REGION Network 1: CAN COT LIEU AGG1
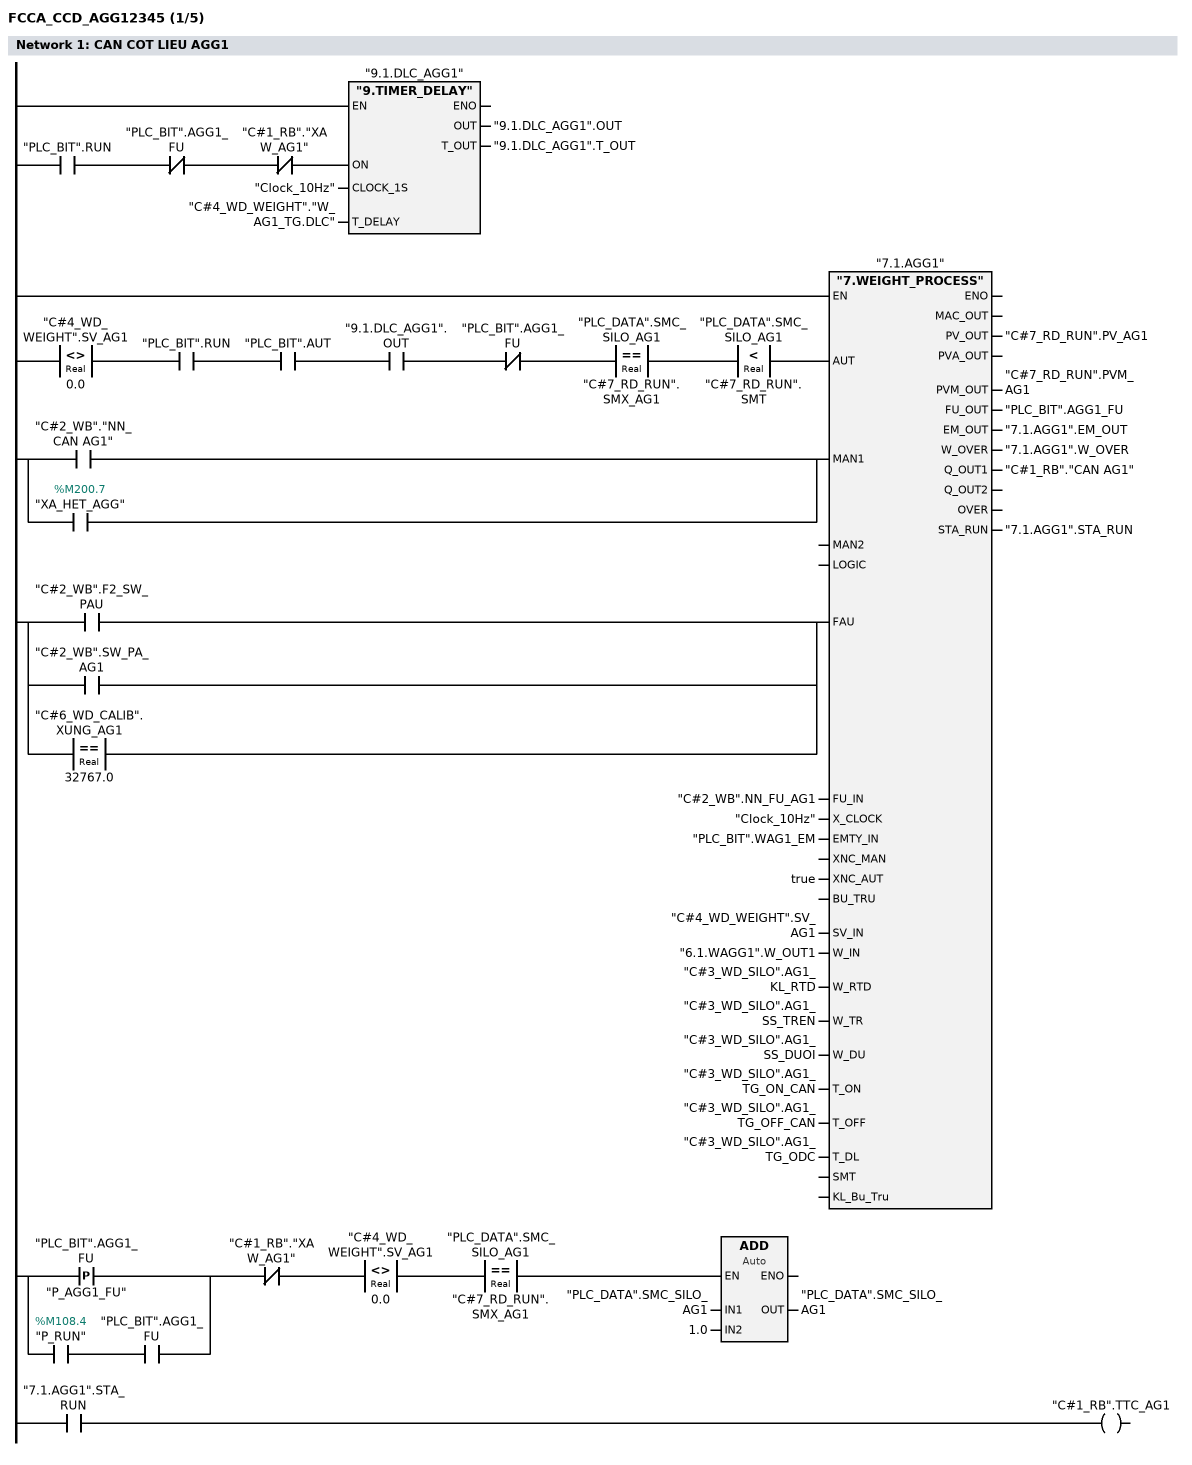
   RUNG wire#powerrail
      "9.1.DLC_AGG1"(ON := wire#w1, CLOCK_1S := "Clock_10Hz", T_DELAY := "C#4_WD_WEIGHT"."W_AG1_TG.DLC", OUT => "9.1.DLC_AGG1".OUT, T_OUT => "9.1.DLC_AGG1".T_OUT)
   END_RUNG
   RUNG wire#powerrail
      Contact( "PLC_BIT".RUN )
      I_Contact( "PLC_BIT".AGG1_FU )
      I_Contact( "C#1_RB"."XA W_AG1" )
   END_RUNG wire#w1
   RUNG wire#powerrail
      "7.1.AGG1"(AUT := wire#w2, MAN1 := wire#w3, FAU := wire#w4, MAN2 :=, LOGIC :=, FU_IN := "C#2_WB".NN_FU_AG1, X_CLOCK := "Clock_10Hz", EMTY_IN := "PLC_BIT".WAG1_EM, XNC_MAN :=, XNC_AUT := true, BU_TRU :=, SV_IN := "C#4_WD_WEIGHT".SV_AG1, W_IN := "6.1.WAGG1".W_OUT1, W_RTD := "C#3_WD_SILO".AG1_KL_RTD, W_TR := "C#3_WD_SILO".AG1_SS_TREN, W_DU := "C#3_WD_SILO".AG1_SS_DUOI, T_ON := "C#3_WD_SILO".AG1_TG_ON_CAN, T_OFF := "C#3_WD_SILO".AG1_TG_OFF_CAN, T_DL := "C#3_WD_SILO".AG1_TG_ODC, SMT :=, KL_Bu_Tru :=, MAC_OUT =>, PV_OUT => "C#7_RD_RUN".PV_AG1, PVA_OUT =>, PVM_OUT => "C#7_RD_RUN".PVM_AG1, FU_OUT => "PLC_BIT".AGG1_FU, EM_OUT => "7.1.AGG1".EM_OUT, W_OVER => "7.1.AGG1".W_OVER, Q_OUT1 => "C#1_RB"."CAN AG1", Q_OUT2 =>, OVER =>, STA_RUN => "7.1.AGG1".STA_RUN)
   END_RUNG
   RUNG wire#powerrail
      { S7_Templates := "SrcType := Real" } NE_Contact(in1 := "C#4_WD_WEIGHT".SV_AG1, in2 := 0.0)
      Contact( "PLC_BIT".RUN )
      Contact( "PLC_BIT".AUT )
      Contact( "9.1.DLC_AGG1".OUT )
      I_Contact( "PLC_BIT".AGG1_FU )
      { S7_Templates := "SrcType := Real" } EQ_Contact(in1 := "PLC_DATA".SMC_SILO_AG1, in2 := "C#7_RD_RUN".SMX_AG1)
      { S7_Templates := "SrcType := Real" } LT_Contact(in1 := "PLC_DATA".SMC_SILO_AG1, in2 := "C#7_RD_RUN".SMT)
   END_RUNG wire#w2
   RUNG wire#powerrail
      Contact( "C#2_WB"."NN_CAN AG1" )
   END_RUNG wire#w3
   RUNG wire#powerrail
      Contact( "XA_HET_AGG" )
   END_RUNG wire#w3
   RUNG wire#powerrail
      Contact( "C#2_WB".F2_SW_PAU )
   END_RUNG wire#w4
   RUNG wire#powerrail
      Contact( "C#2_WB".SW_PA_AG1 )
   END_RUNG wire#w4
   RUNG wire#powerrail
      { S7_Templates := "SrcType := Real" } EQ_Contact(in1 := "C#6_WD_CALIB".XUNG_AG1, in2 := 32767.0)
   END_RUNG wire#w4
   RUNG wire#powerrail
      P_Contact(operand := "PLC_BIT".AGG1_FU, bit := "P_AGG1_FU")
      wire#w5
      I_Contact( "C#1_RB"."XA W_AG1" )
      { S7_Templates := "SrcType := Real" } NE_Contact(in1 := "C#4_WD_WEIGHT".SV_AG1, in2 := 0.0)
      { S7_Templates := "SrcType := Real" } EQ_Contact(in1 := "PLC_DATA".SMC_SILO_AG1, in2 := "C#7_RD_RUN".SMX_AG1)
      Add(in1 := "PLC_DATA".SMC_SILO_AG1, in2 := 1.0, out => "PLC_DATA".SMC_SILO_AG1)
   END_RUNG
   RUNG wire#powerrail
      Contact( "P_RUN" )
      Contact( "PLC_BIT".AGG1_FU )
   END_RUNG wire#w5
   RUNG wire#powerrail
      Contact( "7.1.AGG1".STA_RUN )
      Coil( "C#1_RB".TTC_AG1 )
   END_RUNG
   // the same network as SCL:
   "9.1.DLC_AGG1"(ON := "PLC_BIT".RUN AND NOT "PLC_BIT".AGG1_FU AND NOT "C#1_RB"."XA W_AG1",   // "9.TIMER_DELAY"
                  CLOCK_1S := "Clock_10Hz",
                  T_DELAY := "C#4_WD_WEIGHT"."W_AG1_TG.DLC",
                  OUT => "9.1.DLC_AGG1".OUT,
                  T_OUT => "9.1.DLC_AGG1".T_OUT);
   "7.1.AGG1"(AUT := ("C#4_WD_WEIGHT".SV_AG1 <> 0.0) AND "PLC_BIT".RUN AND "PLC_BIT".AUT AND "9.1.DLC_AGG1".OUT AND NOT "PLC_BIT".AGG1_FU AND ("PLC_DATA".SMC_SILO_AG1 = "C#7_RD_RUN".SMX_AG1) AND ("PLC_DATA".SMC_SILO_AG1 < "C#7_RD_RUN".SMT),   // "7.WEIGHT_PROCESS"
              MAN1 := "C#2_WB"."NN_CAN AG1" OR "XA_HET_AGG",
              FAU := "C#2_WB".F2_SW_PAU OR "C#2_WB".SW_PA_AG1 OR ("C#6_WD_CALIB".XUNG_AG1 = 32767.0),
              FU_IN := "C#2_WB".NN_FU_AG1,
              X_CLOCK := "Clock_10Hz",
              EMTY_IN := "PLC_BIT".WAG1_EM,
              XNC_AUT := true,
              SV_IN := "C#4_WD_WEIGHT".SV_AG1,
              W_IN := "6.1.WAGG1".W_OUT1,
              W_RTD := "C#3_WD_SILO".AG1_KL_RTD,
              W_TR := "C#3_WD_SILO".AG1_SS_TREN,
              W_DU := "C#3_WD_SILO".AG1_SS_DUOI,
              T_ON := "C#3_WD_SILO".AG1_TG_ON_CAN,
              T_OFF := "C#3_WD_SILO".AG1_TG_OFF_CAN,
              T_DL := "C#3_WD_SILO".AG1_TG_ODC,
              PV_OUT => "C#7_RD_RUN".PV_AG1,
              PVM_OUT => "C#7_RD_RUN".PVM_AG1,
              FU_OUT => "PLC_BIT".AGG1_FU,
              EM_OUT => "7.1.AGG1".EM_OUT,
              W_OVER => "7.1.AGG1".W_OVER,
              Q_OUT1 => "C#1_RB"."CAN AG1",
              STA_RUN => "7.1.AGG1".STA_RUN);
   #_w1 := "PLC_BIT".AGG1_FU AND NOT "P_AGG1_FU";   // rising edge of "PLC_BIT".AGG1_FU
   "P_AGG1_FU" := "PLC_BIT".AGG1_FU;
   IF (#_w1 OR ("P_RUN" AND "PLC_BIT".AGG1_FU)) AND NOT "C#1_RB"."XA W_AG1" AND ("C#4_WD_WEIGHT".SV_AG1 <> 0.0) AND ("PLC_DATA".SMC_SILO_AG1 = "C#7_RD_RUN".SMX_AG1) THEN
       "PLC_DATA".SMC_SILO_AG1 := "PLC_DATA".SMC_SILO_AG1 + 1.0;
   END_IF;
   "C#1_RB".TTC_AG1 := "7.1.AGG1".STA_RUN;
END_REGION

REGION Network 2: CAN COT LIEU AGG2
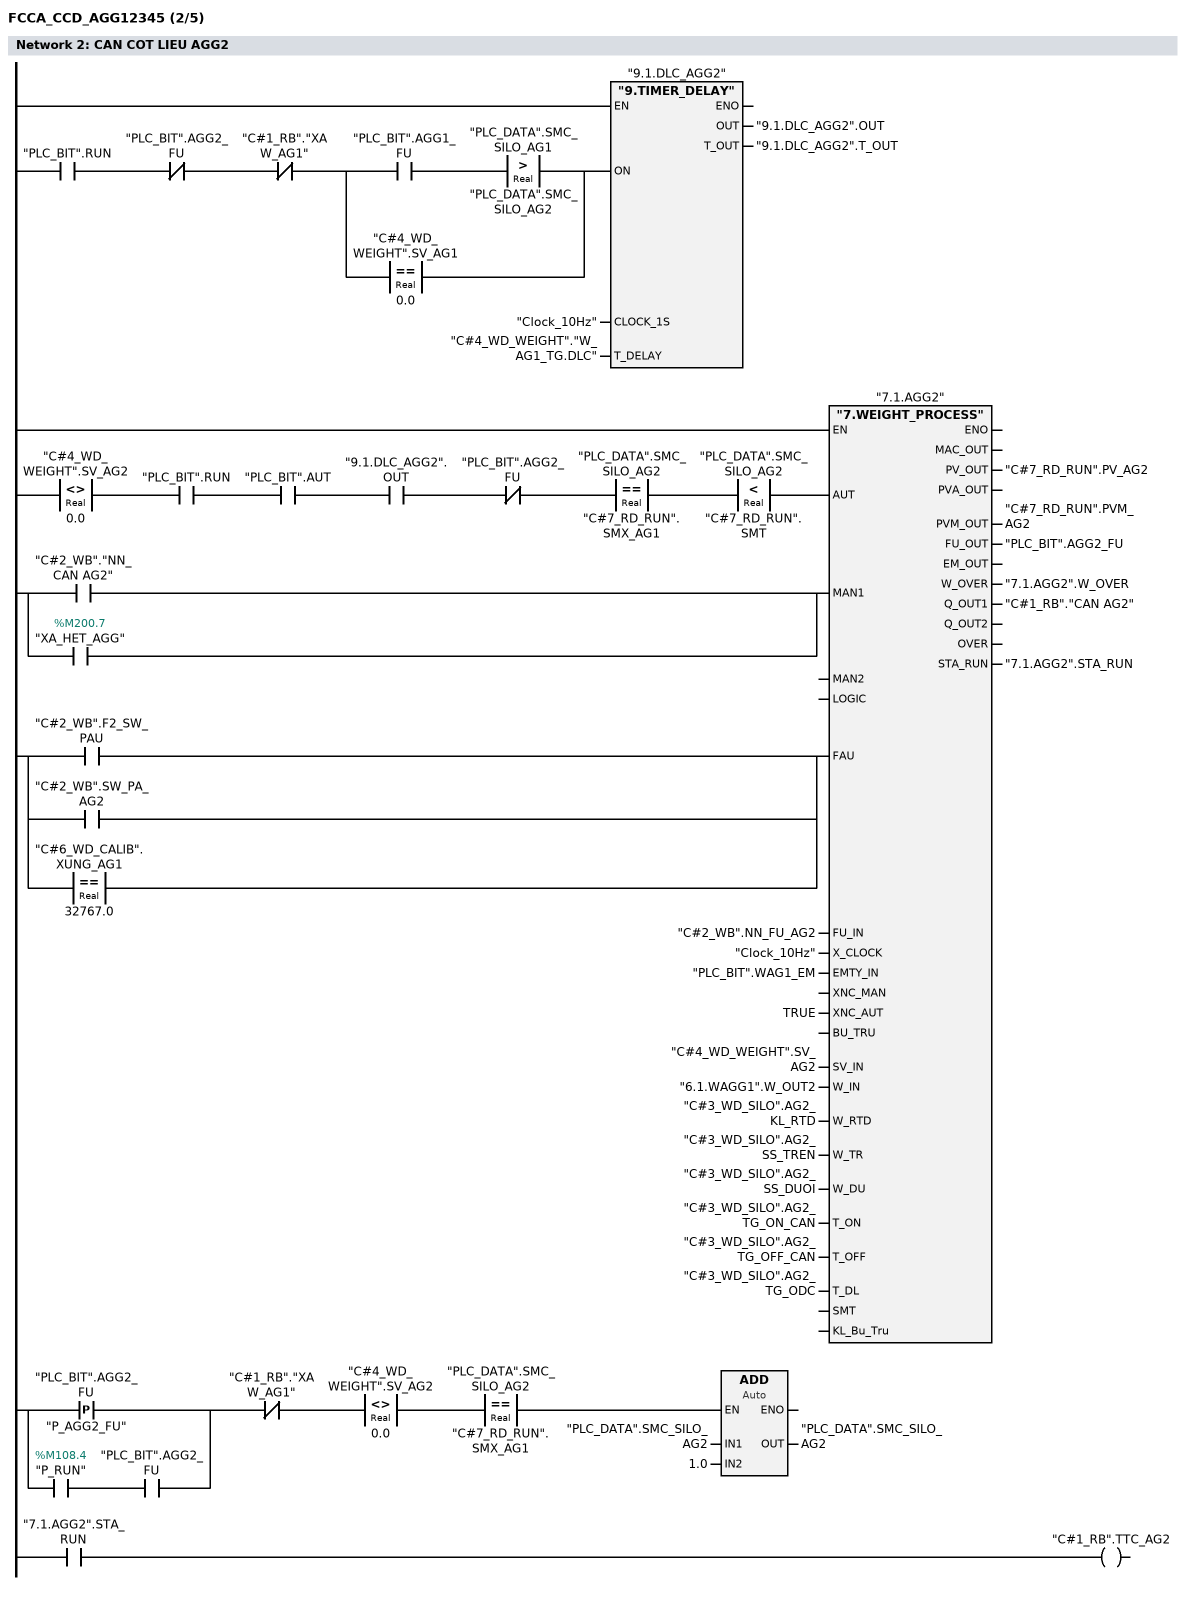
   RUNG wire#powerrail
      "9.1.DLC_AGG2"(ON := wire#w2, CLOCK_1S := "Clock_10Hz", T_DELAY := "C#4_WD_WEIGHT"."W_AG1_TG.DLC", OUT => "9.1.DLC_AGG2".OUT, T_OUT => "9.1.DLC_AGG2".T_OUT)
   END_RUNG
   RUNG wire#powerrail
      Contact( "PLC_BIT".RUN )
      I_Contact( "PLC_BIT".AGG2_FU )
      I_Contact( "C#1_RB"."XA W_AG1" )
      wire#w1
      Contact( "PLC_BIT".AGG1_FU )
      { S7_Templates := "SrcType := Real" } GT_Contact(in1 := "PLC_DATA".SMC_SILO_AG1, in2 := "PLC_DATA".SMC_SILO_AG2)
   END_RUNG wire#w2
   RUNG wire#w1
      { S7_Templates := "SrcType := Real" } EQ_Contact(in1 := "C#4_WD_WEIGHT".SV_AG1, in2 := 0.0)
   END_RUNG wire#w2
   RUNG wire#powerrail
      "7.1.AGG2"(AUT := wire#w3, MAN1 := wire#w4, FAU := wire#w5, MAN2 :=, LOGIC :=, FU_IN := "C#2_WB".NN_FU_AG2, X_CLOCK := "Clock_10Hz", EMTY_IN := "PLC_BIT".WAG1_EM, XNC_MAN :=, XNC_AUT := TRUE, BU_TRU :=, SV_IN := "C#4_WD_WEIGHT".SV_AG2, W_IN := "6.1.WAGG1".W_OUT2, W_RTD := "C#3_WD_SILO".AG2_KL_RTD, W_TR := "C#3_WD_SILO".AG2_SS_TREN, W_DU := "C#3_WD_SILO".AG2_SS_DUOI, T_ON := "C#3_WD_SILO".AG2_TG_ON_CAN, T_OFF := "C#3_WD_SILO".AG2_TG_OFF_CAN, T_DL := "C#3_WD_SILO".AG2_TG_ODC, SMT :=, KL_Bu_Tru :=, MAC_OUT =>, PV_OUT => "C#7_RD_RUN".PV_AG2, PVA_OUT =>, PVM_OUT => "C#7_RD_RUN".PVM_AG2, FU_OUT => "PLC_BIT".AGG2_FU, EM_OUT =>, W_OVER => "7.1.AGG2".W_OVER, Q_OUT1 => "C#1_RB"."CAN AG2", Q_OUT2 =>, OVER =>, STA_RUN => "7.1.AGG2".STA_RUN)
   END_RUNG
   RUNG wire#powerrail
      { S7_Templates := "SrcType := Real" } NE_Contact(in1 := "C#4_WD_WEIGHT".SV_AG2, in2 := 0.0)
      Contact( "PLC_BIT".RUN )
      Contact( "PLC_BIT".AUT )
      Contact( "9.1.DLC_AGG2".OUT )
      I_Contact( "PLC_BIT".AGG2_FU )
      { S7_Templates := "SrcType := Real" } EQ_Contact(in1 := "PLC_DATA".SMC_SILO_AG2, in2 := "C#7_RD_RUN".SMX_AG1)
      { S7_Templates := "SrcType := Real" } LT_Contact(in1 := "PLC_DATA".SMC_SILO_AG2, in2 := "C#7_RD_RUN".SMT)
   END_RUNG wire#w3
   RUNG wire#powerrail
      Contact( "C#2_WB"."NN_CAN AG2" )
   END_RUNG wire#w4
   RUNG wire#powerrail
      Contact( "XA_HET_AGG" )
   END_RUNG wire#w4
   RUNG wire#powerrail
      Contact( "C#2_WB".F2_SW_PAU )
   END_RUNG wire#w5
   RUNG wire#powerrail
      Contact( "C#2_WB".SW_PA_AG2 )
   END_RUNG wire#w5
   RUNG wire#powerrail
      { S7_Templates := "SrcType := Real" } EQ_Contact(in1 := "C#6_WD_CALIB".XUNG_AG1, in2 := 32767.0)
   END_RUNG wire#w5
   RUNG wire#powerrail
      P_Contact(operand := "PLC_BIT".AGG2_FU, bit := "P_AGG2_FU")
      wire#w6
      I_Contact( "C#1_RB"."XA W_AG1" )
      { S7_Templates := "SrcType := Real" } NE_Contact(in1 := "C#4_WD_WEIGHT".SV_AG2, in2 := 0.0)
      { S7_Templates := "SrcType := Real" } EQ_Contact(in1 := "PLC_DATA".SMC_SILO_AG2, in2 := "C#7_RD_RUN".SMX_AG1)
      Add(in1 := "PLC_DATA".SMC_SILO_AG2, in2 := 1.0, out => "PLC_DATA".SMC_SILO_AG2)
   END_RUNG
   RUNG wire#powerrail
      Contact( "P_RUN" )
      Contact( "PLC_BIT".AGG2_FU )
   END_RUNG wire#w6
   RUNG wire#powerrail
      Contact( "7.1.AGG2".STA_RUN )
      Coil( "C#1_RB".TTC_AG2 )
   END_RUNG
   // the same network as SCL:
   "9.1.DLC_AGG2"(ON := "PLC_BIT".RUN AND NOT "PLC_BIT".AGG2_FU AND NOT "C#1_RB"."XA W_AG1" AND (("PLC_BIT".AGG1_FU AND ("PLC_DATA".SMC_SILO_AG1 > "PLC_DATA".SMC_SILO_AG2)) OR ("C#4_WD_WEIGHT".SV_AG1 = 0.0)),   // "9.TIMER_DELAY"
                  CLOCK_1S := "Clock_10Hz",
                  T_DELAY := "C#4_WD_WEIGHT"."W_AG1_TG.DLC",
                  OUT => "9.1.DLC_AGG2".OUT,
                  T_OUT => "9.1.DLC_AGG2".T_OUT);
   "7.1.AGG2"(AUT := ("C#4_WD_WEIGHT".SV_AG2 <> 0.0) AND "PLC_BIT".RUN AND "PLC_BIT".AUT AND "9.1.DLC_AGG2".OUT AND NOT "PLC_BIT".AGG2_FU AND ("PLC_DATA".SMC_SILO_AG2 = "C#7_RD_RUN".SMX_AG1) AND ("PLC_DATA".SMC_SILO_AG2 < "C#7_RD_RUN".SMT),   // "7.WEIGHT_PROCESS"
              MAN1 := "C#2_WB"."NN_CAN AG2" OR "XA_HET_AGG",
              FAU := "C#2_WB".F2_SW_PAU OR "C#2_WB".SW_PA_AG2 OR ("C#6_WD_CALIB".XUNG_AG1 = 32767.0),
              FU_IN := "C#2_WB".NN_FU_AG2,
              X_CLOCK := "Clock_10Hz",
              EMTY_IN := "PLC_BIT".WAG1_EM,
              XNC_AUT := TRUE,
              SV_IN := "C#4_WD_WEIGHT".SV_AG2,
              W_IN := "6.1.WAGG1".W_OUT2,
              W_RTD := "C#3_WD_SILO".AG2_KL_RTD,
              W_TR := "C#3_WD_SILO".AG2_SS_TREN,
              W_DU := "C#3_WD_SILO".AG2_SS_DUOI,
              T_ON := "C#3_WD_SILO".AG2_TG_ON_CAN,
              T_OFF := "C#3_WD_SILO".AG2_TG_OFF_CAN,
              T_DL := "C#3_WD_SILO".AG2_TG_ODC,
              PV_OUT => "C#7_RD_RUN".PV_AG2,
              PVM_OUT => "C#7_RD_RUN".PVM_AG2,
              FU_OUT => "PLC_BIT".AGG2_FU,
              W_OVER => "7.1.AGG2".W_OVER,
              Q_OUT1 => "C#1_RB"."CAN AG2",
              STA_RUN => "7.1.AGG2".STA_RUN);
   #_w1 := "PLC_BIT".AGG2_FU AND NOT "P_AGG2_FU";   // rising edge of "PLC_BIT".AGG2_FU
   "P_AGG2_FU" := "PLC_BIT".AGG2_FU;
   IF (#_w1 OR ("P_RUN" AND "PLC_BIT".AGG2_FU)) AND NOT "C#1_RB"."XA W_AG1" AND ("C#4_WD_WEIGHT".SV_AG2 <> 0.0) AND ("PLC_DATA".SMC_SILO_AG2 = "C#7_RD_RUN".SMX_AG1) THEN
       "PLC_DATA".SMC_SILO_AG2 := "PLC_DATA".SMC_SILO_AG2 + 1.0;
   END_IF;
   "C#1_RB".TTC_AG2 := "7.1.AGG2".STA_RUN;
END_REGION

REGION Network 3: CAN COT LIEU AGG3
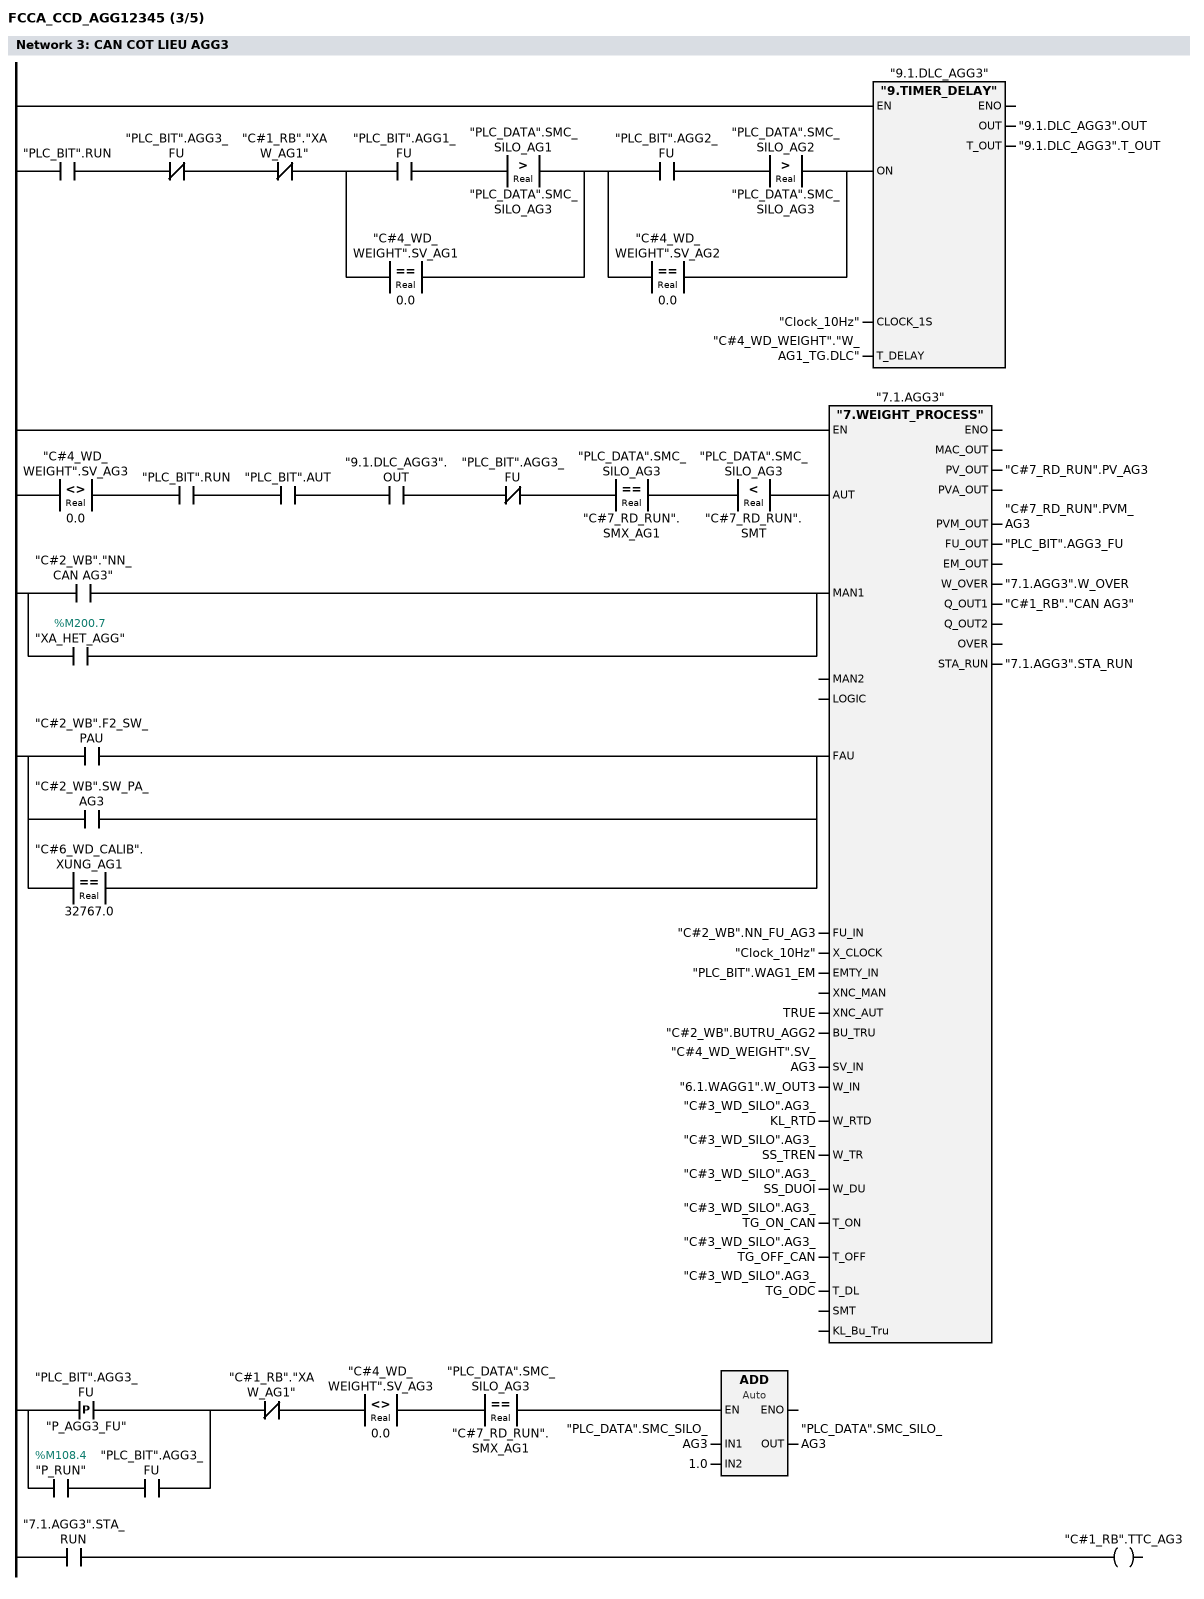
   RUNG wire#powerrail
      "9.1.DLC_AGG3"(ON := wire#w3, CLOCK_1S := "Clock_10Hz", T_DELAY := "C#4_WD_WEIGHT"."W_AG1_TG.DLC", OUT => "9.1.DLC_AGG3".OUT, T_OUT => "9.1.DLC_AGG3".T_OUT)
   END_RUNG
   RUNG wire#powerrail
      Contact( "PLC_BIT".RUN )
      I_Contact( "PLC_BIT".AGG3_FU )
      I_Contact( "C#1_RB"."XA W_AG1" )
      wire#w1
      Contact( "PLC_BIT".AGG1_FU )
      { S7_Templates := "SrcType := Real" } GT_Contact(in1 := "PLC_DATA".SMC_SILO_AG1, in2 := "PLC_DATA".SMC_SILO_AG3)
      wire#w2
      Contact( "PLC_BIT".AGG2_FU )
      { S7_Templates := "SrcType := Real" } GT_Contact(in1 := "PLC_DATA".SMC_SILO_AG2, in2 := "PLC_DATA".SMC_SILO_AG3)
   END_RUNG wire#w3
   RUNG wire#w1
      { S7_Templates := "SrcType := Real" } EQ_Contact(in1 := "C#4_WD_WEIGHT".SV_AG1, in2 := 0.0)
   END_RUNG wire#w2
   RUNG wire#w2
      { S7_Templates := "SrcType := Real" } EQ_Contact(in1 := "C#4_WD_WEIGHT".SV_AG2, in2 := 0.0)
   END_RUNG wire#w3
   RUNG wire#powerrail
      "7.1.AGG3"(AUT := wire#w4, MAN1 := wire#w5, FAU := wire#w6, MAN2 :=, LOGIC :=, FU_IN := "C#2_WB".NN_FU_AG3, X_CLOCK := "Clock_10Hz", EMTY_IN := "PLC_BIT".WAG1_EM, XNC_MAN :=, XNC_AUT := TRUE, BU_TRU := "C#2_WB".BUTRU_AGG2, SV_IN := "C#4_WD_WEIGHT".SV_AG3, W_IN := "6.1.WAGG1".W_OUT3, W_RTD := "C#3_WD_SILO".AG3_KL_RTD, W_TR := "C#3_WD_SILO".AG3_SS_TREN, W_DU := "C#3_WD_SILO".AG3_SS_DUOI, T_ON := "C#3_WD_SILO".AG3_TG_ON_CAN, T_OFF := "C#3_WD_SILO".AG3_TG_OFF_CAN, T_DL := "C#3_WD_SILO".AG3_TG_ODC, SMT :=, KL_Bu_Tru :=, MAC_OUT =>, PV_OUT => "C#7_RD_RUN".PV_AG3, PVA_OUT =>, PVM_OUT => "C#7_RD_RUN".PVM_AG3, FU_OUT => "PLC_BIT".AGG3_FU, EM_OUT =>, W_OVER => "7.1.AGG3".W_OVER, Q_OUT1 => "C#1_RB"."CAN AG3", Q_OUT2 =>, OVER =>, STA_RUN => "7.1.AGG3".STA_RUN)
   END_RUNG
   RUNG wire#powerrail
      { S7_Templates := "SrcType := Real" } NE_Contact(in1 := "C#4_WD_WEIGHT".SV_AG3, in2 := 0.0)
      Contact( "PLC_BIT".RUN )
      Contact( "PLC_BIT".AUT )
      Contact( "9.1.DLC_AGG3".OUT )
      I_Contact( "PLC_BIT".AGG3_FU )
      { S7_Templates := "SrcType := Real" } EQ_Contact(in1 := "PLC_DATA".SMC_SILO_AG3, in2 := "C#7_RD_RUN".SMX_AG1)
      { S7_Templates := "SrcType := Real" } LT_Contact(in1 := "PLC_DATA".SMC_SILO_AG3, in2 := "C#7_RD_RUN".SMT)
   END_RUNG wire#w4
   RUNG wire#powerrail
      Contact( "C#2_WB"."NN_CAN AG3" )
   END_RUNG wire#w5
   RUNG wire#powerrail
      Contact( "XA_HET_AGG" )
   END_RUNG wire#w5
   RUNG wire#powerrail
      Contact( "C#2_WB".F2_SW_PAU )
   END_RUNG wire#w6
   RUNG wire#powerrail
      Contact( "C#2_WB".SW_PA_AG3 )
   END_RUNG wire#w6
   RUNG wire#powerrail
      { S7_Templates := "SrcType := Real" } EQ_Contact(in1 := "C#6_WD_CALIB".XUNG_AG1, in2 := 32767.0)
   END_RUNG wire#w6
   RUNG wire#powerrail
      P_Contact(operand := "PLC_BIT".AGG3_FU, bit := "P_AGG3_FU")
      wire#w7
      I_Contact( "C#1_RB"."XA W_AG1" )
      { S7_Templates := "SrcType := Real" } NE_Contact(in1 := "C#4_WD_WEIGHT".SV_AG3, in2 := 0.0)
      { S7_Templates := "SrcType := Real" } EQ_Contact(in1 := "PLC_DATA".SMC_SILO_AG3, in2 := "C#7_RD_RUN".SMX_AG1)
      Add(in1 := "PLC_DATA".SMC_SILO_AG3, in2 := 1.0, out => "PLC_DATA".SMC_SILO_AG3)
   END_RUNG
   RUNG wire#powerrail
      Contact( "P_RUN" )
      Contact( "PLC_BIT".AGG3_FU )
   END_RUNG wire#w7
   RUNG wire#powerrail
      Contact( "7.1.AGG3".STA_RUN )
      Coil( "C#1_RB".TTC_AG3 )
   END_RUNG
   // the same network as SCL:
   "9.1.DLC_AGG3"(ON := "PLC_BIT".RUN AND NOT "PLC_BIT".AGG3_FU AND NOT "C#1_RB"."XA W_AG1" AND (("PLC_BIT".AGG1_FU AND ("PLC_DATA".SMC_SILO_AG1 > "PLC_DATA".SMC_SILO_AG3)) OR ("C#4_WD_WEIGHT".SV_AG1 = 0.0)) AND (("PLC_BIT".AGG2_FU AND ("PLC_DATA".SMC_SILO_AG2 > "PLC_DATA".SMC_SILO_AG3)) OR ("C#4_WD_WEIGHT".SV_AG2 = 0.0)),   // "9.TIMER_DELAY"
                  CLOCK_1S := "Clock_10Hz",
                  T_DELAY := "C#4_WD_WEIGHT"."W_AG1_TG.DLC",
                  OUT => "9.1.DLC_AGG3".OUT,
                  T_OUT => "9.1.DLC_AGG3".T_OUT);
   "7.1.AGG3"(AUT := ("C#4_WD_WEIGHT".SV_AG3 <> 0.0) AND "PLC_BIT".RUN AND "PLC_BIT".AUT AND "9.1.DLC_AGG3".OUT AND NOT "PLC_BIT".AGG3_FU AND ("PLC_DATA".SMC_SILO_AG3 = "C#7_RD_RUN".SMX_AG1) AND ("PLC_DATA".SMC_SILO_AG3 < "C#7_RD_RUN".SMT),   // "7.WEIGHT_PROCESS"
              MAN1 := "C#2_WB"."NN_CAN AG3" OR "XA_HET_AGG",
              FAU := "C#2_WB".F2_SW_PAU OR "C#2_WB".SW_PA_AG3 OR ("C#6_WD_CALIB".XUNG_AG1 = 32767.0),
              FU_IN := "C#2_WB".NN_FU_AG3,
              X_CLOCK := "Clock_10Hz",
              EMTY_IN := "PLC_BIT".WAG1_EM,
              XNC_AUT := TRUE,
              BU_TRU := "C#2_WB".BUTRU_AGG2,
              SV_IN := "C#4_WD_WEIGHT".SV_AG3,
              W_IN := "6.1.WAGG1".W_OUT3,
              W_RTD := "C#3_WD_SILO".AG3_KL_RTD,
              W_TR := "C#3_WD_SILO".AG3_SS_TREN,
              W_DU := "C#3_WD_SILO".AG3_SS_DUOI,
              T_ON := "C#3_WD_SILO".AG3_TG_ON_CAN,
              T_OFF := "C#3_WD_SILO".AG3_TG_OFF_CAN,
              T_DL := "C#3_WD_SILO".AG3_TG_ODC,
              PV_OUT => "C#7_RD_RUN".PV_AG3,
              PVM_OUT => "C#7_RD_RUN".PVM_AG3,
              FU_OUT => "PLC_BIT".AGG3_FU,
              W_OVER => "7.1.AGG3".W_OVER,
              Q_OUT1 => "C#1_RB"."CAN AG3",
              STA_RUN => "7.1.AGG3".STA_RUN);
   #_w1 := "PLC_BIT".AGG3_FU AND NOT "P_AGG3_FU";   // rising edge of "PLC_BIT".AGG3_FU
   "P_AGG3_FU" := "PLC_BIT".AGG3_FU;
   IF (#_w1 OR ("P_RUN" AND "PLC_BIT".AGG3_FU)) AND NOT "C#1_RB"."XA W_AG1" AND ("C#4_WD_WEIGHT".SV_AG3 <> 0.0) AND ("PLC_DATA".SMC_SILO_AG3 = "C#7_RD_RUN".SMX_AG1) THEN
       "PLC_DATA".SMC_SILO_AG3 := "PLC_DATA".SMC_SILO_AG3 + 1.0;
   END_IF;
   "C#1_RB".TTC_AG3 := "7.1.AGG3".STA_RUN;
END_REGION

REGION Network 4: CAN COT LIEU AGG4
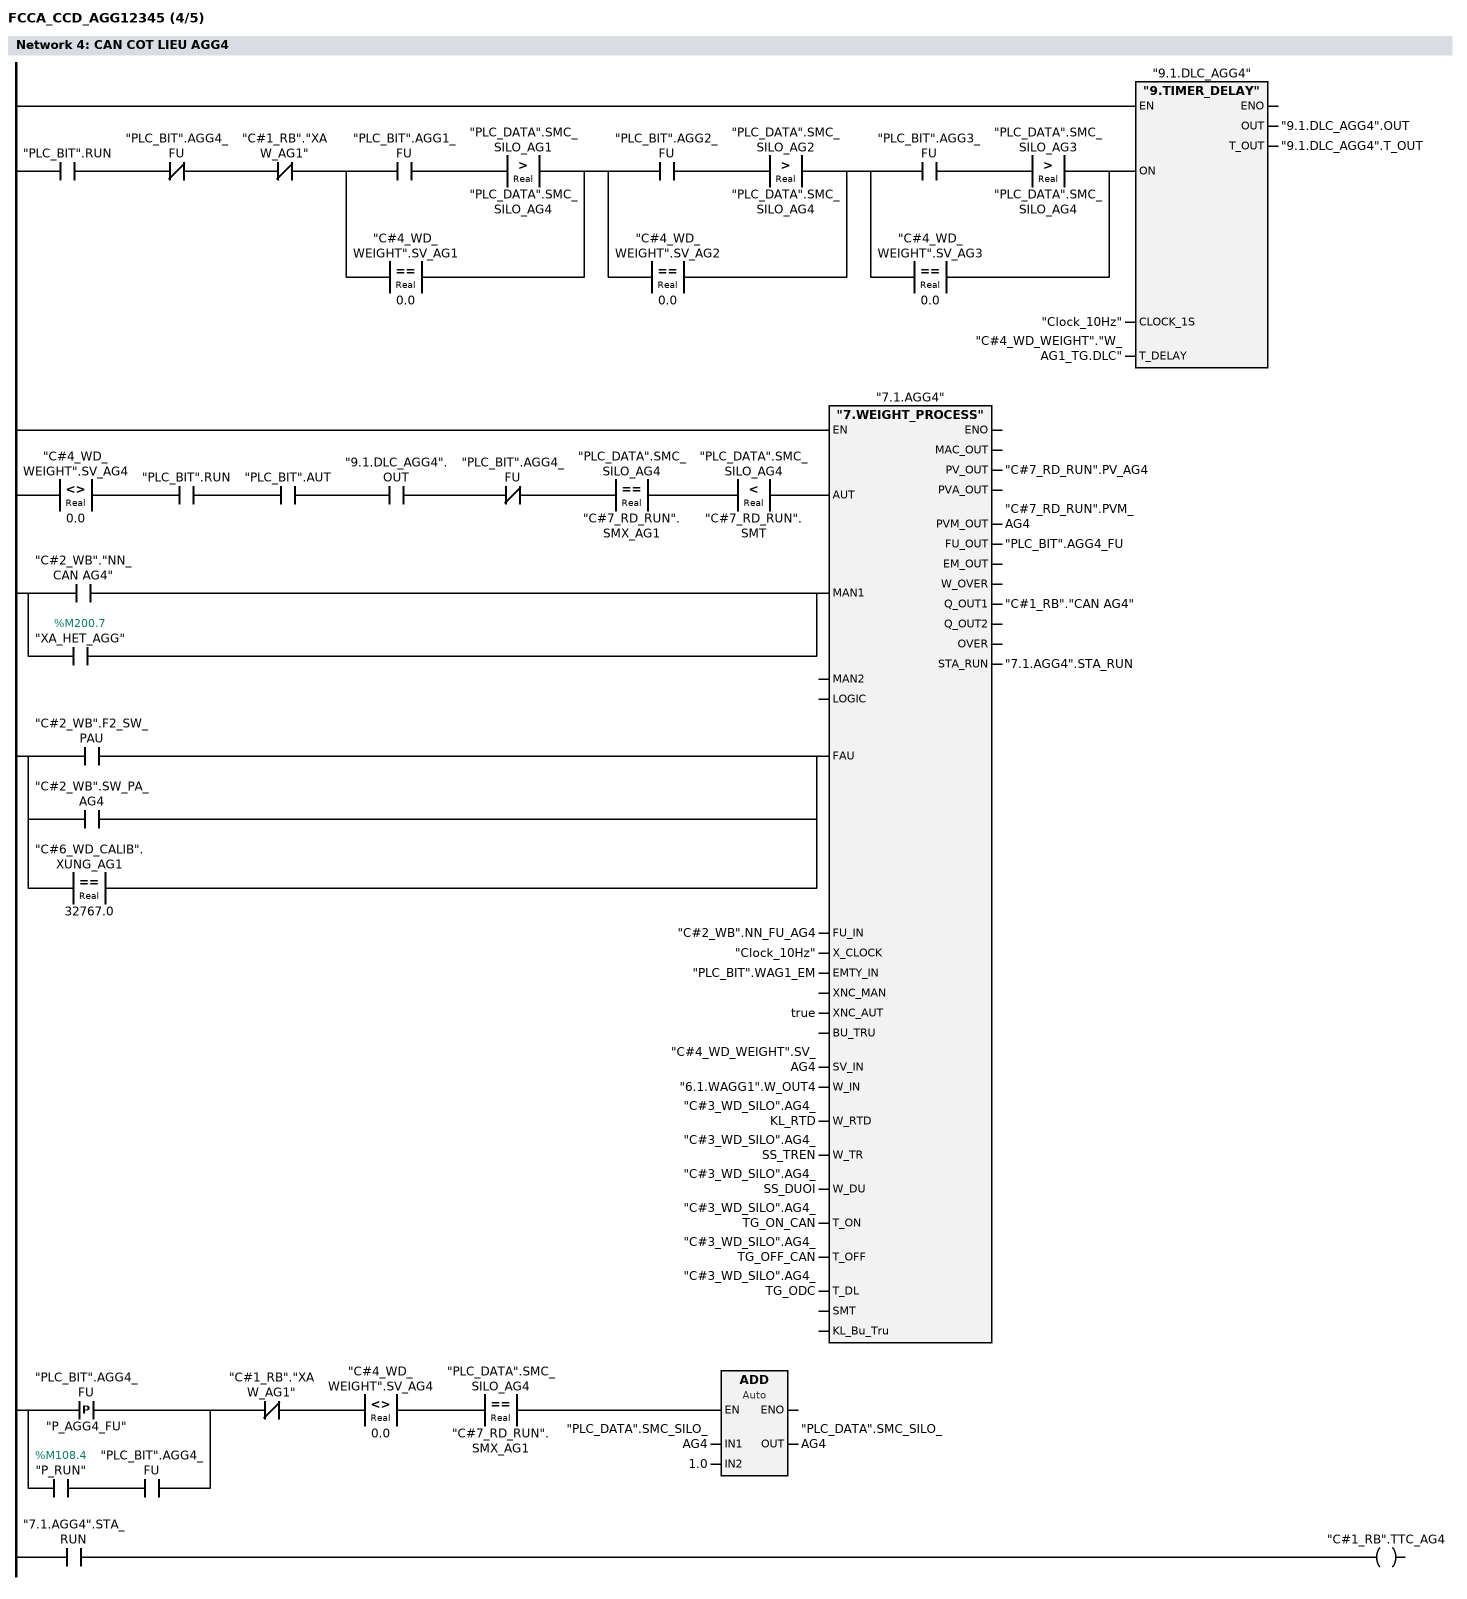
   RUNG wire#powerrail
      "9.1.DLC_AGG4"(ON := wire#w4, CLOCK_1S := "Clock_10Hz", T_DELAY := "C#4_WD_WEIGHT"."W_AG1_TG.DLC", OUT => "9.1.DLC_AGG4".OUT, T_OUT => "9.1.DLC_AGG4".T_OUT)
   END_RUNG
   RUNG wire#powerrail
      Contact( "PLC_BIT".RUN )
      I_Contact( "PLC_BIT".AGG4_FU )
      I_Contact( "C#1_RB"."XA W_AG1" )
      wire#w1
      Contact( "PLC_BIT".AGG1_FU )
      { S7_Templates := "SrcType := Real" } GT_Contact(in1 := "PLC_DATA".SMC_SILO_AG1, in2 := "PLC_DATA".SMC_SILO_AG4)
      wire#w2
      Contact( "PLC_BIT".AGG2_FU )
      { S7_Templates := "SrcType := Real" } GT_Contact(in1 := "PLC_DATA".SMC_SILO_AG2, in2 := "PLC_DATA".SMC_SILO_AG4)
      wire#w3
      Contact( "PLC_BIT".AGG3_FU )
      { S7_Templates := "SrcType := Real" } GT_Contact(in1 := "PLC_DATA".SMC_SILO_AG3, in2 := "PLC_DATA".SMC_SILO_AG4)
   END_RUNG wire#w4
   RUNG wire#w1
      { S7_Templates := "SrcType := Real" } EQ_Contact(in1 := "C#4_WD_WEIGHT".SV_AG1, in2 := 0.0)
   END_RUNG wire#w2
   RUNG wire#w2
      { S7_Templates := "SrcType := Real" } EQ_Contact(in1 := "C#4_WD_WEIGHT".SV_AG2, in2 := 0.0)
   END_RUNG wire#w3
   RUNG wire#w3
      { S7_Templates := "SrcType := Real" } EQ_Contact(in1 := "C#4_WD_WEIGHT".SV_AG3, in2 := 0.0)
   END_RUNG wire#w4
   RUNG wire#powerrail
      "7.1.AGG4"(AUT := wire#w5, MAN1 := wire#w6, FAU := wire#w7, MAN2 :=, LOGIC :=, FU_IN := "C#2_WB".NN_FU_AG4, X_CLOCK := "Clock_10Hz", EMTY_IN := "PLC_BIT".WAG1_EM, XNC_MAN :=, XNC_AUT := true, BU_TRU :=, SV_IN := "C#4_WD_WEIGHT".SV_AG4, W_IN := "6.1.WAGG1".W_OUT4, W_RTD := "C#3_WD_SILO".AG4_KL_RTD, W_TR := "C#3_WD_SILO".AG4_SS_TREN, W_DU := "C#3_WD_SILO".AG4_SS_DUOI, T_ON := "C#3_WD_SILO".AG4_TG_ON_CAN, T_OFF := "C#3_WD_SILO".AG4_TG_OFF_CAN, T_DL := "C#3_WD_SILO".AG4_TG_ODC, SMT :=, KL_Bu_Tru :=, MAC_OUT =>, PV_OUT => "C#7_RD_RUN".PV_AG4, PVA_OUT =>, PVM_OUT => "C#7_RD_RUN".PVM_AG4, FU_OUT => "PLC_BIT".AGG4_FU, EM_OUT =>, W_OVER =>, Q_OUT1 => "C#1_RB"."CAN AG4", Q_OUT2 =>, OVER =>, STA_RUN => "7.1.AGG4".STA_RUN)
   END_RUNG
   RUNG wire#powerrail
      { S7_Templates := "SrcType := Real" } NE_Contact(in1 := "C#4_WD_WEIGHT".SV_AG4, in2 := 0.0)
      Contact( "PLC_BIT".RUN )
      Contact( "PLC_BIT".AUT )
      Contact( "9.1.DLC_AGG4".OUT )
      I_Contact( "PLC_BIT".AGG4_FU )
      { S7_Templates := "SrcType := Real" } EQ_Contact(in1 := "PLC_DATA".SMC_SILO_AG4, in2 := "C#7_RD_RUN".SMX_AG1)
      { S7_Templates := "SrcType := Real" } LT_Contact(in1 := "PLC_DATA".SMC_SILO_AG4, in2 := "C#7_RD_RUN".SMT)
   END_RUNG wire#w5
   RUNG wire#powerrail
      Contact( "C#2_WB"."NN_CAN AG4" )
   END_RUNG wire#w6
   RUNG wire#powerrail
      Contact( "XA_HET_AGG" )
   END_RUNG wire#w6
   RUNG wire#powerrail
      Contact( "C#2_WB".F2_SW_PAU )
   END_RUNG wire#w7
   RUNG wire#powerrail
      Contact( "C#2_WB".SW_PA_AG4 )
   END_RUNG wire#w7
   RUNG wire#powerrail
      { S7_Templates := "SrcType := Real" } EQ_Contact(in1 := "C#6_WD_CALIB".XUNG_AG1, in2 := 32767.0)
   END_RUNG wire#w7
   RUNG wire#powerrail
      P_Contact(operand := "PLC_BIT".AGG4_FU, bit := "P_AGG4_FU")
      wire#w8
      I_Contact( "C#1_RB"."XA W_AG1" )
      { S7_Templates := "SrcType := Real" } NE_Contact(in1 := "C#4_WD_WEIGHT".SV_AG4, in2 := 0.0)
      { S7_Templates := "SrcType := Real" } EQ_Contact(in1 := "PLC_DATA".SMC_SILO_AG4, in2 := "C#7_RD_RUN".SMX_AG1)
      Add(in1 := "PLC_DATA".SMC_SILO_AG4, in2 := 1.0, out => "PLC_DATA".SMC_SILO_AG4)
   END_RUNG
   RUNG wire#powerrail
      Contact( "P_RUN" )
      Contact( "PLC_BIT".AGG4_FU )
   END_RUNG wire#w8
   RUNG wire#powerrail
      Contact( "7.1.AGG4".STA_RUN )
      Coil( "C#1_RB".TTC_AG4 )
   END_RUNG
   // the same network as SCL:
   "9.1.DLC_AGG4"(ON := "PLC_BIT".RUN AND NOT "PLC_BIT".AGG4_FU AND NOT "C#1_RB"."XA W_AG1" AND (("PLC_BIT".AGG1_FU AND ("PLC_DATA".SMC_SILO_AG1 > "PLC_DATA".SMC_SILO_AG4)) OR ("C#4_WD_WEIGHT".SV_AG1 = 0.0)) AND (("PLC_BIT".AGG2_FU AND ("PLC_DATA".SMC_SILO_AG2 > "PLC_DATA".SMC_SILO_AG4)) OR ("C#4_WD_WEIGHT".SV_AG2 = 0.0)) AND (("PLC_BIT".AGG3_FU AND ("PLC_DATA".SMC_SILO_AG3 > "PLC_DATA".SMC_SILO_AG4)) OR ("C#4_WD_WEIGHT".SV_AG3 = 0.0)),   // "9.TIMER_DELAY"
                  CLOCK_1S := "Clock_10Hz",
                  T_DELAY := "C#4_WD_WEIGHT"."W_AG1_TG.DLC",
                  OUT => "9.1.DLC_AGG4".OUT,
                  T_OUT => "9.1.DLC_AGG4".T_OUT);
   "7.1.AGG4"(AUT := ("C#4_WD_WEIGHT".SV_AG4 <> 0.0) AND "PLC_BIT".RUN AND "PLC_BIT".AUT AND "9.1.DLC_AGG4".OUT AND NOT "PLC_BIT".AGG4_FU AND ("PLC_DATA".SMC_SILO_AG4 = "C#7_RD_RUN".SMX_AG1) AND ("PLC_DATA".SMC_SILO_AG4 < "C#7_RD_RUN".SMT),   // "7.WEIGHT_PROCESS"
              MAN1 := "C#2_WB"."NN_CAN AG4" OR "XA_HET_AGG",
              FAU := "C#2_WB".F2_SW_PAU OR "C#2_WB".SW_PA_AG4 OR ("C#6_WD_CALIB".XUNG_AG1 = 32767.0),
              FU_IN := "C#2_WB".NN_FU_AG4,
              X_CLOCK := "Clock_10Hz",
              EMTY_IN := "PLC_BIT".WAG1_EM,
              XNC_AUT := true,
              SV_IN := "C#4_WD_WEIGHT".SV_AG4,
              W_IN := "6.1.WAGG1".W_OUT4,
              W_RTD := "C#3_WD_SILO".AG4_KL_RTD,
              W_TR := "C#3_WD_SILO".AG4_SS_TREN,
              W_DU := "C#3_WD_SILO".AG4_SS_DUOI,
              T_ON := "C#3_WD_SILO".AG4_TG_ON_CAN,
              T_OFF := "C#3_WD_SILO".AG4_TG_OFF_CAN,
              T_DL := "C#3_WD_SILO".AG4_TG_ODC,
              PV_OUT => "C#7_RD_RUN".PV_AG4,
              PVM_OUT => "C#7_RD_RUN".PVM_AG4,
              FU_OUT => "PLC_BIT".AGG4_FU,
              Q_OUT1 => "C#1_RB"."CAN AG4",
              STA_RUN => "7.1.AGG4".STA_RUN);
   #_w1 := "PLC_BIT".AGG4_FU AND NOT "P_AGG4_FU";   // rising edge of "PLC_BIT".AGG4_FU
   "P_AGG4_FU" := "PLC_BIT".AGG4_FU;
   IF (#_w1 OR ("P_RUN" AND "PLC_BIT".AGG4_FU)) AND NOT "C#1_RB"."XA W_AG1" AND ("C#4_WD_WEIGHT".SV_AG4 <> 0.0) AND ("PLC_DATA".SMC_SILO_AG4 = "C#7_RD_RUN".SMX_AG1) THEN
       "PLC_DATA".SMC_SILO_AG4 := "PLC_DATA".SMC_SILO_AG4 + 1.0;
   END_IF;
   "C#1_RB".TTC_AG4 := "7.1.AGG4".STA_RUN;
END_REGION

REGION Network 5: Trạng thái cân Ag4
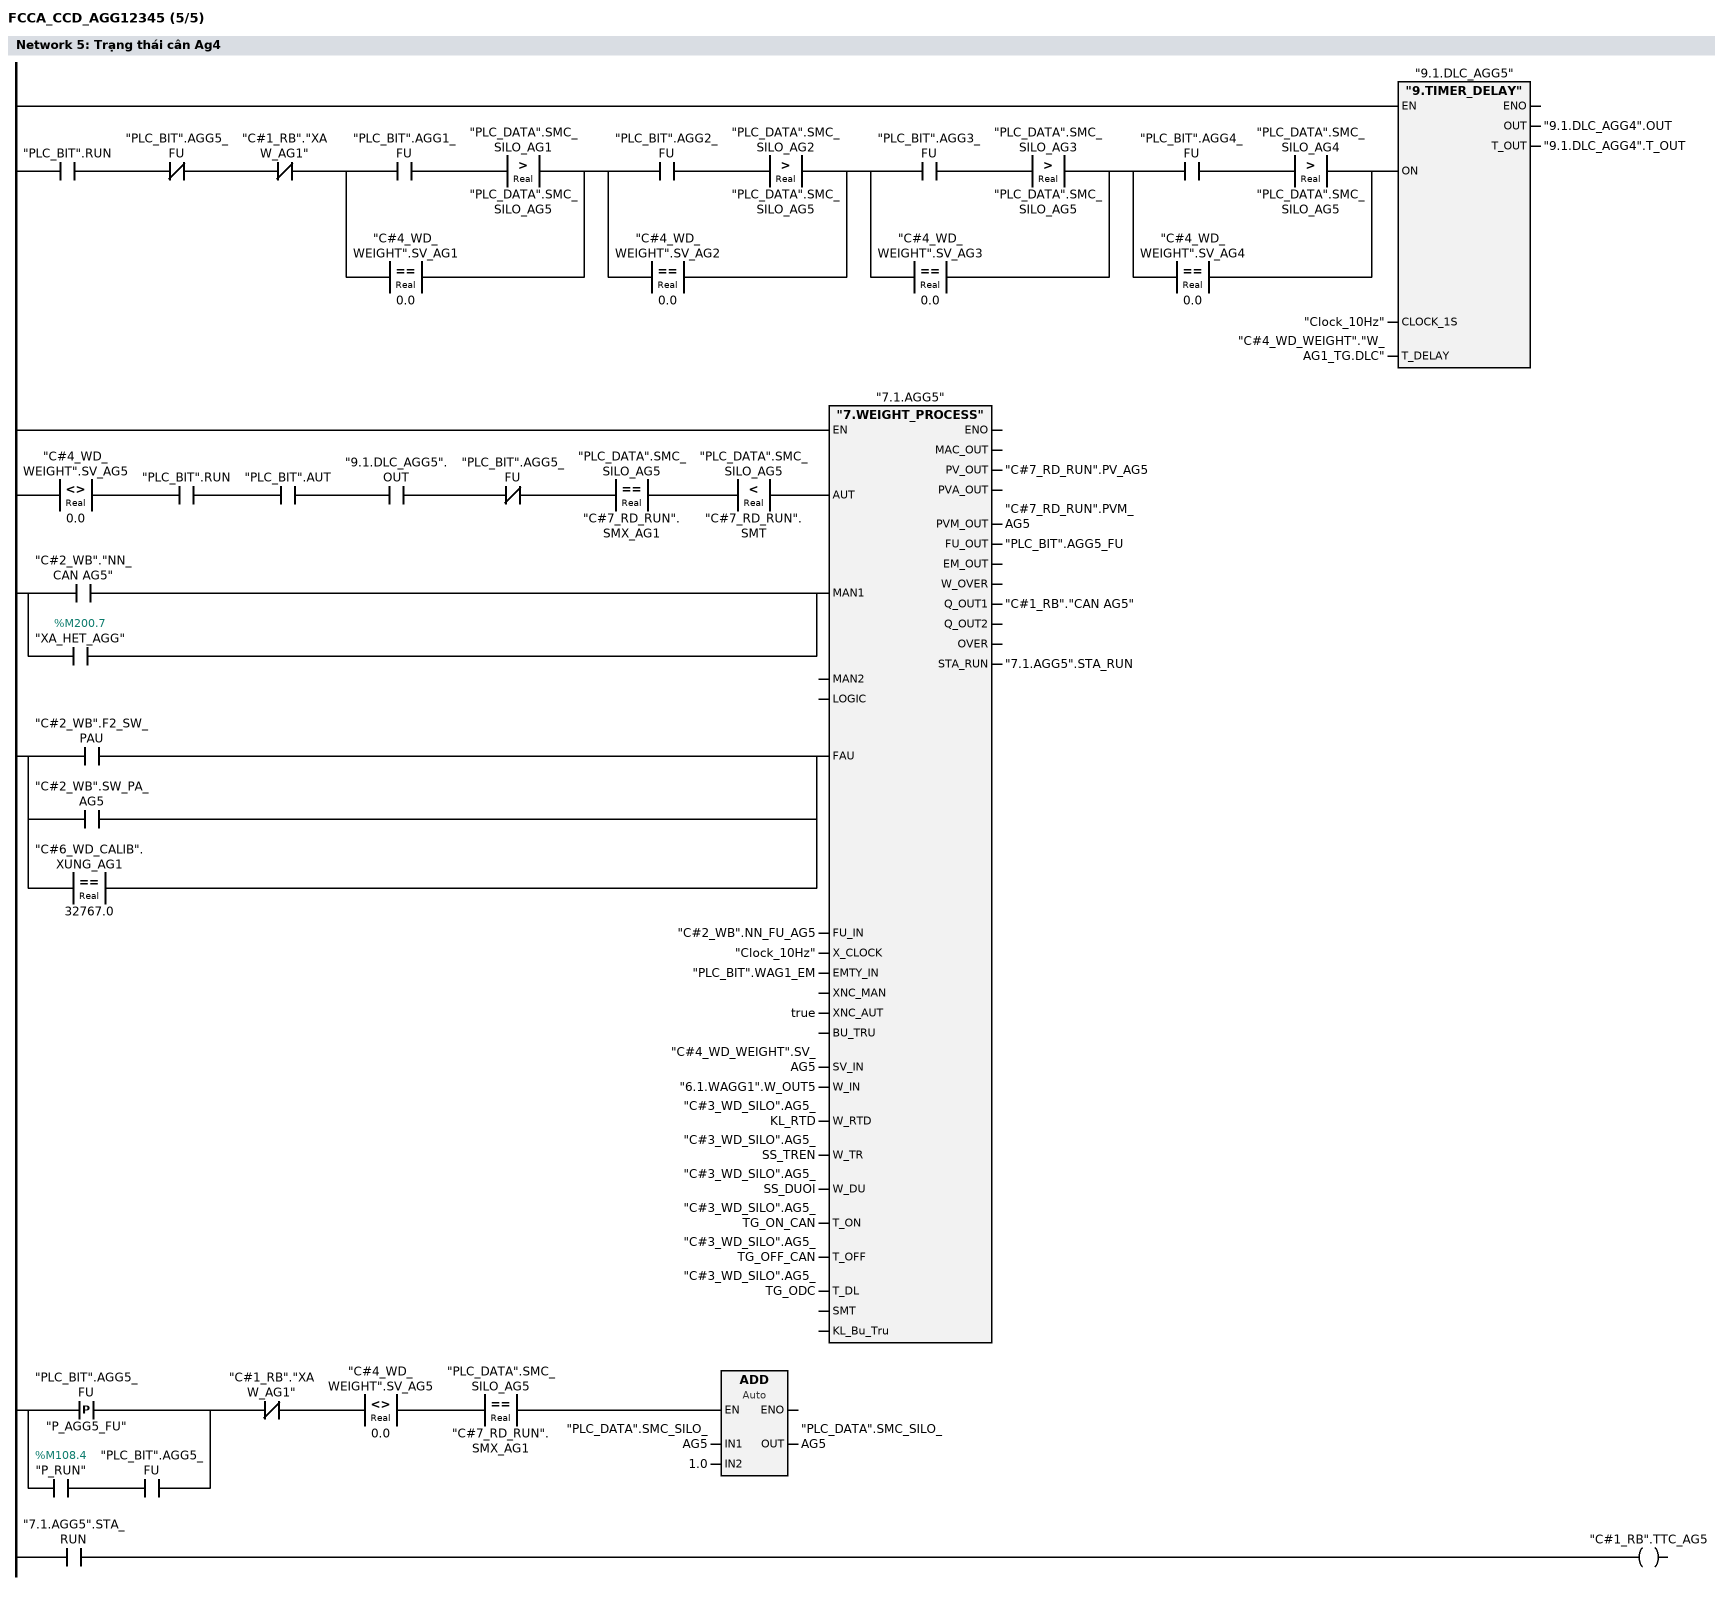
   RUNG wire#powerrail
      "9.1.DLC_AGG5"(ON := wire#w5, CLOCK_1S := "Clock_10Hz", T_DELAY := "C#4_WD_WEIGHT"."W_AG1_TG.DLC", OUT => "9.1.DLC_AGG4".OUT, T_OUT => "9.1.DLC_AGG4".T_OUT)
   END_RUNG
   RUNG wire#powerrail
      Contact( "PLC_BIT".RUN )
      I_Contact( "PLC_BIT".AGG5_FU )
      I_Contact( "C#1_RB"."XA W_AG1" )
      wire#w1
      Contact( "PLC_BIT".AGG1_FU )
      { S7_Templates := "SrcType := Real" } GT_Contact(in1 := "PLC_DATA".SMC_SILO_AG1, in2 := "PLC_DATA".SMC_SILO_AG5)
      wire#w2
      Contact( "PLC_BIT".AGG2_FU )
      { S7_Templates := "SrcType := Real" } GT_Contact(in1 := "PLC_DATA".SMC_SILO_AG2, in2 := "PLC_DATA".SMC_SILO_AG5)
      wire#w3
      Contact( "PLC_BIT".AGG3_FU )
      { S7_Templates := "SrcType := Real" } GT_Contact(in1 := "PLC_DATA".SMC_SILO_AG3, in2 := "PLC_DATA".SMC_SILO_AG5)
      wire#w4
      Contact( "PLC_BIT".AGG4_FU )
      { S7_Templates := "SrcType := Real" } GT_Contact(in1 := "PLC_DATA".SMC_SILO_AG4, in2 := "PLC_DATA".SMC_SILO_AG5)
   END_RUNG wire#w5
   RUNG wire#w1
      { S7_Templates := "SrcType := Real" } EQ_Contact(in1 := "C#4_WD_WEIGHT".SV_AG1, in2 := 0.0)
   END_RUNG wire#w2
   RUNG wire#w2
      { S7_Templates := "SrcType := Real" } EQ_Contact(in1 := "C#4_WD_WEIGHT".SV_AG2, in2 := 0.0)
   END_RUNG wire#w3
   RUNG wire#w3
      { S7_Templates := "SrcType := Real" } EQ_Contact(in1 := "C#4_WD_WEIGHT".SV_AG3, in2 := 0.0)
   END_RUNG wire#w4
   RUNG wire#w4
      { S7_Templates := "SrcType := Real" } EQ_Contact(in1 := "C#4_WD_WEIGHT".SV_AG4, in2 := 0.0)
   END_RUNG wire#w5
   RUNG wire#powerrail
      "7.1.AGG5"(AUT := wire#w6, MAN1 := wire#w7, FAU := wire#w8, MAN2 :=, LOGIC :=, FU_IN := "C#2_WB".NN_FU_AG5, X_CLOCK := "Clock_10Hz", EMTY_IN := "PLC_BIT".WAG1_EM, XNC_MAN :=, XNC_AUT := true, BU_TRU :=, SV_IN := "C#4_WD_WEIGHT".SV_AG5, W_IN := "6.1.WAGG1".W_OUT5, W_RTD := "C#3_WD_SILO".AG5_KL_RTD, W_TR := "C#3_WD_SILO".AG5_SS_TREN, W_DU := "C#3_WD_SILO".AG5_SS_DUOI, T_ON := "C#3_WD_SILO".AG5_TG_ON_CAN, T_OFF := "C#3_WD_SILO".AG5_TG_OFF_CAN, T_DL := "C#3_WD_SILO".AG5_TG_ODC, SMT :=, KL_Bu_Tru :=, MAC_OUT =>, PV_OUT => "C#7_RD_RUN".PV_AG5, PVA_OUT =>, PVM_OUT => "C#7_RD_RUN".PVM_AG5, FU_OUT => "PLC_BIT".AGG5_FU, EM_OUT =>, W_OVER =>, Q_OUT1 => "C#1_RB"."CAN AG5", Q_OUT2 =>, OVER =>, STA_RUN => "7.1.AGG5".STA_RUN)
   END_RUNG
   RUNG wire#powerrail
      { S7_Templates := "SrcType := Real" } NE_Contact(in1 := "C#4_WD_WEIGHT".SV_AG5, in2 := 0.0)
      Contact( "PLC_BIT".RUN )
      Contact( "PLC_BIT".AUT )
      Contact( "9.1.DLC_AGG5".OUT )
      I_Contact( "PLC_BIT".AGG5_FU )
      { S7_Templates := "SrcType := Real" } EQ_Contact(in1 := "PLC_DATA".SMC_SILO_AG5, in2 := "C#7_RD_RUN".SMX_AG1)
      { S7_Templates := "SrcType := Real" } LT_Contact(in1 := "PLC_DATA".SMC_SILO_AG5, in2 := "C#7_RD_RUN".SMT)
   END_RUNG wire#w6
   RUNG wire#powerrail
      Contact( "C#2_WB"."NN_CAN AG5" )
   END_RUNG wire#w7
   RUNG wire#powerrail
      Contact( "XA_HET_AGG" )
   END_RUNG wire#w7
   RUNG wire#powerrail
      Contact( "C#2_WB".F2_SW_PAU )
   END_RUNG wire#w8
   RUNG wire#powerrail
      Contact( "C#2_WB".SW_PA_AG5 )
   END_RUNG wire#w8
   RUNG wire#powerrail
      { S7_Templates := "SrcType := Real" } EQ_Contact(in1 := "C#6_WD_CALIB".XUNG_AG1, in2 := 32767.0)
   END_RUNG wire#w8
   RUNG wire#powerrail
      P_Contact(operand := "PLC_BIT".AGG5_FU, bit := "P_AGG5_FU")
      wire#w9
      I_Contact( "C#1_RB"."XA W_AG1" )
      { S7_Templates := "SrcType := Real" } NE_Contact(in1 := "C#4_WD_WEIGHT".SV_AG5, in2 := 0.0)
      { S7_Templates := "SrcType := Real" } EQ_Contact(in1 := "PLC_DATA".SMC_SILO_AG5, in2 := "C#7_RD_RUN".SMX_AG1)
      Add(in1 := "PLC_DATA".SMC_SILO_AG5, in2 := 1.0, out => "PLC_DATA".SMC_SILO_AG5)
   END_RUNG
   RUNG wire#powerrail
      Contact( "P_RUN" )
      Contact( "PLC_BIT".AGG5_FU )
   END_RUNG wire#w9
   RUNG wire#powerrail
      Contact( "7.1.AGG5".STA_RUN )
      Coil( "C#1_RB".TTC_AG5 )
   END_RUNG
   // the same network as SCL:
   "9.1.DLC_AGG5"(ON := "PLC_BIT".RUN AND NOT "PLC_BIT".AGG5_FU AND NOT "C#1_RB"."XA W_AG1" AND (("PLC_BIT".AGG1_FU AND ("PLC_DATA".SMC_SILO_AG1 > "PLC_DATA".SMC_SILO_AG5)) OR ("C#4_WD_WEIGHT".SV_AG1 = 0.0)) AND (("PLC_BIT".AGG2_FU AND ("PLC_DATA".SMC_SILO_AG2 > "PLC_DATA".SMC_SILO_AG5)) OR ("C#4_WD_WEIGHT".SV_AG2 = 0.0)) AND (("PLC_BIT".AGG3_FU AND ("PLC_DATA".SMC_SILO_AG3 > "PLC_DATA".SMC_SILO_AG5)) OR ("C#4_WD_WEIGHT".SV_AG3 = 0.0)) AND (("PLC_BIT".AGG4_FU AND ("PLC_DATA".SMC_SILO_AG4 > "PLC_DATA".SMC_SILO_AG5)) OR ("C#4_WD_WEIGHT".SV_AG4 = 0.0)),   // "9.TIMER_DELAY"
                  CLOCK_1S := "Clock_10Hz",
                  T_DELAY := "C#4_WD_WEIGHT"."W_AG1_TG.DLC",
                  OUT => "9.1.DLC_AGG4".OUT,
                  T_OUT => "9.1.DLC_AGG4".T_OUT);
   "7.1.AGG5"(AUT := ("C#4_WD_WEIGHT".SV_AG5 <> 0.0) AND "PLC_BIT".RUN AND "PLC_BIT".AUT AND "9.1.DLC_AGG5".OUT AND NOT "PLC_BIT".AGG5_FU AND ("PLC_DATA".SMC_SILO_AG5 = "C#7_RD_RUN".SMX_AG1) AND ("PLC_DATA".SMC_SILO_AG5 < "C#7_RD_RUN".SMT),   // "7.WEIGHT_PROCESS"
              MAN1 := "C#2_WB"."NN_CAN AG5" OR "XA_HET_AGG",
              FAU := "C#2_WB".F2_SW_PAU OR "C#2_WB".SW_PA_AG5 OR ("C#6_WD_CALIB".XUNG_AG1 = 32767.0),
              FU_IN := "C#2_WB".NN_FU_AG5,
              X_CLOCK := "Clock_10Hz",
              EMTY_IN := "PLC_BIT".WAG1_EM,
              XNC_AUT := true,
              SV_IN := "C#4_WD_WEIGHT".SV_AG5,
              W_IN := "6.1.WAGG1".W_OUT5,
              W_RTD := "C#3_WD_SILO".AG5_KL_RTD,
              W_TR := "C#3_WD_SILO".AG5_SS_TREN,
              W_DU := "C#3_WD_SILO".AG5_SS_DUOI,
              T_ON := "C#3_WD_SILO".AG5_TG_ON_CAN,
              T_OFF := "C#3_WD_SILO".AG5_TG_OFF_CAN,
              T_DL := "C#3_WD_SILO".AG5_TG_ODC,
              PV_OUT => "C#7_RD_RUN".PV_AG5,
              PVM_OUT => "C#7_RD_RUN".PVM_AG5,
              FU_OUT => "PLC_BIT".AGG5_FU,
              Q_OUT1 => "C#1_RB"."CAN AG5",
              STA_RUN => "7.1.AGG5".STA_RUN);
   #_w1 := "PLC_BIT".AGG5_FU AND NOT "P_AGG5_FU";   // rising edge of "PLC_BIT".AGG5_FU
   "P_AGG5_FU" := "PLC_BIT".AGG5_FU;
   IF (#_w1 OR ("P_RUN" AND "PLC_BIT".AGG5_FU)) AND NOT "C#1_RB"."XA W_AG1" AND ("C#4_WD_WEIGHT".SV_AG5 <> 0.0) AND ("PLC_DATA".SMC_SILO_AG5 = "C#7_RD_RUN".SMX_AG1) THEN
       "PLC_DATA".SMC_SILO_AG5 := "PLC_DATA".SMC_SILO_AG5 + 1.0;
   END_IF;
   "C#1_RB".TTC_AG5 := "7.1.AGG5".STA_RUN;
END_REGION
END_FUNCTION

FUNCTION_BLOCK "7.WEIGHT_PROCESS"   // FB7, LAD
{ S7_Optimized_Access := 'TRUE' }
VERSION : 0.1
// Chú ý:
// W_DU: nhập khối lượng giớ hạn dưới để tính SS_DUOI sai số dưới, ví dụ SV_IN cài là 1000kg, giới hạn dưới cài là W_DU=55kg, vì KL_BU=0.0 nên> SS_DUOI=1000-55=945kg
// W_RTD: cài đặt khối lượng rơi tự do, từ đó tính điểm cắt Rơi tự do, ví dụ W_RTD=95kg, khi đó điểm cắt Rơi tự do KL_RTD=1000-95=905kg
// Thực tế khi đó: cân sẽ được cân thô đến điểm cắt RTD là 905kg thì nó sẽ bắt đầu chuyển sang Cân Tinh,
// stored: AutoNumber false, CodeModifiedDate 2026-01-15T16:25:50.2794651Z, CompileDate 2026-01-15T16:25:50.5180497Z, CreationDate 2026-01-15T16:22:49.8270549Z, DownloadWithoutReinit false, HandleErrorsWithinBlock false, InterfaceModifiedDate 2024-08-06T09:13:34.3012657Z, IsConsistent true, IsIECCheckEnabled false, IsKnowHowProtected false, IsRetainMemResEnabled false, IsWriteProtected false, LibraryConformanceStatus Warning: The object contains access to global data blocks., MemoryReserve 100, ModifiedDate 2026-01-15T16:25:50.2794651Z, ParameterModified 2024-08-06T08:53:48.4792275Z, PLCSimAdvancedSupport false, SetENOAutomatically False, StructureModified 2024-08-06T09:13:34.3012657Z, UDAEnableTagReadback false
   VAR_INPUT
      AUT : Bool;
      MAN1 : Bool;
      MAN2 : Bool;
      LOGIC : Bool;
      FAU : Bool;   // Tạm dừng cân trong mode Auto
      FU_IN : Bool;   // Nút nhấn báo đầy Silo (phần mềm ghi xuống)
      X_CLOCK : Bool;
      EMTY_IN : Bool;   // Nút nhấn (hoặc tín hiệu trên phần mềm) báo cân rỗng
      XNC_MAN : Bool;
      XNC_AUT : Bool;
      BU_TRU : Bool;   // Nếu =false thì CAN_DƯ luôn bằng 0
      SV_IN : Real;
      W_IN : Real;   // Khối lượng cân hiện tại
      W_RTD : Real;   // Khối lựng rơi tự do
      W_TR : Real;   // KL giới hạn trên
      W_DU : Real;   // KL giới hạn dưới
      T_ON : Real;   // Thời gian cân mở
      T_OFF : Real;   // Thời gian cân đóng
      T_DL : Real;   // Thời gian đợi rơi thêm
      SMT : Real;
      KL_Bu_Tru : Real;   // >0.0 là bù chủ động vào KL_BU, ngược lại sẽ dùng CAN DƯ
   END_VAR
   VAR_OUTPUT
      MAC_OUT : Real;
      PV_OUT : Real;
      PVA_OUT : Real;
      PVM_OUT : Real;
      FU_OUT : Bool;   // Báo cân đầy
      EM_OUT : Bool;
      W_OVER : Real;
      Q_OUT1 : Bool;
      Q_OUT2 : Bool;
      OVER : Bool;
      STA_RUN : Bool;
   END_VAR
   VAR RETAIN
      FU { ExternalAccessible := 'False'; ExternalVisible := 'False'; ExternalWritable := 'False'} : Bool;   // Bít nhớ báo cân đầy
      EM { ExternalAccessible := 'False'; ExternalVisible := 'False'; ExternalWritable := 'False'} : Bool;
      "CAN DU" { ExternalAccessible := 'False'; ExternalVisible := 'False'; ExternalWritable := 'False'} : Real;   // Nếu BU_TRU=false thì CAN_DU luôn =0
      PVA { ExternalAccessible := 'False'; ExternalVisible := 'False'; ExternalWritable := 'False'} : Real;
      PVM { ExternalAccessible := 'False'; ExternalVisible := 'False'; ExternalWritable := 'False'} : Real;
      TOFF { ExternalAccessible := 'False'; ExternalVisible := 'False'; ExternalWritable := 'False'} : Real;
      TON { ExternalAccessible := 'False'; ExternalVisible := 'False'; ExternalWritable := 'False'} : Real;
      T_DLFULL { ExternalAccessible := 'False'; ExternalVisible := 'False'; ExternalWritable := 'False'} : Real;   // Đếm thời gian báo đầy
      "T_DLT/T" { ExternalAccessible := 'False'; ExternalVisible := 'False'; ExternalWritable := 'False'} : Real;   // Đếm thời gian cho lượng rơi thêm
      KL_BU : Real;   // Nhập băng KL_tru_bu hoặc nếu cân bị Cân Dư
      CLK_DLE { ExternalAccessible := 'False'; ExternalVisible := 'False'; ExternalWritable := 'False'} : Bool;
      CLK_DLF { ExternalAccessible := 'False'; ExternalVisible := 'False'; ExternalWritable := 'False'} : Bool;
      "CLK_DLT/T" { ExternalAccessible := 'False'; ExternalVisible := 'False'; ExternalWritable := 'False'} : Bool;
      CLK_TT { ExternalAccessible := 'False'; ExternalVisible := 'False'; ExternalWritable := 'False'} : Bool;
      "TEMP_T/T" { ExternalAccessible := 'False'; ExternalVisible := 'False'; ExternalWritable := 'False'} : Bool;   // Hết thời gian đóng cân ==> mở cân
      "RUN_T/T" { ExternalAccessible := 'False'; ExternalVisible := 'False'; ExternalWritable := 'False'} : Bool;   // Bật chạy thô tinh sau khi hết thời gian đợi rơi thêm
   END_VAR
   VAR
      RUN_MAN : Bool;
      RUN_AUT : Bool;
      "CUA_T/T" : Bool;
      P_OUT1 : Bool;
      P_OUT2 : Bool;
      P_EMTY : Bool;
      P_FU : Bool;
   END_VAR
   VAR_TEMP
      "SS TREN" : Real;
      "SS DUOI" : Real;
      "KL RTD" : Real;   // Điểm cắt Rơi tự do
   END_VAR
   VAR_TEMP   // added for the SCL form of the ladder/FBD networks
      _w1 : Bool;
      _w2 : Bool;
      _w3 : Bool;
   END_VAR
BEGIN

REGION Network 1: MOVE MAC
   // Nếu BU_TRU=false thì CAN_Du luôn bằng 0, khi đó nếu KL_Bu_Tru không được nhập thì KL_BU luôn =0.0
   // Thực tế trong chưng trình này, các điều kiện đang khiến CAN_DU=0.0 và KL_BU=0.0
   // Khi đó SS_DUOI=SV_IN - W_DU
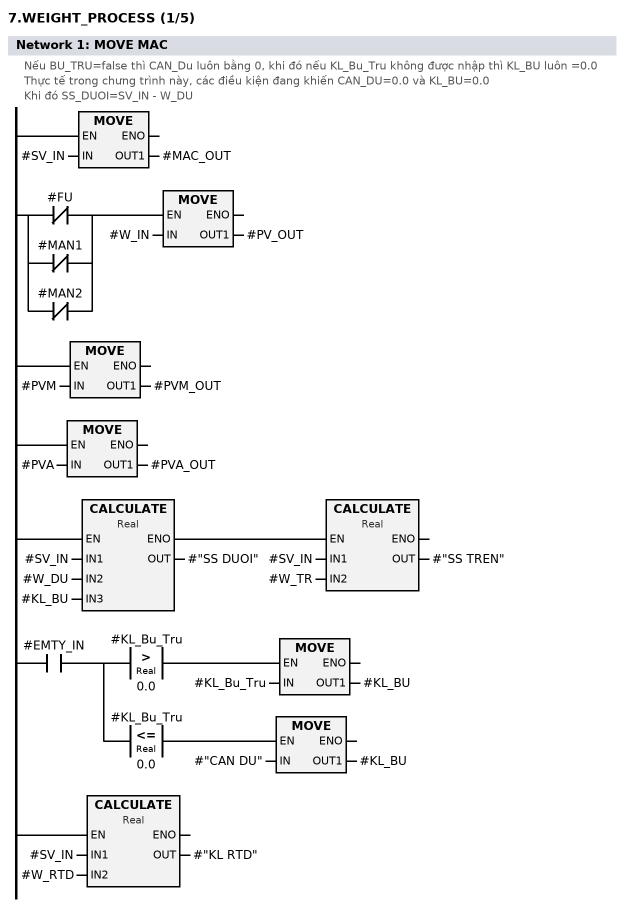
   RUNG wire#powerrail
      Move(in := #SV_IN, out1 => #MAC_OUT)
   END_RUNG
   RUNG wire#powerrail
      I_Contact( #FU )
      wire#w1
      Move(in := #W_IN, out1 => #PV_OUT)
   END_RUNG
   RUNG wire#powerrail
      I_Contact( #MAN1 )
   END_RUNG wire#w1
   RUNG wire#powerrail
      I_Contact( #MAN2 )
   END_RUNG wire#w1
   RUNG wire#powerrail
      Move(in := #PVM, out1 => #PVM_OUT)
   END_RUNG
   RUNG wire#powerrail
      Move(in := #PVA, out1 => #PVA_OUT)
   END_RUNG
   RUNG wire#powerrail
      { S7_Templates := "SrcType := Real"; S7_Expression := "IN1-IN2-IN3" } Calculate(in1 := #SV_IN, in2 := #W_DU, in3 := #KL_BU, out => #"SS DUOI")
      { S7_Templates := "SrcType := Real"; S7_Expression := "IN1+IN2" } Calculate(in1 := #SV_IN, in2 := #W_TR, out => #"SS TREN")
   END_RUNG
   RUNG wire#powerrail
      Contact( #EMTY_IN )
      wire#w2
      { S7_Templates := "SrcType := Real" } GT_Contact(in1 := #KL_Bu_Tru, in2 := 0.0)
      Move(in := #KL_Bu_Tru, out1 => #KL_BU)
   END_RUNG
   RUNG wire#w2
      { S7_Templates := "SrcType := Real" } LE_Contact(in1 := #KL_Bu_Tru, in2 := 0.0)
      Move(in := #"CAN DU", out1 => #KL_BU)
   END_RUNG
   RUNG wire#powerrail
      { S7_Templates := "SrcType := Real"; S7_Expression := "IN1-IN2" } Calculate(in1 := #SV_IN, in2 := #W_RTD, out => #"KL RTD")
   END_RUNG
   // the same network as SCL:
   #MAC_OUT := #SV_IN;
   IF NOT #FU OR NOT #MAN1 OR NOT #MAN2 THEN #PV_OUT := #W_IN; END_IF;
   #PVM_OUT := #PVM;
   #PVA_OUT := #PVA;
   #"SS DUOI" := #SV_IN-#W_DU-#KL_BU;
   #"SS TREN" := #SV_IN+#W_TR;
   IF #EMTY_IN AND (#KL_Bu_Tru > 0.0) THEN #KL_BU := #KL_Bu_Tru; END_IF;
   IF #EMTY_IN AND (#KL_Bu_Tru <= 0.0) THEN #KL_BU := #"CAN DU"; END_IF;
   #"KL RTD" := #SV_IN-#W_RTD;
END_REGION

REGION Network 2: KHOI LUONG CAN DU
   // Tính lượng CAN DƯ, khi cân FU, nếu vì lý do nào đó mà W_IN tiếp tục tăng, túc cân tiếp tục được nạp, thì  giá trị Dư đó xẽ được lưu lại vào biến #CAN DU
   // Báo tràn OVER: trong chế độ AUTO, nếu W_IN lớn hơn SS TRÊN sẽ báo tràn, khi bật FU_OUT thì không kích báo tràn tiếp được
   // Nhưng OVER này được giữ, nó chỉ bị reset khi xả cân, khi đó W_IN nhỏ hơn SS_TREN
   // W_OVER chính là lượng cân dư
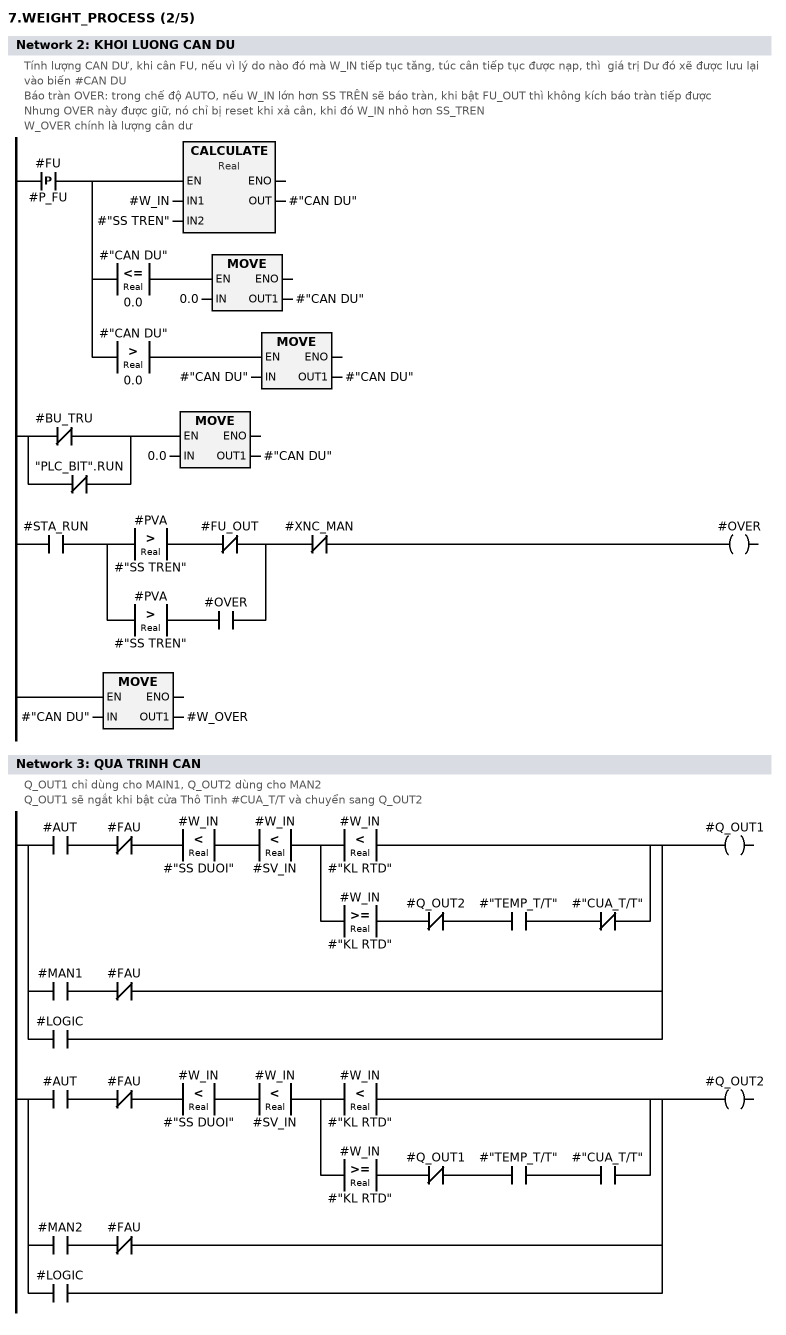
   RUNG wire#powerrail
      P_Contact(operand := #FU, bit := #P_FU)
      wire#w1
      { S7_Templates := "SrcType := Real"; S7_Expression := "IN1-IN2" } Calculate(in1 := #W_IN, in2 := #"SS TREN", out => #"CAN DU")
   END_RUNG
   RUNG wire#w1
      { S7_Templates := "SrcType := Real" } LE_Contact(in1 := #"CAN DU", in2 := 0.0)
      Move(in := 0.0, out1 => #"CAN DU")
   END_RUNG
   RUNG wire#w1
      { S7_Templates := "SrcType := Real" } GT_Contact(in1 := #"CAN DU", in2 := 0.0)
      Move(in := #"CAN DU", out1 => #"CAN DU")
   END_RUNG
   RUNG wire#powerrail
      I_Contact( #BU_TRU )
      wire#w2
      Move(in := 0.0, out1 => #"CAN DU")
   END_RUNG
   RUNG wire#powerrail
      I_Contact( "PLC_BIT".RUN )
   END_RUNG wire#w2
   RUNG wire#powerrail
      Contact( #STA_RUN )
      wire#w3
      { S7_Templates := "SrcType := Real" } GT_Contact(in1 := #PVA, in2 := #"SS TREN")
      I_Contact( #FU_OUT )
      wire#w4
      I_Contact( #XNC_MAN )
      Coil( #OVER )
   END_RUNG
   RUNG wire#w3
      { S7_Templates := "SrcType := Real" } GT_Contact(in1 := #PVA, in2 := #"SS TREN")
      Contact( #OVER )
   END_RUNG wire#w4
   RUNG wire#powerrail
      Move(in := #"CAN DU", out1 => #W_OVER)
   END_RUNG
   // the same network as SCL:
   #_w1 := #FU AND NOT #P_FU;   // rising edge of #FU
   #P_FU := #FU;
   IF #_w1 THEN #"CAN DU" := #W_IN-#"SS TREN"; END_IF;
   IF #_w1 AND (#"CAN DU" <= 0.0) THEN #"CAN DU" := 0.0; END_IF;
   IF #_w1 AND (#"CAN DU" > 0.0) THEN #"CAN DU" := #"CAN DU"; END_IF;
   IF NOT #BU_TRU OR NOT "PLC_BIT".RUN THEN #"CAN DU" := 0.0; END_IF;
   #OVER := #STA_RUN AND (((#PVA > #"SS TREN") AND NOT #FU_OUT) OR ((#PVA > #"SS TREN") AND #OVER)) AND NOT #XNC_MAN;
   #W_OVER := #"CAN DU";
END_REGION

REGION Network 3: QUA TRINH CAN
   // Q_OUT1 chỉ dùng cho MAIN1, Q_OUT2 dùng cho MAN2
   // Q_OUT1 sẽ ngắt khi bật cửa Thô Tinh #CUA_T/T và chuyển sang Q_OUT2
   RUNG wire#powerrail
      Contact( #AUT )
      I_Contact( #FAU )
      { S7_Templates := "SrcType := Real" } LT_Contact(in1 := #W_IN, in2 := #"SS DUOI")
      { S7_Templates := "SrcType := Real" } LT_Contact(in1 := #W_IN, in2 := #SV_IN)
      wire#w1
      { S7_Templates := "SrcType := Real" } LT_Contact(in1 := #W_IN, in2 := #"KL RTD")
      wire#w2
      Coil( #Q_OUT1 )
   END_RUNG
   RUNG wire#w1
      { S7_Templates := "SrcType := Real" } GE_Contact(in1 := #W_IN, in2 := #"KL RTD")
      I_Contact( #Q_OUT2 )
      Contact( #"TEMP_T/T" )
      I_Contact( #"CUA_T/T" )
   END_RUNG wire#w2
   RUNG wire#powerrail
      Contact( #MAN1 )
      I_Contact( #FAU )
   END_RUNG wire#w2
   RUNG wire#powerrail
      Contact( #LOGIC )
   END_RUNG wire#w2
   RUNG wire#powerrail
      Contact( #AUT )
      I_Contact( #FAU )
      { S7_Templates := "SrcType := Real" } LT_Contact(in1 := #W_IN, in2 := #"SS DUOI")
      { S7_Templates := "SrcType := Real" } LT_Contact(in1 := #W_IN, in2 := #SV_IN)
      wire#w3
      { S7_Templates := "SrcType := Real" } LT_Contact(in1 := #W_IN, in2 := #"KL RTD")
      wire#w4
      Coil( #Q_OUT2 )
   END_RUNG
   RUNG wire#w3
      { S7_Templates := "SrcType := Real" } GE_Contact(in1 := #W_IN, in2 := #"KL RTD")
      I_Contact( #Q_OUT1 )
      Contact( #"TEMP_T/T" )
      Contact( #"CUA_T/T" )
   END_RUNG wire#w4
   RUNG wire#powerrail
      Contact( #MAN2 )
      I_Contact( #FAU )
   END_RUNG wire#w4
   RUNG wire#powerrail
      Contact( #LOGIC )
   END_RUNG wire#w4
   // the same network as SCL:
   #Q_OUT1 := (#AUT AND NOT #FAU AND (#W_IN < #"SS DUOI") AND (#W_IN < #SV_IN) AND ((#W_IN < #"KL RTD") OR ((#W_IN >= #"KL RTD") AND NOT #Q_OUT2 AND #"TEMP_T/T" AND NOT #"CUA_T/T"))) OR (#MAN1 AND NOT #FAU) OR #LOGIC;
   #Q_OUT2 := (#AUT AND NOT #FAU AND (#W_IN < #"SS DUOI") AND (#W_IN < #SV_IN) AND ((#W_IN < #"KL RTD") OR ((#W_IN >= #"KL RTD") AND NOT #Q_OUT1 AND #"TEMP_T/T" AND #"CUA_T/T"))) OR (#MAN2 AND NOT #FAU) OR #LOGIC;
END_REGION

REGION Network 4: CHIA PV
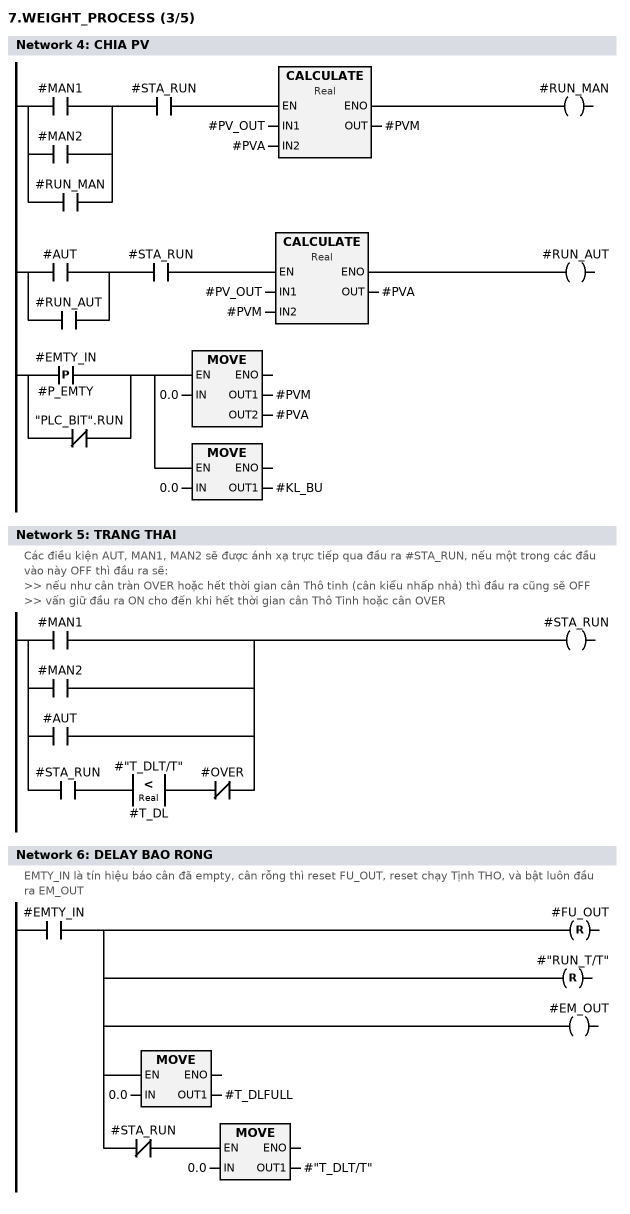
   RUNG wire#powerrail
      Contact( #MAN1 )
      wire#w1
      Contact( #STA_RUN )
      { S7_Templates := "SrcType := Real"; S7_Expression := "IN1-IN2" } Calculate(in1 := #PV_OUT, in2 := #PVA, out => #PVM)
      Coil( #RUN_MAN )
   END_RUNG
   RUNG wire#powerrail
      Contact( #MAN2 )
   END_RUNG wire#w1
   RUNG wire#powerrail
      Contact( #RUN_MAN )
   END_RUNG wire#w1
   RUNG wire#powerrail
      Contact( #AUT )
      wire#w2
      Contact( #STA_RUN )
      { S7_Templates := "SrcType := Real"; S7_Expression := "IN1-IN2" } Calculate(in1 := #PV_OUT, in2 := #PVM, out => #PVA)
      Coil( #RUN_AUT )
   END_RUNG
   RUNG wire#powerrail
      Contact( #RUN_AUT )
   END_RUNG wire#w2
   RUNG wire#powerrail
      P_Contact(operand := #EMTY_IN, bit := #P_EMTY)
      wire#w3
      Move(in := 0.0, out1 => #PVM, out2 => #PVA)
   END_RUNG
   RUNG wire#powerrail
      I_Contact( "PLC_BIT".RUN )
   END_RUNG wire#w3
   RUNG wire#w3
      Move(in := 0.0, out1 => #KL_BU)
   END_RUNG
   // the same network as SCL:
   #_w1 := (#MAN1 OR #MAN2 OR #RUN_MAN) AND #STA_RUN;
   IF #_w1 THEN #PVM := #PV_OUT-#PVA; END_IF;
   #RUN_MAN := #_w1;
   #_w2 := (#AUT OR #RUN_AUT) AND #STA_RUN;
   IF #_w2 THEN #PVA := #PV_OUT-#PVM; END_IF;
   #RUN_AUT := #_w2;
   #_w3 := #EMTY_IN AND NOT #P_EMTY;   // rising edge of #EMTY_IN
   #P_EMTY := #EMTY_IN;
   IF #_w3 OR NOT "PLC_BIT".RUN THEN
       #PVM := 0.0;
       #PVA := 0.0;
       #KL_BU := 0.0;
   END_IF;
END_REGION

REGION Network 5: TRANG THAI
   // Các điều kiện AUT, MAN1, MAN2 sẽ được ánh xạ trực tiếp qua đầu ra #STA_RUN, nếu một trong các đầu vào này OFF thì đầu ra sẽ:
   // >> nếu như cân tràn OVER hoặc hết thời gian cân Thô tinh (cân kiểu nhấp nhả) thì đầu ra cũng sẽ OFF
   // >> vấn giữ đầu ra ON cho đến khi hết thời gian cân Thô Tinh hoặc cân OVER
   RUNG wire#powerrail
      Contact( #MAN1 )
      wire#w1
      Coil( #STA_RUN )
   END_RUNG
   RUNG wire#powerrail
      Contact( #MAN2 )
   END_RUNG wire#w1
   RUNG wire#powerrail
      Contact( #AUT )
   END_RUNG wire#w1
   RUNG wire#powerrail
      Contact( #STA_RUN )
      { S7_Templates := "SrcType := Real" } LT_Contact(in1 := #"T_DLT/T", in2 := #T_DL)
      I_Contact( #OVER )
   END_RUNG wire#w1
   // the same network as SCL:
   #STA_RUN := #MAN1 OR #MAN2 OR #AUT OR (#STA_RUN AND (#"T_DLT/T" < #T_DL) AND NOT #OVER);
END_REGION

REGION Network 6: DELAY BAO RONG
   // EMTY_IN là tín hiệu báo cân đã empty, cân rỗng thì reset FU_OUT, reset chạy Tịnh THO, và bật luôn đầu ra EM_OUT
   RUNG wire#powerrail
      Contact( #EMTY_IN )
      wire#w1
      R_Coil( #FU_OUT )
   END_RUNG
   RUNG wire#w1
      R_Coil( #"RUN_T/T" )
   END_RUNG
   RUNG wire#w1
      Coil( #EM_OUT )
   END_RUNG
   RUNG wire#w1
      Move(in := 0.0, out1 => #T_DLFULL)
   END_RUNG
   RUNG wire#w1
      I_Contact( #STA_RUN )
      Move(in := 0.0, out1 => #"T_DLT/T")
   END_RUNG
   // the same network as SCL:
   IF #EMTY_IN THEN
       #FU_OUT := FALSE;
       #"RUN_T/T" := FALSE;
   END_IF;
   #EM_OUT := #EMTY_IN;
   IF #EMTY_IN THEN #T_DLFULL := 0.0; END_IF;
   IF #EMTY_IN AND NOT #STA_RUN THEN #"T_DLT/T" := 0.0; END_IF;
END_REGION

REGION Network 7: DELAY BAO DAY
   // Khi khối lượng đầu vào vượt qua sai số dưới, thì bắt đầu đếm để tình thời gian Delay trước khi báo FU
   // nếu thời gian đếm nó vượt qua giá trị cài đặt (cũng chính là thời gian đợi chơ lượng rơi thêm), thì SET ngõ ra #FU_OUT
   // 
   // Chú ý: chế độ MAN thì nó không báo FU
   // Cân FULL khi giá trị cân nó vượt qua SS_DUOI rồi đợi thêm một khoảng thời gian rơi thêm
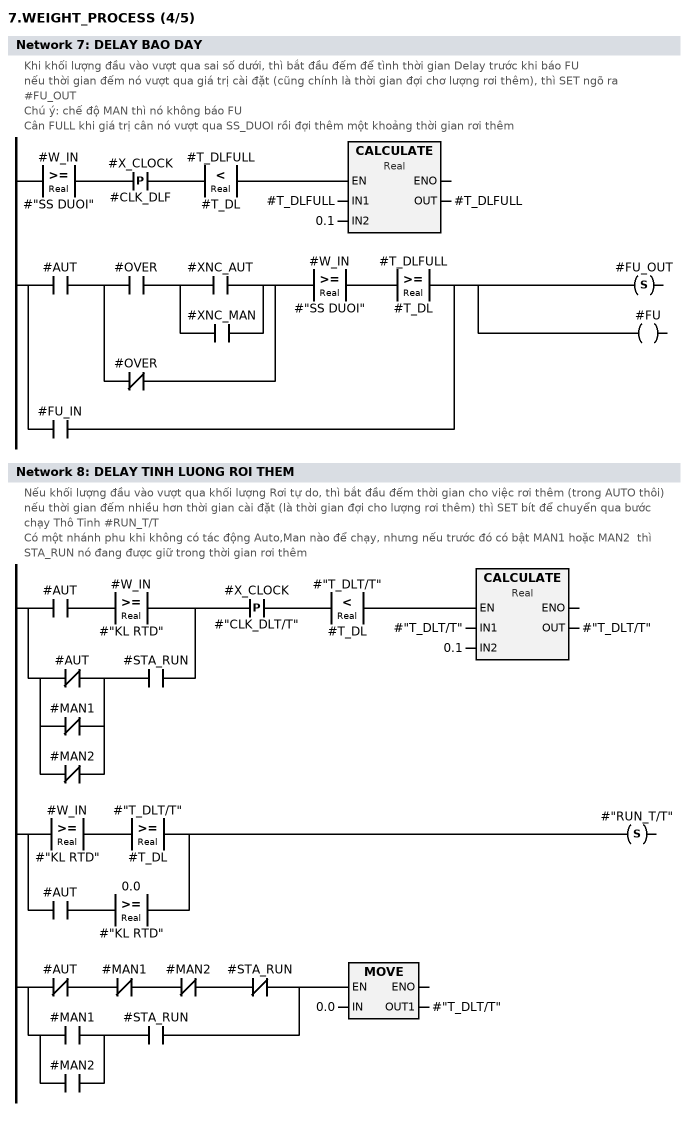
   RUNG wire#powerrail
      { S7_Templates := "SrcType := Real" } GE_Contact(in1 := #W_IN, in2 := #"SS DUOI")
      P_Contact(operand := #X_CLOCK, bit := #CLK_DLF)
      { S7_Templates := "SrcType := Real" } LT_Contact(in1 := #T_DLFULL, in2 := #T_DL)
      { S7_Templates := "SrcType := Real"; S7_Expression := "IN1+IN2" } Calculate(in1 := #T_DLFULL, in2 := 0.1, out => #T_DLFULL)
   END_RUNG
   RUNG wire#powerrail
      Contact( #AUT )
      wire#w1
      Contact( #OVER )
      wire#w2
      Contact( #XNC_AUT )
      wire#w3
      { S7_Templates := "SrcType := Real" } GE_Contact(in1 := #W_IN, in2 := #"SS DUOI")
      { S7_Templates := "SrcType := Real" } GE_Contact(in1 := #T_DLFULL, in2 := #T_DL)
      wire#w4
      S_Coil( #FU_OUT )
   END_RUNG
   RUNG wire#w2
      Contact( #XNC_MAN )
   END_RUNG wire#w3
   RUNG wire#w1
      I_Contact( #OVER )
   END_RUNG wire#w3
   RUNG wire#powerrail
      Contact( #FU_IN )
   END_RUNG wire#w4
   RUNG wire#w4
      Coil( #FU )
   END_RUNG
   // the same network as SCL:
   #_w1 := (#W_IN >= #"SS DUOI") AND #X_CLOCK AND NOT #CLK_DLF;   // rising edge of #X_CLOCK
   #CLK_DLF := #X_CLOCK;
   IF #_w1 AND (#T_DLFULL < #T_DL) THEN #T_DLFULL := #T_DLFULL+0.1; END_IF;
   #_w2 := (#AUT AND ((#OVER AND (#XNC_AUT OR #XNC_MAN)) OR NOT #OVER) AND (#W_IN >= #"SS DUOI") AND (#T_DLFULL >= #T_DL)) OR #FU_IN;
   IF #_w2 THEN #FU_OUT := TRUE; END_IF;
   #FU := #_w2;
END_REGION

REGION Network 8: DELAY TINH LUONG ROI THEM
   // Nếu khối lượng đầu vào vượt qua khối lượng Rơi tự do, thì bắt đầu đếm thời gian cho việc rơi thêm (trong AUTO thôi)
   // nếu thời gian đếm nhiều hơn thời gian cài đặt (là thời gian đợi cho lượng rơi thêm) thì SET bít để chuyển qua bước chạy Thô Tinh #RUN_T/T
   // 
   // Có một nhánh phu khi không có tác động Auto,Man nào để chạy, nhưng nếu trước đó có bật MAN1 hoặc MAN2  thì STA_RUN nó đang được giữ trong thời gian rơi thêm
   RUNG wire#powerrail
      Contact( #AUT )
      { S7_Templates := "SrcType := Real" } GE_Contact(in1 := #W_IN, in2 := #"KL RTD")
      wire#w1
      P_Contact(operand := #X_CLOCK, bit := #"CLK_DLT/T")
      { S7_Templates := "SrcType := Real" } LT_Contact(in1 := #"T_DLT/T", in2 := #T_DL)
      { S7_Templates := "SrcType := Real"; S7_Expression := "IN1+IN2" } Calculate(in1 := #"T_DLT/T", in2 := 0.1, out => #"T_DLT/T")
   END_RUNG
   RUNG wire#powerrail
      I_Contact( #AUT )
      wire#w2
      Contact( #STA_RUN )
   END_RUNG wire#w1
   RUNG wire#powerrail
      I_Contact( #MAN1 )
   END_RUNG wire#w2
   RUNG wire#powerrail
      I_Contact( #MAN2 )
   END_RUNG wire#w2
   RUNG wire#powerrail
      { S7_Templates := "SrcType := Real" } GE_Contact(in1 := #W_IN, in2 := #"KL RTD")
      { S7_Templates := "SrcType := Real" } GE_Contact(in1 := #"T_DLT/T", in2 := #T_DL)
      wire#w3
      S_Coil( #"RUN_T/T" )
   END_RUNG
   RUNG wire#powerrail
      Contact( #AUT )
      { S7_Templates := "SrcType := Real" } GE_Contact(in1 := 0.0, in2 := #"KL RTD")
   END_RUNG wire#w3
   RUNG wire#powerrail
      I_Contact( #AUT )
      I_Contact( #MAN1 )
      I_Contact( #MAN2 )
      I_Contact( #STA_RUN )
      wire#w4
      Move(in := 0.0, out1 => #"T_DLT/T")
   END_RUNG
   RUNG wire#powerrail
      Contact( #MAN1 )
      wire#w5
      Contact( #STA_RUN )
   END_RUNG wire#w4
   RUNG wire#powerrail
      Contact( #MAN2 )
   END_RUNG wire#w5
   // the same network as SCL:
   #_w1 := ((#AUT AND (#W_IN >= #"KL RTD")) OR ((NOT #AUT OR NOT #MAN1 OR NOT #MAN2) AND #STA_RUN)) AND #X_CLOCK AND NOT #"CLK_DLT/T";   // rising edge of #X_CLOCK
   #"CLK_DLT/T" := #X_CLOCK;
   IF #_w1 AND (#"T_DLT/T" < #T_DL) THEN #"T_DLT/T" := #"T_DLT/T"+0.1; END_IF;
   IF ((#W_IN >= #"KL RTD") AND (#"T_DLT/T" >= #T_DL)) OR (#AUT AND (0.0 >= #"KL RTD")) THEN
       #"RUN_T/T" := TRUE;
   END_IF;
   IF (NOT #AUT AND NOT #MAN1 AND NOT #MAN2 AND NOT #STA_RUN) OR ((#MAN1 OR #MAN2) AND #STA_RUN) THEN
       #"T_DLT/T" := 0.0;
   END_IF;
END_REGION

REGION Network 9: CAN THO TINH
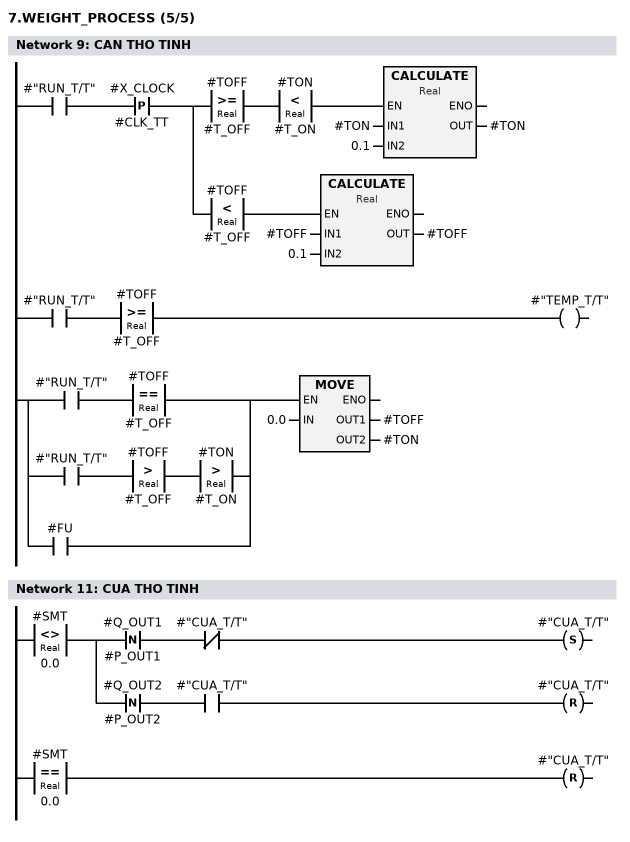
   RUNG wire#powerrail
      Contact( #"RUN_T/T" )
      P_Contact(operand := #X_CLOCK, bit := #CLK_TT)
      wire#w1
      { S7_Templates := "SrcType := Real" } GE_Contact(in1 := #TOFF, in2 := #T_OFF)
      { S7_Templates := "SrcType := Real" } LT_Contact(in1 := #TON, in2 := #T_ON)
      { S7_Templates := "SrcType := Real"; S7_Expression := "IN1+IN2" } Calculate(in1 := #TON, in2 := 0.1, out => #TON)
   END_RUNG
   RUNG wire#w1
      { S7_Templates := "SrcType := Real" } LT_Contact(in1 := #TOFF, in2 := #T_OFF)
      { S7_Templates := "SrcType := Real"; S7_Expression := "IN1+IN2" } Calculate(in1 := #TOFF, in2 := 0.1, out => #TOFF)
   END_RUNG
   RUNG wire#powerrail
      Contact( #"RUN_T/T" )
      { S7_Templates := "SrcType := Real" } GE_Contact(in1 := #TOFF, in2 := #T_OFF)
      Coil( #"TEMP_T/T" )
   END_RUNG
   RUNG wire#powerrail
      Contact( #"RUN_T/T" )
      { S7_Templates := "SrcType := Real" } EQ_Contact(in1 := #TOFF, in2 := #T_OFF)
      wire#w2
      Move(in := 0.0, out1 => #TOFF, out2 => #TON)
   END_RUNG
   RUNG wire#powerrail
      Contact( #"RUN_T/T" )
      { S7_Templates := "SrcType := Real" } GT_Contact(in1 := #TOFF, in2 := #T_OFF)
      { S7_Templates := "SrcType := Real" } GT_Contact(in1 := #TON, in2 := #T_ON)
   END_RUNG wire#w2
   RUNG wire#powerrail
      Contact( #FU )
   END_RUNG wire#w2
   // the same network as SCL:
   #_w1 := #"RUN_T/T" AND #X_CLOCK AND NOT #CLK_TT;   // rising edge of #X_CLOCK
   #CLK_TT := #X_CLOCK;
   IF #_w1 AND (#TOFF >= #T_OFF) AND (#TON < #T_ON) THEN #TON := #TON+0.1; END_IF;
   IF #_w1 AND (#TOFF < #T_OFF) THEN #TOFF := #TOFF+0.1; END_IF;
   #"TEMP_T/T" := #"RUN_T/T" AND (#TOFF >= #T_OFF);
   IF (#"RUN_T/T" AND (#TOFF = #T_OFF)) OR (#"RUN_T/T" AND (#TOFF > #T_OFF) AND (#TON > #T_ON)) OR #FU THEN
       #TOFF := 0.0;
       #TON := 0.0;
   END_IF;
END_REGION

REGION Network 10: CAN LOGIC
END_REGION

REGION Network 11: CUA THO TINH
   RUNG wire#powerrail
      { S7_Templates := "SrcType := Real" } NE_Contact(in1 := #SMT, in2 := 0.0)
      wire#w1
      N_Contact(operand := #Q_OUT1, bit := #P_OUT1)
      I_Contact( #"CUA_T/T" )
      S_Coil( #"CUA_T/T" )
   END_RUNG
   RUNG wire#w1
      N_Contact(operand := #Q_OUT2, bit := #P_OUT2)
      Contact( #"CUA_T/T" )
      R_Coil( #"CUA_T/T" )
   END_RUNG
   RUNG wire#powerrail
      { S7_Templates := "SrcType := Real" } EQ_Contact(in1 := #SMT, in2 := 0.0)
      R_Coil( #"CUA_T/T" )
   END_RUNG
   // the same network as SCL:
   #_w1 := #SMT <> 0.0;
   #_w2 := #_w1 AND NOT #Q_OUT1 AND #P_OUT1;   // falling edge of #Q_OUT1
   #P_OUT1 := #Q_OUT1;
   IF #_w2 AND NOT #"CUA_T/T" THEN #"CUA_T/T" := TRUE; END_IF;
   #_w3 := #_w1 AND NOT #Q_OUT2 AND #P_OUT2;   // falling edge of #Q_OUT2
   #P_OUT2 := #Q_OUT2;
   IF #_w3 AND #"CUA_T/T" THEN #"CUA_T/T" := FALSE; END_IF;
   IF #SMT = 0.0 THEN #"CUA_T/T" := FALSE; END_IF;
END_REGION
END_FUNCTION_BLOCK

FUNCTION "FCXL_IND_AGG1" : Void   // FC6, LAD
{ S7_Optimized_Access := 'TRUE' }
VERSION : 0.1
// stored: AutoNumber true, CodeModifiedDate 2026-01-15T16:25:53.86748Z, CompileDate 2026-01-15T16:25:53.9093246Z, CreationDate 2026-01-15T16:24:02.4619467Z, HandleErrorsWithinBlock false, InterfaceModifiedDate 2026-01-10T11:03:05.6285532Z, IsConsistent true, IsIECCheckEnabled false, IsKnowHowProtected false, IsWriteProtected false, LibraryConformanceStatus Error: The block contains calls of single instances. Warning: The object contains access to global data blocks. Warning: The block contains direct access to inputs, outputs, bit memories, indirect access to the registry or indirect access to external memory areas that are unknown at the time of compilation., ModifiedDate 2026-01-15T16:25:53.86748Z, ParameterModified 2026-01-10T11:03:05.6285532Z, PLCSimAdvancedSupport false, SetENOAutomatically False, StructureModified 2026-01-10T11:03:05.6285532Z, UDAEnableTagReadback false
   VAR_TEMP   // added for the SCL form of the ladder/FBD networks
      _w1 : Bool;
      _w2 : Bool;
      _w3 : Bool;
   END_VAR
BEGIN

REGION Network 1: Cân độc lập AGG1 Full
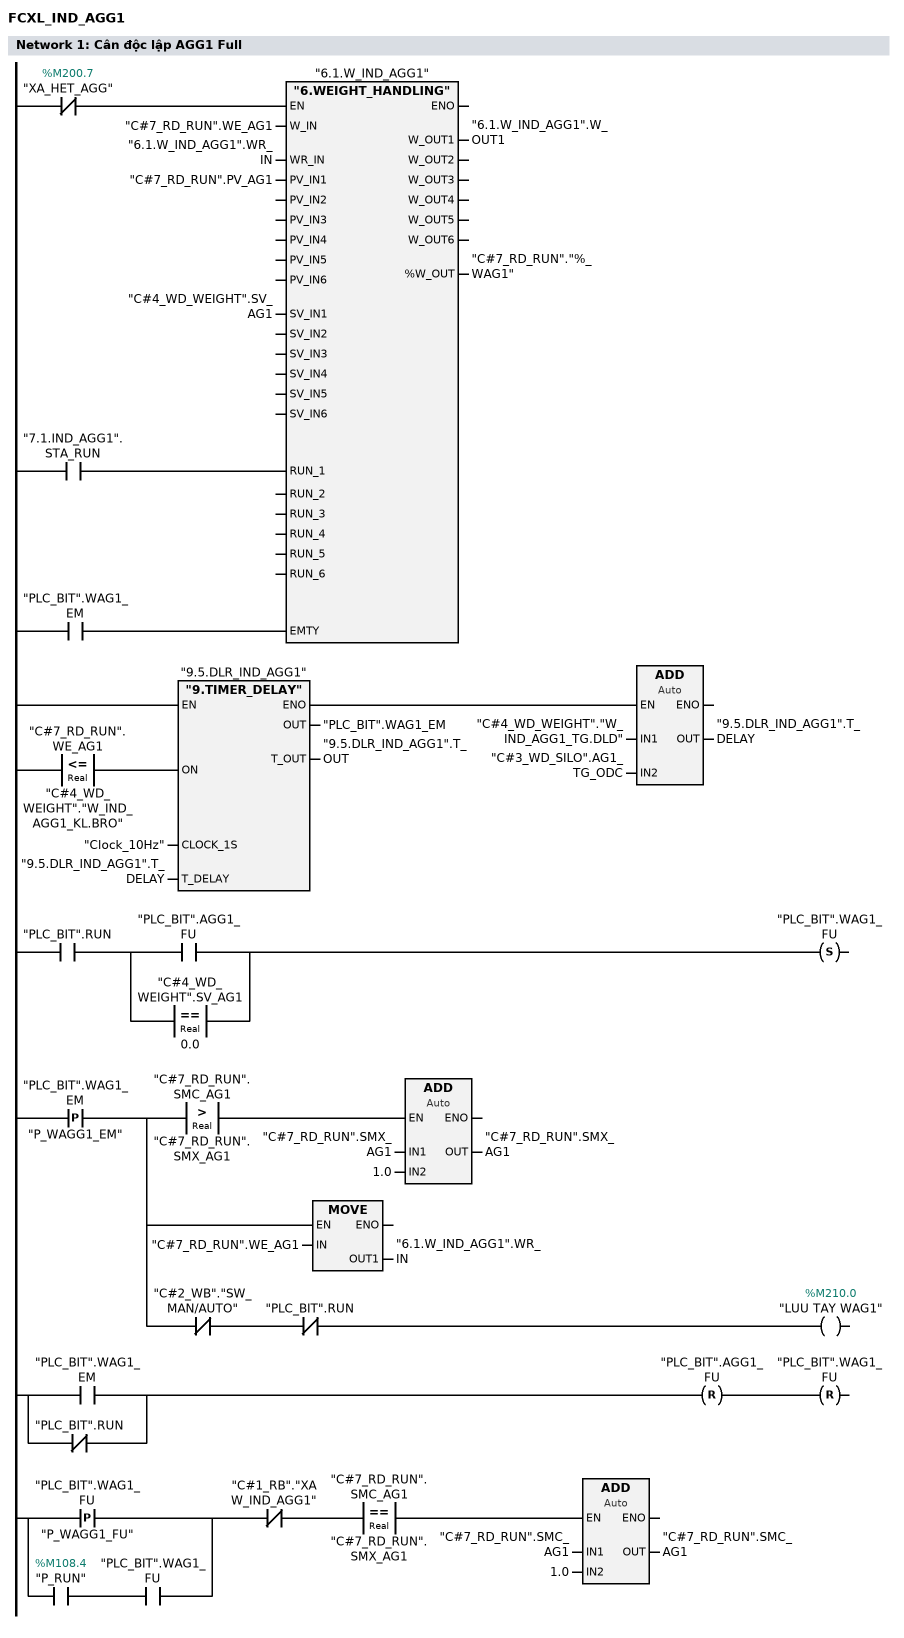
   RUNG wire#powerrail
      I_Contact( "XA_HET_AGG" )
      "6.1.W_IND_AGG1"(RUN_1 := wire#w1, EMTY := wire#w2, W_IN := "C#7_RD_RUN".WE_AG1, WR_IN := "6.1.W_IND_AGG1".WR_IN, PV_IN1 := "C#7_RD_RUN".PV_AG1, PV_IN2 :=, PV_IN3 :=, PV_IN4 :=, PV_IN5 :=, PV_IN6 :=, SV_IN1 := "C#4_WD_WEIGHT".SV_AG1, SV_IN2 :=, SV_IN3 :=, SV_IN4 :=, SV_IN5 :=, SV_IN6 :=, RUN_2 :=, RUN_3 :=, RUN_4 :=, RUN_5 :=, RUN_6 :=, W_OUT1 => "6.1.W_IND_AGG1".W_OUT1, W_OUT2 =>, W_OUT3 =>, W_OUT4 =>, W_OUT5 =>, W_OUT6 =>, "%W_OUT" => "C#7_RD_RUN"."%_WAG1")
   END_RUNG
   RUNG wire#powerrail
      Contact( "7.1.IND_AGG1".STA_RUN )
   END_RUNG wire#w1
   RUNG wire#powerrail
      Contact( "PLC_BIT".WAG1_EM )
   END_RUNG wire#w2
   RUNG wire#powerrail
      "9.5.DLR_IND_AGG1"(ON := wire#w3, CLOCK_1S := "Clock_10Hz", T_DELAY := "9.5.DLR_IND_AGG1".T_DELAY, OUT => "PLC_BIT".WAG1_EM, T_OUT => "9.5.DLR_IND_AGG1".T_OUT)
      Add(in1 := "C#4_WD_WEIGHT"."W_IND_AGG1_TG.DLD", in2 := "C#3_WD_SILO".AG1_TG_ODC, out => "9.5.DLR_IND_AGG1".T_DELAY)
   END_RUNG
   RUNG wire#powerrail
      { S7_Templates := "SrcType := Real" } LE_Contact(in1 := "C#7_RD_RUN".WE_AG1, in2 := "C#4_WD_WEIGHT"."W_IND_AGG1_KL.BRO")
   END_RUNG wire#w3
   RUNG wire#powerrail
      Contact( "PLC_BIT".RUN )
      wire#w4
      Contact( "PLC_BIT".AGG1_FU )
      wire#w5
      S_Coil( "PLC_BIT".WAG1_FU )
   END_RUNG
   RUNG wire#w4
      { S7_Templates := "SrcType := Real" } EQ_Contact(in1 := "C#4_WD_WEIGHT".SV_AG1, in2 := 0.0)
   END_RUNG wire#w5
   RUNG wire#powerrail
      P_Contact(operand := "PLC_BIT".WAG1_EM, bit := "P_WAGG1_EM")
      wire#w6
      { S7_Templates := "SrcType := Real" } GT_Contact(in1 := "C#7_RD_RUN".SMC_AG1, in2 := "C#7_RD_RUN".SMX_AG1)
      Add(in1 := "C#7_RD_RUN".SMX_AG1, in2 := 1.0, out => "C#7_RD_RUN".SMX_AG1)
   END_RUNG
   RUNG wire#w6
      Move(in := "C#7_RD_RUN".WE_AG1, out1 => "6.1.W_IND_AGG1".WR_IN)
   END_RUNG
   RUNG wire#w6
      I_Contact( "C#2_WB"."SW_MAN/AUTO" )
      I_Contact( "PLC_BIT".RUN )
      Coil( "LUU TAY WAG1" )
   END_RUNG
   RUNG wire#powerrail
      Contact( "PLC_BIT".WAG1_EM )
      wire#w7
      R_Coil( "PLC_BIT".AGG1_FU )
      R_Coil( "PLC_BIT".WAG1_FU )
   END_RUNG
   RUNG wire#powerrail
      I_Contact( "PLC_BIT".RUN )
   END_RUNG wire#w7
   RUNG wire#powerrail
      P_Contact(operand := "PLC_BIT".WAG1_FU, bit := "P_WAGG1_FU")
      wire#w8
      I_Contact( "C#1_RB"."XA W_IND_AGG1" )
      { S7_Templates := "SrcType := Real" } EQ_Contact(in1 := "C#7_RD_RUN".SMC_AG1, in2 := "C#7_RD_RUN".SMX_AG1)
      Add(in1 := "C#7_RD_RUN".SMC_AG1, in2 := 1.0, out => "C#7_RD_RUN".SMC_AG1)
   END_RUNG
   RUNG wire#powerrail
      Contact( "P_RUN" )
      Contact( "PLC_BIT".WAG1_FU )
   END_RUNG wire#w8
   // the same network as SCL:
   IF NOT "XA_HET_AGG" THEN
       "6.1.W_IND_AGG1"(W_IN := "C#7_RD_RUN".WE_AG1,   // "6.WEIGHT_HANDLING"
                        WR_IN := "6.1.W_IND_AGG1".WR_IN,
                        PV_IN1 := "C#7_RD_RUN".PV_AG1,
                        SV_IN1 := "C#4_WD_WEIGHT".SV_AG1,
                        RUN_1 := "7.1.IND_AGG1".STA_RUN,
                        EMTY := "PLC_BIT".WAG1_EM,
                        W_OUT1 => "6.1.W_IND_AGG1".W_OUT1,
                        "%W_OUT" => "C#7_RD_RUN"."%_WAG1");
   END_IF;
   "9.5.DLR_IND_AGG1"(ON := "C#7_RD_RUN".WE_AG1 <= "C#4_WD_WEIGHT"."W_IND_AGG1_KL.BRO",   // "9.TIMER_DELAY"
                      CLOCK_1S := "Clock_10Hz",
                      T_DELAY := "9.5.DLR_IND_AGG1".T_DELAY,
                      OUT => "PLC_BIT".WAG1_EM,
                      T_OUT => "9.5.DLR_IND_AGG1".T_OUT,
                      ENO => #_w1);
   IF #_w1 THEN
       "9.5.DLR_IND_AGG1".T_DELAY := "C#4_WD_WEIGHT"."W_IND_AGG1_TG.DLD" + "C#3_WD_SILO".AG1_TG_ODC;
   END_IF;
   IF "PLC_BIT".RUN AND ("PLC_BIT".AGG1_FU OR ("C#4_WD_WEIGHT".SV_AG1 = 0.0)) THEN
       "PLC_BIT".WAG1_FU := TRUE;
   END_IF;
   #_w2 := "PLC_BIT".WAG1_EM AND NOT "P_WAGG1_EM";   // rising edge of "PLC_BIT".WAG1_EM
   "P_WAGG1_EM" := "PLC_BIT".WAG1_EM;
   IF #_w2 AND ("C#7_RD_RUN".SMC_AG1 > "C#7_RD_RUN".SMX_AG1) THEN
       "C#7_RD_RUN".SMX_AG1 := "C#7_RD_RUN".SMX_AG1 + 1.0;
   END_IF;
   IF #_w2 THEN "6.1.W_IND_AGG1".WR_IN := "C#7_RD_RUN".WE_AG1; END_IF;
   "LUU TAY WAG1" := #_w2 AND NOT "C#2_WB"."SW_MAN/AUTO" AND NOT "PLC_BIT".RUN;
   IF "PLC_BIT".WAG1_EM OR NOT "PLC_BIT".RUN THEN
       "PLC_BIT".AGG1_FU := FALSE;
       "PLC_BIT".WAG1_FU := FALSE;
   END_IF;
   #_w3 := "PLC_BIT".WAG1_FU AND NOT "P_WAGG1_FU";   // rising edge of "PLC_BIT".WAG1_FU
   "P_WAGG1_FU" := "PLC_BIT".WAG1_FU;
   IF (#_w3 OR ("P_RUN" AND "PLC_BIT".WAG1_FU)) AND NOT "C#1_RB"."XA W_IND_AGG1" AND ("C#7_RD_RUN".SMC_AG1 = "C#7_RD_RUN".SMX_AG1) THEN
       "C#7_RD_RUN".SMC_AG1 := "C#7_RD_RUN".SMC_AG1 + 1.0;
   END_IF;
END_REGION
END_FUNCTION

FUNCTION "FCCA_IND_AGG1" : Void   // FC20, LAD
{ S7_Optimized_Access := 'TRUE' }
VERSION : 0.1
// stored: AutoNumber false, CodeModifiedDate 2026-01-15T16:25:53.7815162Z, CompileDate 2026-01-15T16:25:53.8212538Z, CreationDate 2026-01-15T16:24:02.4619467Z, HandleErrorsWithinBlock false, InterfaceModifiedDate 2026-01-10T08:55:50.3009267Z, IsConsistent true, IsIECCheckEnabled false, IsKnowHowProtected false, IsWriteProtected false, LibraryConformanceStatus Error: The block contains calls of single instances. Warning: The object contains access to global data blocks. Warning: The block contains direct access to inputs, outputs, bit memories, indirect access to the registry or indirect access to external memory areas that are unknown at the time of compilation., ModifiedDate 2026-01-15T16:25:53.7815162Z, ParameterModified 2026-01-10T08:55:50.3009267Z, PLCSimAdvancedSupport false, SetENOAutomatically False, StructureModified 2026-01-10T08:55:50.3009267Z, UDAEnableTagReadback false
BEGIN

REGION Network 1: Trạng thái cân AGG1
   // Đầu tiên nó sẽ đợi một khoảng thời gian gọi là Thời gian trễ cân, sau đó nó mới đủ điều kiện để cân
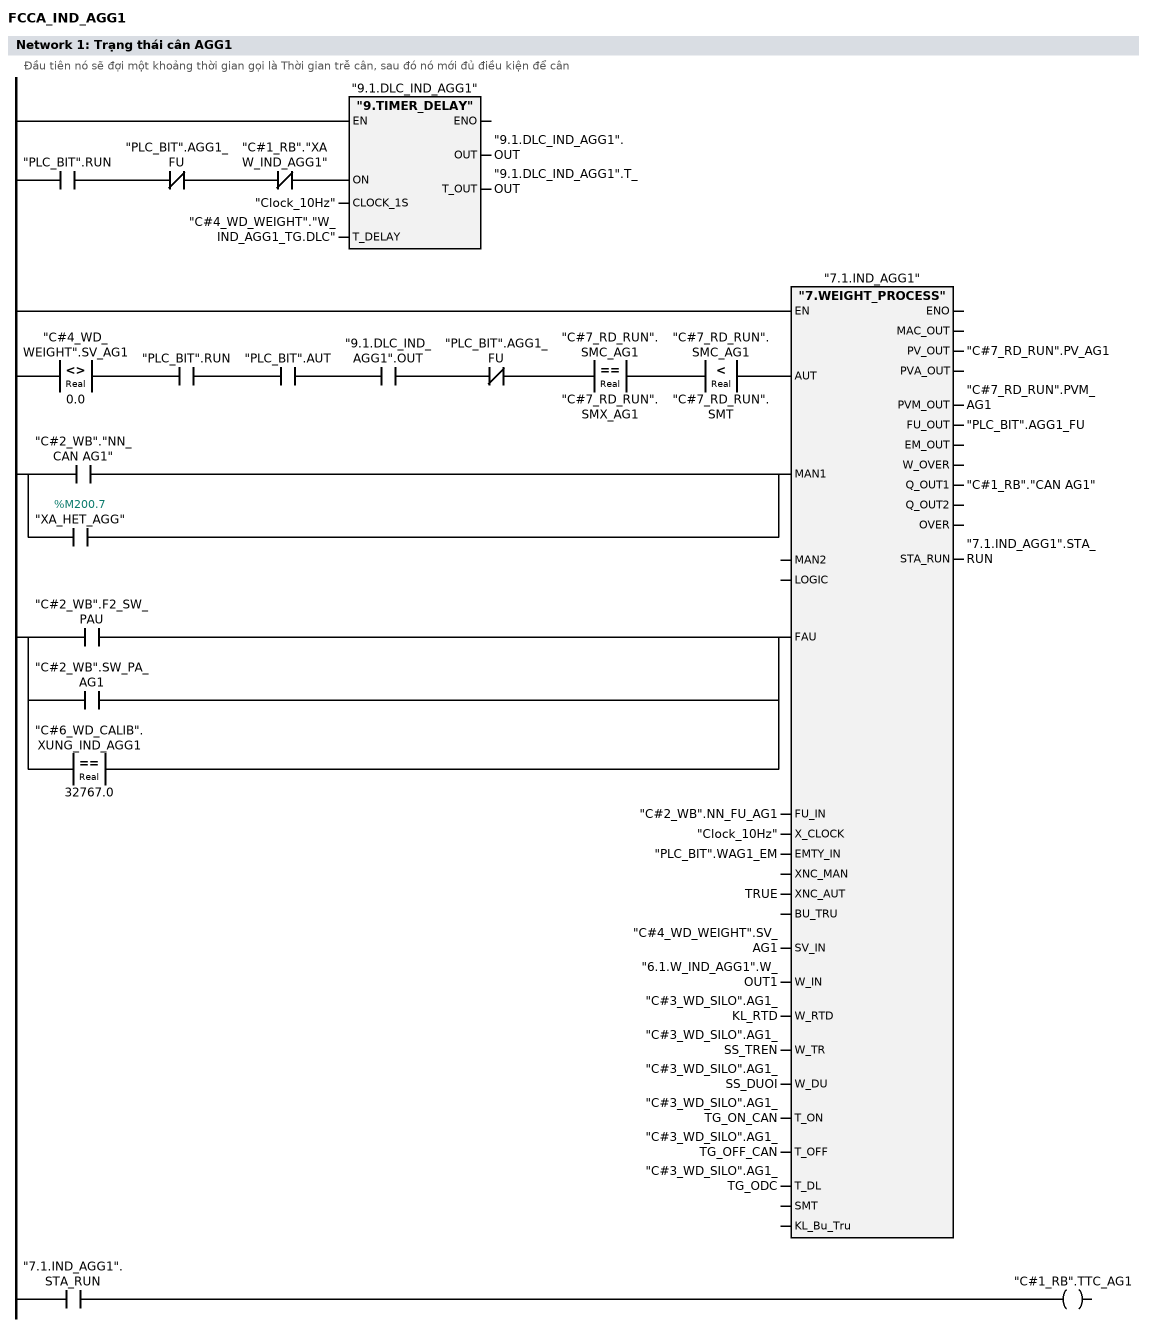
   RUNG wire#powerrail
      "9.1.DLC_IND_AGG1"(ON := wire#w1, CLOCK_1S := "Clock_10Hz", T_DELAY := "C#4_WD_WEIGHT"."W_IND_AGG1_TG.DLC", OUT => "9.1.DLC_IND_AGG1".OUT, T_OUT => "9.1.DLC_IND_AGG1".T_OUT)
   END_RUNG
   RUNG wire#powerrail
      Contact( "PLC_BIT".RUN )
      I_Contact( "PLC_BIT".AGG1_FU )
      I_Contact( "C#1_RB"."XA W_IND_AGG1" )
   END_RUNG wire#w1
   RUNG wire#powerrail
      "7.1.IND_AGG1"(AUT := wire#w2, MAN1 := wire#w3, FAU := wire#w4, MAN2 :=, LOGIC :=, FU_IN := "C#2_WB".NN_FU_AG1, X_CLOCK := "Clock_10Hz", EMTY_IN := "PLC_BIT".WAG1_EM, XNC_MAN :=, XNC_AUT := TRUE, BU_TRU :=, SV_IN := "C#4_WD_WEIGHT".SV_AG1, W_IN := "6.1.W_IND_AGG1".W_OUT1, W_RTD := "C#3_WD_SILO".AG1_KL_RTD, W_TR := "C#3_WD_SILO".AG1_SS_TREN, W_DU := "C#3_WD_SILO".AG1_SS_DUOI, T_ON := "C#3_WD_SILO".AG1_TG_ON_CAN, T_OFF := "C#3_WD_SILO".AG1_TG_OFF_CAN, T_DL := "C#3_WD_SILO".AG1_TG_ODC, SMT :=, KL_Bu_Tru :=, MAC_OUT =>, PV_OUT => "C#7_RD_RUN".PV_AG1, PVA_OUT =>, PVM_OUT => "C#7_RD_RUN".PVM_AG1, FU_OUT => "PLC_BIT".AGG1_FU, EM_OUT =>, W_OVER =>, Q_OUT1 => "C#1_RB"."CAN AG1", Q_OUT2 =>, OVER =>, STA_RUN => "7.1.IND_AGG1".STA_RUN)
   END_RUNG
   RUNG wire#powerrail
      { S7_Templates := "SrcType := Real" } NE_Contact(in1 := "C#4_WD_WEIGHT".SV_AG1, in2 := 0.0)
      Contact( "PLC_BIT".RUN )
      Contact( "PLC_BIT".AUT )
      Contact( "9.1.DLC_IND_AGG1".OUT )
      I_Contact( "PLC_BIT".AGG1_FU )
      { S7_Templates := "SrcType := Real" } EQ_Contact(in1 := "C#7_RD_RUN".SMC_AG1, in2 := "C#7_RD_RUN".SMX_AG1)
      { S7_Templates := "SrcType := Real" } LT_Contact(in1 := "C#7_RD_RUN".SMC_AG1, in2 := "C#7_RD_RUN".SMT)
   END_RUNG wire#w2
   RUNG wire#powerrail
      Contact( "C#2_WB"."NN_CAN AG1" )
   END_RUNG wire#w3
   RUNG wire#powerrail
      Contact( "XA_HET_AGG" )
   END_RUNG wire#w3
   RUNG wire#powerrail
      Contact( "C#2_WB".F2_SW_PAU )
   END_RUNG wire#w4
   RUNG wire#powerrail
      Contact( "C#2_WB".SW_PA_AG1 )
   END_RUNG wire#w4
   RUNG wire#powerrail
      { S7_Templates := "SrcType := Real" } EQ_Contact(in1 := "C#6_WD_CALIB".XUNG_IND_AGG1, in2 := 32767.0)
   END_RUNG wire#w4
   RUNG wire#powerrail
      Contact( "7.1.IND_AGG1".STA_RUN )
      Coil( "C#1_RB".TTC_AG1 )
   END_RUNG
   // the same network as SCL:
   "9.1.DLC_IND_AGG1"(ON := "PLC_BIT".RUN AND NOT "PLC_BIT".AGG1_FU AND NOT "C#1_RB"."XA W_IND_AGG1",   // "9.TIMER_DELAY"
                      CLOCK_1S := "Clock_10Hz",
                      T_DELAY := "C#4_WD_WEIGHT"."W_IND_AGG1_TG.DLC",
                      OUT => "9.1.DLC_IND_AGG1".OUT,
                      T_OUT => "9.1.DLC_IND_AGG1".T_OUT);
   "7.1.IND_AGG1"(AUT := ("C#4_WD_WEIGHT".SV_AG1 <> 0.0) AND "PLC_BIT".RUN AND "PLC_BIT".AUT AND "9.1.DLC_IND_AGG1".OUT AND NOT "PLC_BIT".AGG1_FU AND ("C#7_RD_RUN".SMC_AG1 = "C#7_RD_RUN".SMX_AG1) AND ("C#7_RD_RUN".SMC_AG1 < "C#7_RD_RUN".SMT),   // "7.WEIGHT_PROCESS"
                  MAN1 := "C#2_WB"."NN_CAN AG1" OR "XA_HET_AGG",
                  FAU := "C#2_WB".F2_SW_PAU OR "C#2_WB".SW_PA_AG1 OR ("C#6_WD_CALIB".XUNG_IND_AGG1 = 32767.0),
                  FU_IN := "C#2_WB".NN_FU_AG1,
                  X_CLOCK := "Clock_10Hz",
                  EMTY_IN := "PLC_BIT".WAG1_EM,
                  XNC_AUT := TRUE,
                  SV_IN := "C#4_WD_WEIGHT".SV_AG1,
                  W_IN := "6.1.W_IND_AGG1".W_OUT1,
                  W_RTD := "C#3_WD_SILO".AG1_KL_RTD,
                  W_TR := "C#3_WD_SILO".AG1_SS_TREN,
                  W_DU := "C#3_WD_SILO".AG1_SS_DUOI,
                  T_ON := "C#3_WD_SILO".AG1_TG_ON_CAN,
                  T_OFF := "C#3_WD_SILO".AG1_TG_OFF_CAN,
                  T_DL := "C#3_WD_SILO".AG1_TG_ODC,
                  PV_OUT => "C#7_RD_RUN".PV_AG1,
                  PVM_OUT => "C#7_RD_RUN".PVM_AG1,
                  FU_OUT => "PLC_BIT".AGG1_FU,
                  Q_OUT1 => "C#1_RB"."CAN AG1",
                  STA_RUN => "7.1.IND_AGG1".STA_RUN);
   "C#1_RB".TTC_AG1 := "7.1.IND_AGG1".STA_RUN;
END_REGION
END_FUNCTION

FUNCTION "FCXL_IND_AGG2" : Void   // FC21, LAD
{ S7_Optimized_Access := 'TRUE' }
VERSION : 0.1
// stored: AutoNumber true, CodeModifiedDate 2026-01-15T16:25:53.7007107Z, CompileDate 2026-01-15T16:25:53.7394906Z, CreationDate 2026-01-15T16:24:02.4619467Z, HandleErrorsWithinBlock false, InterfaceModifiedDate 2026-01-11T04:47:47.7058671Z, IsConsistent true, IsIECCheckEnabled false, IsKnowHowProtected false, IsWriteProtected false, LibraryConformanceStatus Error: The block contains calls of single instances. Warning: The object contains access to global data blocks. Warning: The block contains direct access to inputs, outputs, bit memories, indirect access to the registry or indirect access to external memory areas that are unknown at the time of compilation., ModifiedDate 2026-01-15T16:25:53.7007107Z, ParameterModified 2026-01-11T04:47:47.7058671Z, PLCSimAdvancedSupport false, SetENOAutomatically False, StructureModified 2026-01-11T04:47:47.7058671Z, UDAEnableTagReadback false
   VAR_TEMP   // added for the SCL form of the ladder/FBD networks
      _w1 : Bool;
      _w2 : Bool;
      _w3 : Bool;
   END_VAR
BEGIN

REGION Network 1: Cân độc lập AGG2 Full
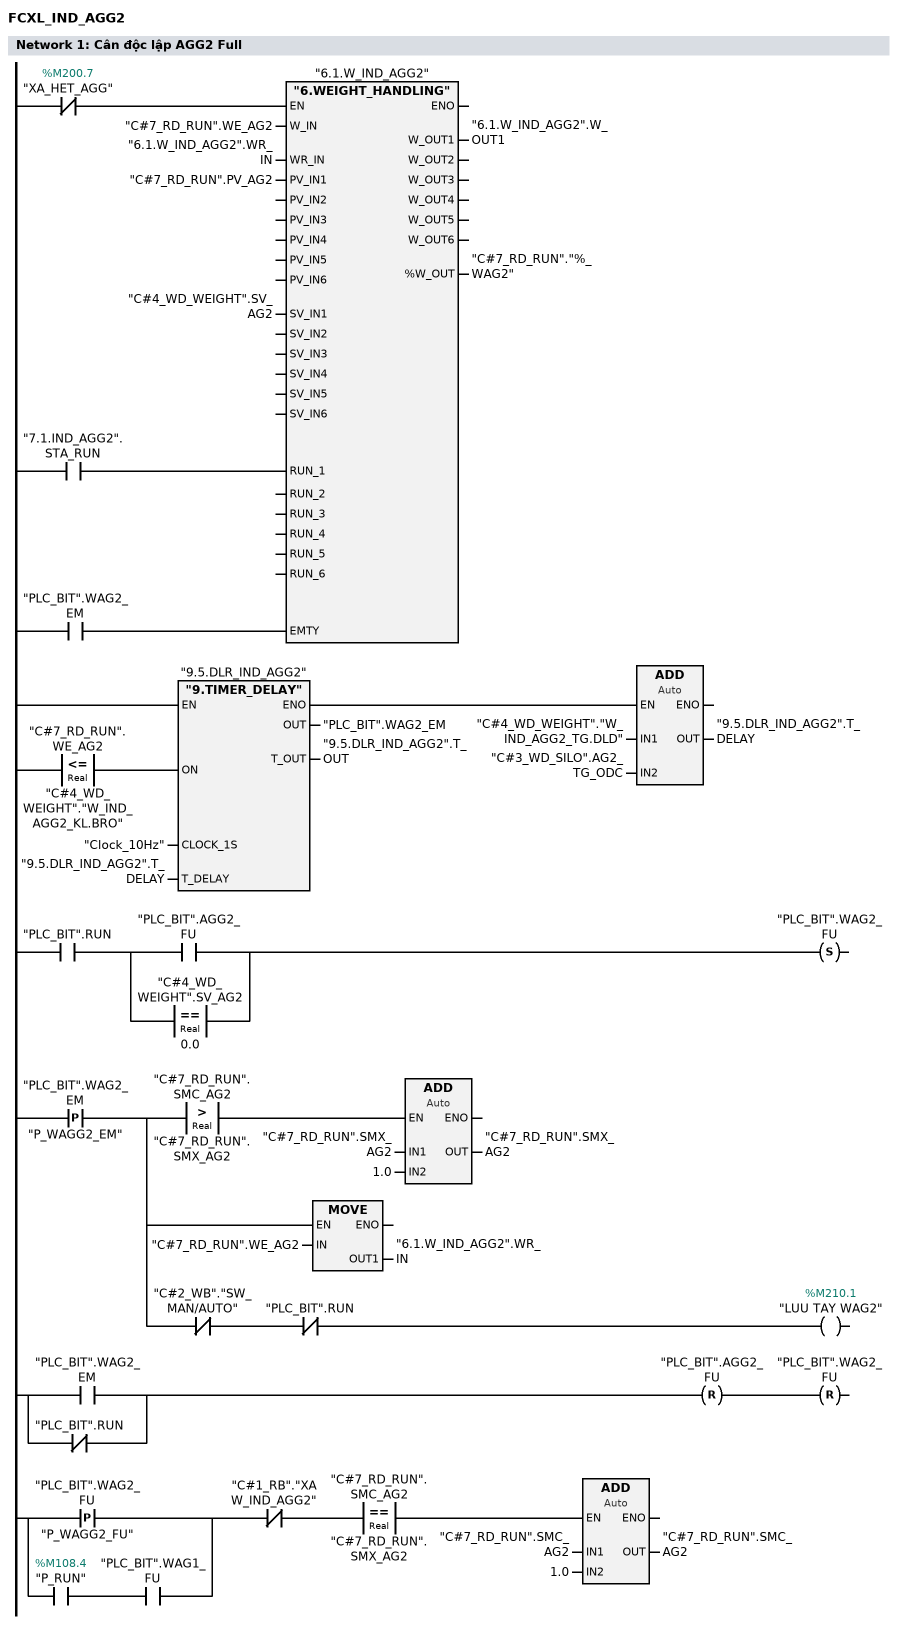
   RUNG wire#powerrail
      I_Contact( "XA_HET_AGG" )
      "6.1.W_IND_AGG2"(RUN_1 := wire#w1, EMTY := wire#w2, W_IN := "C#7_RD_RUN".WE_AG2, WR_IN := "6.1.W_IND_AGG2".WR_IN, PV_IN1 := "C#7_RD_RUN".PV_AG2, PV_IN2 :=, PV_IN3 :=, PV_IN4 :=, PV_IN5 :=, PV_IN6 :=, SV_IN1 := "C#4_WD_WEIGHT".SV_AG2, SV_IN2 :=, SV_IN3 :=, SV_IN4 :=, SV_IN5 :=, SV_IN6 :=, RUN_2 :=, RUN_3 :=, RUN_4 :=, RUN_5 :=, RUN_6 :=, W_OUT1 => "6.1.W_IND_AGG2".W_OUT1, W_OUT2 =>, W_OUT3 =>, W_OUT4 =>, W_OUT5 =>, W_OUT6 =>, "%W_OUT" => "C#7_RD_RUN"."%_WAG2")
   END_RUNG
   RUNG wire#powerrail
      Contact( "7.1.IND_AGG2".STA_RUN )
   END_RUNG wire#w1
   RUNG wire#powerrail
      Contact( "PLC_BIT".WAG2_EM )
   END_RUNG wire#w2
   RUNG wire#powerrail
      "9.5.DLR_IND_AGG2"(ON := wire#w3, CLOCK_1S := "Clock_10Hz", T_DELAY := "9.5.DLR_IND_AGG2".T_DELAY, OUT => "PLC_BIT".WAG2_EM, T_OUT => "9.5.DLR_IND_AGG2".T_OUT)
      Add(in1 := "C#4_WD_WEIGHT"."W_IND_AGG2_TG.DLD", in2 := "C#3_WD_SILO".AG2_TG_ODC, out => "9.5.DLR_IND_AGG2".T_DELAY)
   END_RUNG
   RUNG wire#powerrail
      { S7_Templates := "SrcType := Real" } LE_Contact(in1 := "C#7_RD_RUN".WE_AG2, in2 := "C#4_WD_WEIGHT"."W_IND_AGG2_KL.BRO")
   END_RUNG wire#w3
   RUNG wire#powerrail
      Contact( "PLC_BIT".RUN )
      wire#w4
      Contact( "PLC_BIT".AGG2_FU )
      wire#w5
      S_Coil( "PLC_BIT".WAG2_FU )
   END_RUNG
   RUNG wire#w4
      { S7_Templates := "SrcType := Real" } EQ_Contact(in1 := "C#4_WD_WEIGHT".SV_AG2, in2 := 0.0)
   END_RUNG wire#w5
   RUNG wire#powerrail
      P_Contact(operand := "PLC_BIT".WAG2_EM, bit := "P_WAGG2_EM")
      wire#w6
      { S7_Templates := "SrcType := Real" } GT_Contact(in1 := "C#7_RD_RUN".SMC_AG2, in2 := "C#7_RD_RUN".SMX_AG2)
      Add(in1 := "C#7_RD_RUN".SMX_AG2, in2 := 1.0, out => "C#7_RD_RUN".SMX_AG2)
   END_RUNG
   RUNG wire#w6
      Move(in := "C#7_RD_RUN".WE_AG2, out1 => "6.1.W_IND_AGG2".WR_IN)
   END_RUNG
   RUNG wire#w6
      I_Contact( "C#2_WB"."SW_MAN/AUTO" )
      I_Contact( "PLC_BIT".RUN )
      Coil( "LUU TAY WAG2" )
   END_RUNG
   RUNG wire#powerrail
      Contact( "PLC_BIT".WAG2_EM )
      wire#w7
      R_Coil( "PLC_BIT".AGG2_FU )
      R_Coil( "PLC_BIT".WAG2_FU )
   END_RUNG
   RUNG wire#powerrail
      I_Contact( "PLC_BIT".RUN )
   END_RUNG wire#w7
   RUNG wire#powerrail
      P_Contact(operand := "PLC_BIT".WAG2_FU, bit := "P_WAGG2_FU")
      wire#w8
      I_Contact( "C#1_RB"."XA W_IND_AGG2" )
      { S7_Templates := "SrcType := Real" } EQ_Contact(in1 := "C#7_RD_RUN".SMC_AG2, in2 := "C#7_RD_RUN".SMX_AG2)
      Add(in1 := "C#7_RD_RUN".SMC_AG2, in2 := 1.0, out => "C#7_RD_RUN".SMC_AG2)
   END_RUNG
   RUNG wire#powerrail
      Contact( "P_RUN" )
      Contact( "PLC_BIT".WAG1_FU )
   END_RUNG wire#w8
   // the same network as SCL:
   IF NOT "XA_HET_AGG" THEN
       "6.1.W_IND_AGG2"(W_IN := "C#7_RD_RUN".WE_AG2,   // "6.WEIGHT_HANDLING"
                        WR_IN := "6.1.W_IND_AGG2".WR_IN,
                        PV_IN1 := "C#7_RD_RUN".PV_AG2,
                        SV_IN1 := "C#4_WD_WEIGHT".SV_AG2,
                        RUN_1 := "7.1.IND_AGG2".STA_RUN,
                        EMTY := "PLC_BIT".WAG2_EM,
                        W_OUT1 => "6.1.W_IND_AGG2".W_OUT1,
                        "%W_OUT" => "C#7_RD_RUN"."%_WAG2");
   END_IF;
   "9.5.DLR_IND_AGG2"(ON := "C#7_RD_RUN".WE_AG2 <= "C#4_WD_WEIGHT"."W_IND_AGG2_KL.BRO",   // "9.TIMER_DELAY"
                      CLOCK_1S := "Clock_10Hz",
                      T_DELAY := "9.5.DLR_IND_AGG2".T_DELAY,
                      OUT => "PLC_BIT".WAG2_EM,
                      T_OUT => "9.5.DLR_IND_AGG2".T_OUT,
                      ENO => #_w1);
   IF #_w1 THEN
       "9.5.DLR_IND_AGG2".T_DELAY := "C#4_WD_WEIGHT"."W_IND_AGG2_TG.DLD" + "C#3_WD_SILO".AG2_TG_ODC;
   END_IF;
   IF "PLC_BIT".RUN AND ("PLC_BIT".AGG2_FU OR ("C#4_WD_WEIGHT".SV_AG2 = 0.0)) THEN
       "PLC_BIT".WAG2_FU := TRUE;
   END_IF;
   #_w2 := "PLC_BIT".WAG2_EM AND NOT "P_WAGG2_EM";   // rising edge of "PLC_BIT".WAG2_EM
   "P_WAGG2_EM" := "PLC_BIT".WAG2_EM;
   IF #_w2 AND ("C#7_RD_RUN".SMC_AG2 > "C#7_RD_RUN".SMX_AG2) THEN
       "C#7_RD_RUN".SMX_AG2 := "C#7_RD_RUN".SMX_AG2 + 1.0;
   END_IF;
   IF #_w2 THEN "6.1.W_IND_AGG2".WR_IN := "C#7_RD_RUN".WE_AG2; END_IF;
   "LUU TAY WAG2" := #_w2 AND NOT "C#2_WB"."SW_MAN/AUTO" AND NOT "PLC_BIT".RUN;
   IF "PLC_BIT".WAG2_EM OR NOT "PLC_BIT".RUN THEN
       "PLC_BIT".AGG2_FU := FALSE;
       "PLC_BIT".WAG2_FU := FALSE;
   END_IF;
   #_w3 := "PLC_BIT".WAG2_FU AND NOT "P_WAGG2_FU";   // rising edge of "PLC_BIT".WAG2_FU
   "P_WAGG2_FU" := "PLC_BIT".WAG2_FU;
   IF (#_w3 OR ("P_RUN" AND "PLC_BIT".WAG1_FU)) AND NOT "C#1_RB"."XA W_IND_AGG2" AND ("C#7_RD_RUN".SMC_AG2 = "C#7_RD_RUN".SMX_AG2) THEN
       "C#7_RD_RUN".SMC_AG2 := "C#7_RD_RUN".SMC_AG2 + 1.0;
   END_IF;
END_REGION
END_FUNCTION

FUNCTION "FCCA_IND_AGG2" : Void   // FC8, LAD
{ S7_Optimized_Access := 'TRUE' }
VERSION : 0.1
// stored: AutoNumber true, CodeModifiedDate 2026-01-15T16:25:55.0920194Z, CompileDate 2026-01-15T16:25:55.1307959Z, CreationDate 2026-01-15T16:24:02.4619467Z, HandleErrorsWithinBlock false, InterfaceModifiedDate 2026-01-11T04:46:28.8679318Z, IsConsistent true, IsIECCheckEnabled false, IsKnowHowProtected false, IsWriteProtected false, LibraryConformanceStatus Error: The block contains calls of single instances. Warning: The object contains access to global data blocks. Warning: The block contains direct access to inputs, outputs, bit memories, indirect access to the registry or indirect access to external memory areas that are unknown at the time of compilation., ModifiedDate 2026-01-15T16:25:55.0920194Z, ParameterModified 2026-01-11T04:46:28.8679318Z, PLCSimAdvancedSupport false, SetENOAutomatically False, StructureModified 2026-01-11T04:46:28.8679318Z, UDAEnableTagReadback false
BEGIN

REGION Network 1: Trạng thái cân AGG2
   // Đầu tiên nó sẽ đợi một khoảng thời gian gọi là Thời gian trễ cân, sau đó nó mới đủ điều kiện để cân
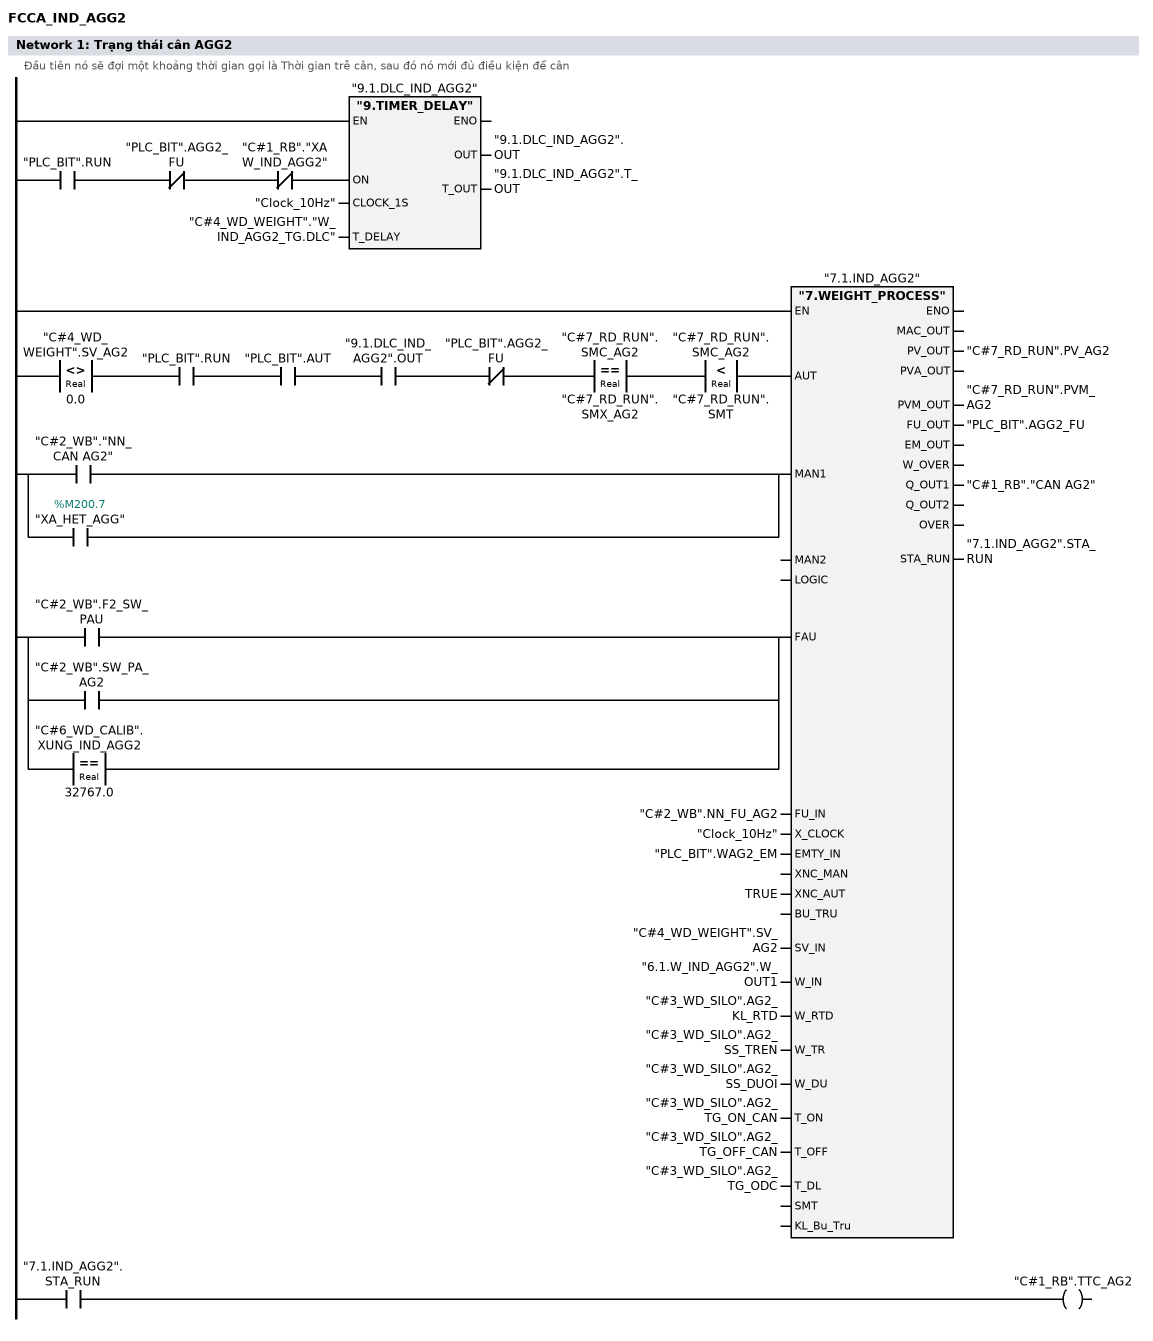
   RUNG wire#powerrail
      "9.1.DLC_IND_AGG2"(ON := wire#w1, CLOCK_1S := "Clock_10Hz", T_DELAY := "C#4_WD_WEIGHT"."W_IND_AGG2_TG.DLC", OUT => "9.1.DLC_IND_AGG2".OUT, T_OUT => "9.1.DLC_IND_AGG2".T_OUT)
   END_RUNG
   RUNG wire#powerrail
      Contact( "PLC_BIT".RUN )
      I_Contact( "PLC_BIT".AGG2_FU )
      I_Contact( "C#1_RB"."XA W_IND_AGG2" )
   END_RUNG wire#w1
   RUNG wire#powerrail
      "7.1.IND_AGG2"(AUT := wire#w2, MAN1 := wire#w3, FAU := wire#w4, MAN2 :=, LOGIC :=, FU_IN := "C#2_WB".NN_FU_AG2, X_CLOCK := "Clock_10Hz", EMTY_IN := "PLC_BIT".WAG2_EM, XNC_MAN :=, XNC_AUT := TRUE, BU_TRU :=, SV_IN := "C#4_WD_WEIGHT".SV_AG2, W_IN := "6.1.W_IND_AGG2".W_OUT1, W_RTD := "C#3_WD_SILO".AG2_KL_RTD, W_TR := "C#3_WD_SILO".AG2_SS_TREN, W_DU := "C#3_WD_SILO".AG2_SS_DUOI, T_ON := "C#3_WD_SILO".AG2_TG_ON_CAN, T_OFF := "C#3_WD_SILO".AG2_TG_OFF_CAN, T_DL := "C#3_WD_SILO".AG2_TG_ODC, SMT :=, KL_Bu_Tru :=, MAC_OUT =>, PV_OUT => "C#7_RD_RUN".PV_AG2, PVA_OUT =>, PVM_OUT => "C#7_RD_RUN".PVM_AG2, FU_OUT => "PLC_BIT".AGG2_FU, EM_OUT =>, W_OVER =>, Q_OUT1 => "C#1_RB"."CAN AG2", Q_OUT2 =>, OVER =>, STA_RUN => "7.1.IND_AGG2".STA_RUN)
   END_RUNG
   RUNG wire#powerrail
      { S7_Templates := "SrcType := Real" } NE_Contact(in1 := "C#4_WD_WEIGHT".SV_AG2, in2 := 0.0)
      Contact( "PLC_BIT".RUN )
      Contact( "PLC_BIT".AUT )
      Contact( "9.1.DLC_IND_AGG2".OUT )
      I_Contact( "PLC_BIT".AGG2_FU )
      { S7_Templates := "SrcType := Real" } EQ_Contact(in1 := "C#7_RD_RUN".SMC_AG2, in2 := "C#7_RD_RUN".SMX_AG2)
      { S7_Templates := "SrcType := Real" } LT_Contact(in1 := "C#7_RD_RUN".SMC_AG2, in2 := "C#7_RD_RUN".SMT)
   END_RUNG wire#w2
   RUNG wire#powerrail
      Contact( "C#2_WB"."NN_CAN AG2" )
   END_RUNG wire#w3
   RUNG wire#powerrail
      Contact( "XA_HET_AGG" )
   END_RUNG wire#w3
   RUNG wire#powerrail
      Contact( "C#2_WB".F2_SW_PAU )
   END_RUNG wire#w4
   RUNG wire#powerrail
      Contact( "C#2_WB".SW_PA_AG2 )
   END_RUNG wire#w4
   RUNG wire#powerrail
      { S7_Templates := "SrcType := Real" } EQ_Contact(in1 := "C#6_WD_CALIB".XUNG_IND_AGG2, in2 := 32767.0)
   END_RUNG wire#w4
   RUNG wire#powerrail
      Contact( "7.1.IND_AGG2".STA_RUN )
      Coil( "C#1_RB".TTC_AG2 )
   END_RUNG
   // the same network as SCL:
   "9.1.DLC_IND_AGG2"(ON := "PLC_BIT".RUN AND NOT "PLC_BIT".AGG2_FU AND NOT "C#1_RB"."XA W_IND_AGG2",   // "9.TIMER_DELAY"
                      CLOCK_1S := "Clock_10Hz",
                      T_DELAY := "C#4_WD_WEIGHT"."W_IND_AGG2_TG.DLC",
                      OUT => "9.1.DLC_IND_AGG2".OUT,
                      T_OUT => "9.1.DLC_IND_AGG2".T_OUT);
   "7.1.IND_AGG2"(AUT := ("C#4_WD_WEIGHT".SV_AG2 <> 0.0) AND "PLC_BIT".RUN AND "PLC_BIT".AUT AND "9.1.DLC_IND_AGG2".OUT AND NOT "PLC_BIT".AGG2_FU AND ("C#7_RD_RUN".SMC_AG2 = "C#7_RD_RUN".SMX_AG2) AND ("C#7_RD_RUN".SMC_AG2 < "C#7_RD_RUN".SMT),   // "7.WEIGHT_PROCESS"
                  MAN1 := "C#2_WB"."NN_CAN AG2" OR "XA_HET_AGG",
                  FAU := "C#2_WB".F2_SW_PAU OR "C#2_WB".SW_PA_AG2 OR ("C#6_WD_CALIB".XUNG_IND_AGG2 = 32767.0),
                  FU_IN := "C#2_WB".NN_FU_AG2,
                  X_CLOCK := "Clock_10Hz",
                  EMTY_IN := "PLC_BIT".WAG2_EM,
                  XNC_AUT := TRUE,
                  SV_IN := "C#4_WD_WEIGHT".SV_AG2,
                  W_IN := "6.1.W_IND_AGG2".W_OUT1,
                  W_RTD := "C#3_WD_SILO".AG2_KL_RTD,
                  W_TR := "C#3_WD_SILO".AG2_SS_TREN,
                  W_DU := "C#3_WD_SILO".AG2_SS_DUOI,
                  T_ON := "C#3_WD_SILO".AG2_TG_ON_CAN,
                  T_OFF := "C#3_WD_SILO".AG2_TG_OFF_CAN,
                  T_DL := "C#3_WD_SILO".AG2_TG_ODC,
                  PV_OUT => "C#7_RD_RUN".PV_AG2,
                  PVM_OUT => "C#7_RD_RUN".PVM_AG2,
                  FU_OUT => "PLC_BIT".AGG2_FU,
                  Q_OUT1 => "C#1_RB"."CAN AG2",
                  STA_RUN => "7.1.IND_AGG2".STA_RUN);
   "C#1_RB".TTC_AG2 := "7.1.IND_AGG2".STA_RUN;
END_REGION
END_FUNCTION

FUNCTION "FCXL_IND_AGG3" : Void   // FC22, LAD
{ S7_Optimized_Access := 'TRUE' }
VERSION : 0.1
// stored: AutoNumber true, CodeModifiedDate 2026-01-15T16:25:53.6082795Z, CompileDate 2026-01-15T16:25:53.6491144Z, CreationDate 2026-01-15T16:24:02.4619467Z, HandleErrorsWithinBlock false, InterfaceModifiedDate 2026-01-11T04:48:05.8897553Z, IsConsistent true, IsIECCheckEnabled false, IsKnowHowProtected false, IsWriteProtected false, LibraryConformanceStatus Error: The block contains calls of single instances. Warning: The object contains access to global data blocks. Warning: The block contains direct access to inputs, outputs, bit memories, indirect access to the registry or indirect access to external memory areas that are unknown at the time of compilation., ModifiedDate 2026-01-15T16:25:53.6082795Z, ParameterModified 2026-01-11T04:48:05.8897553Z, PLCSimAdvancedSupport false, SetENOAutomatically False, StructureModified 2026-01-11T04:48:05.8897553Z, UDAEnableTagReadback false
   VAR_TEMP   // added for the SCL form of the ladder/FBD networks
      _w1 : Bool;
      _w2 : Bool;
      _w3 : Bool;
   END_VAR
BEGIN

REGION Network 1: Cân độc lập AGG3 Full
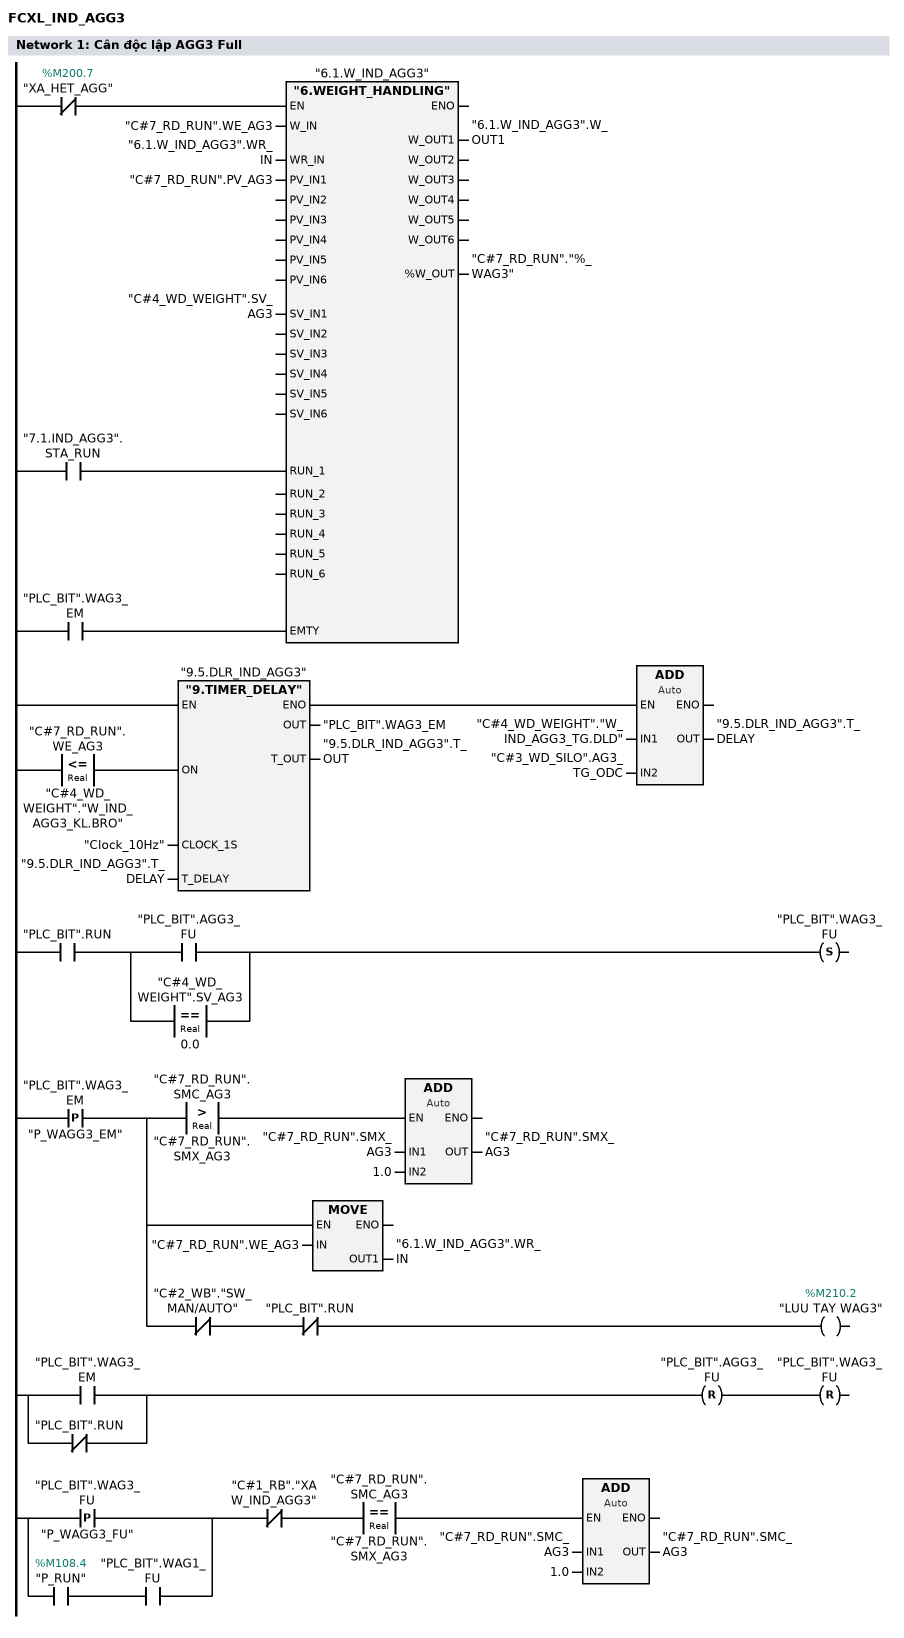
   RUNG wire#powerrail
      I_Contact( "XA_HET_AGG" )
      "6.1.W_IND_AGG3"(RUN_1 := wire#w1, EMTY := wire#w2, W_IN := "C#7_RD_RUN".WE_AG3, WR_IN := "6.1.W_IND_AGG3".WR_IN, PV_IN1 := "C#7_RD_RUN".PV_AG3, PV_IN2 :=, PV_IN3 :=, PV_IN4 :=, PV_IN5 :=, PV_IN6 :=, SV_IN1 := "C#4_WD_WEIGHT".SV_AG3, SV_IN2 :=, SV_IN3 :=, SV_IN4 :=, SV_IN5 :=, SV_IN6 :=, RUN_2 :=, RUN_3 :=, RUN_4 :=, RUN_5 :=, RUN_6 :=, W_OUT1 => "6.1.W_IND_AGG3".W_OUT1, W_OUT2 =>, W_OUT3 =>, W_OUT4 =>, W_OUT5 =>, W_OUT6 =>, "%W_OUT" => "C#7_RD_RUN"."%_WAG3")
   END_RUNG
   RUNG wire#powerrail
      Contact( "7.1.IND_AGG3".STA_RUN )
   END_RUNG wire#w1
   RUNG wire#powerrail
      Contact( "PLC_BIT".WAG3_EM )
   END_RUNG wire#w2
   RUNG wire#powerrail
      "9.5.DLR_IND_AGG3"(ON := wire#w3, CLOCK_1S := "Clock_10Hz", T_DELAY := "9.5.DLR_IND_AGG3".T_DELAY, OUT => "PLC_BIT".WAG3_EM, T_OUT => "9.5.DLR_IND_AGG3".T_OUT)
      Add(in1 := "C#4_WD_WEIGHT"."W_IND_AGG3_TG.DLD", in2 := "C#3_WD_SILO".AG3_TG_ODC, out => "9.5.DLR_IND_AGG3".T_DELAY)
   END_RUNG
   RUNG wire#powerrail
      { S7_Templates := "SrcType := Real" } LE_Contact(in1 := "C#7_RD_RUN".WE_AG3, in2 := "C#4_WD_WEIGHT"."W_IND_AGG3_KL.BRO")
   END_RUNG wire#w3
   RUNG wire#powerrail
      Contact( "PLC_BIT".RUN )
      wire#w4
      Contact( "PLC_BIT".AGG3_FU )
      wire#w5
      S_Coil( "PLC_BIT".WAG3_FU )
   END_RUNG
   RUNG wire#w4
      { S7_Templates := "SrcType := Real" } EQ_Contact(in1 := "C#4_WD_WEIGHT".SV_AG3, in2 := 0.0)
   END_RUNG wire#w5
   RUNG wire#powerrail
      P_Contact(operand := "PLC_BIT".WAG3_EM, bit := "P_WAGG3_EM")
      wire#w6
      { S7_Templates := "SrcType := Real" } GT_Contact(in1 := "C#7_RD_RUN".SMC_AG3, in2 := "C#7_RD_RUN".SMX_AG3)
      Add(in1 := "C#7_RD_RUN".SMX_AG3, in2 := 1.0, out => "C#7_RD_RUN".SMX_AG3)
   END_RUNG
   RUNG wire#w6
      Move(in := "C#7_RD_RUN".WE_AG3, out1 => "6.1.W_IND_AGG3".WR_IN)
   END_RUNG
   RUNG wire#w6
      I_Contact( "C#2_WB"."SW_MAN/AUTO" )
      I_Contact( "PLC_BIT".RUN )
      Coil( "LUU TAY WAG3" )
   END_RUNG
   RUNG wire#powerrail
      Contact( "PLC_BIT".WAG3_EM )
      wire#w7
      R_Coil( "PLC_BIT".AGG3_FU )
      R_Coil( "PLC_BIT".WAG3_FU )
   END_RUNG
   RUNG wire#powerrail
      I_Contact( "PLC_BIT".RUN )
   END_RUNG wire#w7
   RUNG wire#powerrail
      P_Contact(operand := "PLC_BIT".WAG3_FU, bit := "P_WAGG3_FU")
      wire#w8
      I_Contact( "C#1_RB"."XA W_IND_AGG3" )
      { S7_Templates := "SrcType := Real" } EQ_Contact(in1 := "C#7_RD_RUN".SMC_AG3, in2 := "C#7_RD_RUN".SMX_AG3)
      Add(in1 := "C#7_RD_RUN".SMC_AG3, in2 := 1.0, out => "C#7_RD_RUN".SMC_AG3)
   END_RUNG
   RUNG wire#powerrail
      Contact( "P_RUN" )
      Contact( "PLC_BIT".WAG1_FU )
   END_RUNG wire#w8
   // the same network as SCL:
   IF NOT "XA_HET_AGG" THEN
       "6.1.W_IND_AGG3"(W_IN := "C#7_RD_RUN".WE_AG3,   // "6.WEIGHT_HANDLING"
                        WR_IN := "6.1.W_IND_AGG3".WR_IN,
                        PV_IN1 := "C#7_RD_RUN".PV_AG3,
                        SV_IN1 := "C#4_WD_WEIGHT".SV_AG3,
                        RUN_1 := "7.1.IND_AGG3".STA_RUN,
                        EMTY := "PLC_BIT".WAG3_EM,
                        W_OUT1 => "6.1.W_IND_AGG3".W_OUT1,
                        "%W_OUT" => "C#7_RD_RUN"."%_WAG3");
   END_IF;
   "9.5.DLR_IND_AGG3"(ON := "C#7_RD_RUN".WE_AG3 <= "C#4_WD_WEIGHT"."W_IND_AGG3_KL.BRO",   // "9.TIMER_DELAY"
                      CLOCK_1S := "Clock_10Hz",
                      T_DELAY := "9.5.DLR_IND_AGG3".T_DELAY,
                      OUT => "PLC_BIT".WAG3_EM,
                      T_OUT => "9.5.DLR_IND_AGG3".T_OUT,
                      ENO => #_w1);
   IF #_w1 THEN
       "9.5.DLR_IND_AGG3".T_DELAY := "C#4_WD_WEIGHT"."W_IND_AGG3_TG.DLD" + "C#3_WD_SILO".AG3_TG_ODC;
   END_IF;
   IF "PLC_BIT".RUN AND ("PLC_BIT".AGG3_FU OR ("C#4_WD_WEIGHT".SV_AG3 = 0.0)) THEN
       "PLC_BIT".WAG3_FU := TRUE;
   END_IF;
   #_w2 := "PLC_BIT".WAG3_EM AND NOT "P_WAGG3_EM";   // rising edge of "PLC_BIT".WAG3_EM
   "P_WAGG3_EM" := "PLC_BIT".WAG3_EM;
   IF #_w2 AND ("C#7_RD_RUN".SMC_AG3 > "C#7_RD_RUN".SMX_AG3) THEN
       "C#7_RD_RUN".SMX_AG3 := "C#7_RD_RUN".SMX_AG3 + 1.0;
   END_IF;
   IF #_w2 THEN "6.1.W_IND_AGG3".WR_IN := "C#7_RD_RUN".WE_AG3; END_IF;
   "LUU TAY WAG3" := #_w2 AND NOT "C#2_WB"."SW_MAN/AUTO" AND NOT "PLC_BIT".RUN;
   IF "PLC_BIT".WAG3_EM OR NOT "PLC_BIT".RUN THEN
       "PLC_BIT".AGG3_FU := FALSE;
       "PLC_BIT".WAG3_FU := FALSE;
   END_IF;
   #_w3 := "PLC_BIT".WAG3_FU AND NOT "P_WAGG3_FU";   // rising edge of "PLC_BIT".WAG3_FU
   "P_WAGG3_FU" := "PLC_BIT".WAG3_FU;
   IF (#_w3 OR ("P_RUN" AND "PLC_BIT".WAG1_FU)) AND NOT "C#1_RB"."XA W_IND_AGG3" AND ("C#7_RD_RUN".SMC_AG3 = "C#7_RD_RUN".SMX_AG3) THEN
       "C#7_RD_RUN".SMC_AG3 := "C#7_RD_RUN".SMC_AG3 + 1.0;
   END_IF;
END_REGION
END_FUNCTION

FUNCTION "FCCA_IND_AGG3" : Void   // FC11, LAD
{ S7_Optimized_Access := 'TRUE' }
VERSION : 0.1
// stored: AutoNumber true, CodeModifiedDate 2026-01-15T16:25:54.8129712Z, CompileDate 2026-01-15T16:25:54.8463711Z, CreationDate 2026-01-15T16:24:02.4619467Z, HandleErrorsWithinBlock false, InterfaceModifiedDate 2026-01-11T04:46:44.6799525Z, IsConsistent true, IsIECCheckEnabled false, IsKnowHowProtected false, IsWriteProtected false, LibraryConformanceStatus Error: The block contains calls of single instances. Warning: The object contains access to global data blocks. Warning: The block contains direct access to inputs, outputs, bit memories, indirect access to the registry or indirect access to external memory areas that are unknown at the time of compilation., ModifiedDate 2026-01-15T16:25:54.8129712Z, ParameterModified 2026-01-11T04:46:44.6799525Z, PLCSimAdvancedSupport false, SetENOAutomatically False, StructureModified 2026-01-11T04:46:44.6799525Z, UDAEnableTagReadback false
BEGIN

REGION Network 1: Trạng thái cân AGG3
   // Đầu tiên nó sẽ đợi một khoảng thời gian gọi là Thời gian trễ cân, sau đó nó mới đủ điều kiện để cân
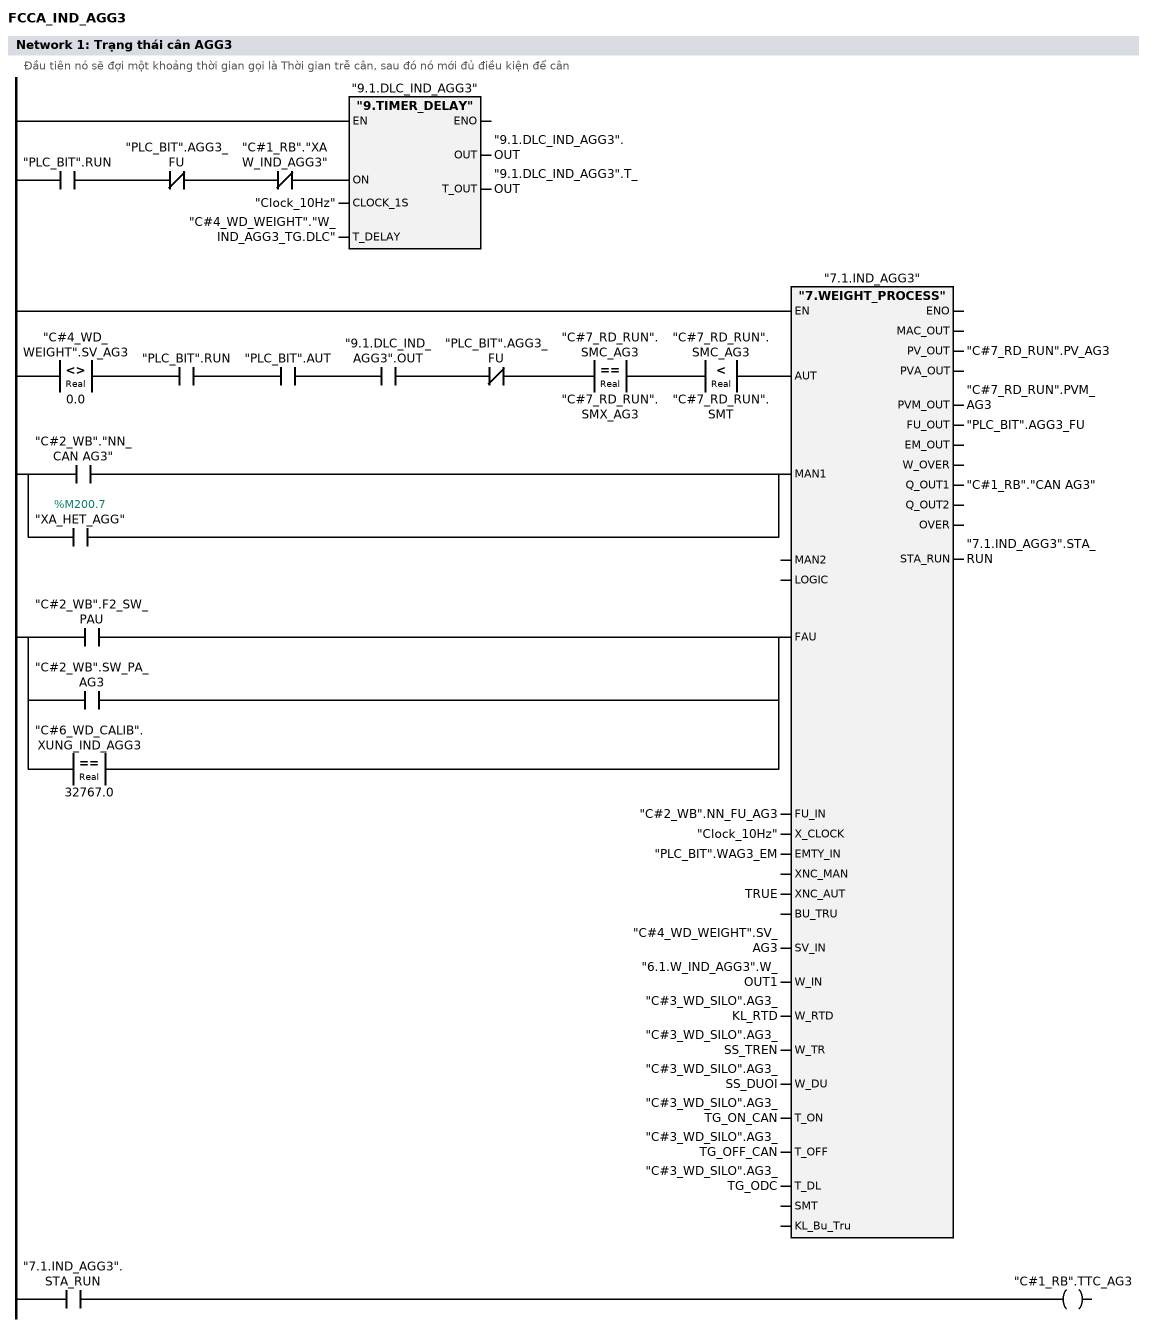
   RUNG wire#powerrail
      "9.1.DLC_IND_AGG3"(ON := wire#w1, CLOCK_1S := "Clock_10Hz", T_DELAY := "C#4_WD_WEIGHT"."W_IND_AGG3_TG.DLC", OUT => "9.1.DLC_IND_AGG3".OUT, T_OUT => "9.1.DLC_IND_AGG3".T_OUT)
   END_RUNG
   RUNG wire#powerrail
      Contact( "PLC_BIT".RUN )
      I_Contact( "PLC_BIT".AGG3_FU )
      I_Contact( "C#1_RB"."XA W_IND_AGG3" )
   END_RUNG wire#w1
   RUNG wire#powerrail
      "7.1.IND_AGG3"(AUT := wire#w2, MAN1 := wire#w3, FAU := wire#w4, MAN2 :=, LOGIC :=, FU_IN := "C#2_WB".NN_FU_AG3, X_CLOCK := "Clock_10Hz", EMTY_IN := "PLC_BIT".WAG3_EM, XNC_MAN :=, XNC_AUT := TRUE, BU_TRU :=, SV_IN := "C#4_WD_WEIGHT".SV_AG3, W_IN := "6.1.W_IND_AGG3".W_OUT1, W_RTD := "C#3_WD_SILO".AG3_KL_RTD, W_TR := "C#3_WD_SILO".AG3_SS_TREN, W_DU := "C#3_WD_SILO".AG3_SS_DUOI, T_ON := "C#3_WD_SILO".AG3_TG_ON_CAN, T_OFF := "C#3_WD_SILO".AG3_TG_OFF_CAN, T_DL := "C#3_WD_SILO".AG3_TG_ODC, SMT :=, KL_Bu_Tru :=, MAC_OUT =>, PV_OUT => "C#7_RD_RUN".PV_AG3, PVA_OUT =>, PVM_OUT => "C#7_RD_RUN".PVM_AG3, FU_OUT => "PLC_BIT".AGG3_FU, EM_OUT =>, W_OVER =>, Q_OUT1 => "C#1_RB"."CAN AG3", Q_OUT2 =>, OVER =>, STA_RUN => "7.1.IND_AGG3".STA_RUN)
   END_RUNG
   RUNG wire#powerrail
      { S7_Templates := "SrcType := Real" } NE_Contact(in1 := "C#4_WD_WEIGHT".SV_AG3, in2 := 0.0)
      Contact( "PLC_BIT".RUN )
      Contact( "PLC_BIT".AUT )
      Contact( "9.1.DLC_IND_AGG3".OUT )
      I_Contact( "PLC_BIT".AGG3_FU )
      { S7_Templates := "SrcType := Real" } EQ_Contact(in1 := "C#7_RD_RUN".SMC_AG3, in2 := "C#7_RD_RUN".SMX_AG3)
      { S7_Templates := "SrcType := Real" } LT_Contact(in1 := "C#7_RD_RUN".SMC_AG3, in2 := "C#7_RD_RUN".SMT)
   END_RUNG wire#w2
   RUNG wire#powerrail
      Contact( "C#2_WB"."NN_CAN AG3" )
   END_RUNG wire#w3
   RUNG wire#powerrail
      Contact( "XA_HET_AGG" )
   END_RUNG wire#w3
   RUNG wire#powerrail
      Contact( "C#2_WB".F2_SW_PAU )
   END_RUNG wire#w4
   RUNG wire#powerrail
      Contact( "C#2_WB".SW_PA_AG3 )
   END_RUNG wire#w4
   RUNG wire#powerrail
      { S7_Templates := "SrcType := Real" } EQ_Contact(in1 := "C#6_WD_CALIB".XUNG_IND_AGG3, in2 := 32767.0)
   END_RUNG wire#w4
   RUNG wire#powerrail
      Contact( "7.1.IND_AGG3".STA_RUN )
      Coil( "C#1_RB".TTC_AG3 )
   END_RUNG
   // the same network as SCL:
   "9.1.DLC_IND_AGG3"(ON := "PLC_BIT".RUN AND NOT "PLC_BIT".AGG3_FU AND NOT "C#1_RB"."XA W_IND_AGG3",   // "9.TIMER_DELAY"
                      CLOCK_1S := "Clock_10Hz",
                      T_DELAY := "C#4_WD_WEIGHT"."W_IND_AGG3_TG.DLC",
                      OUT => "9.1.DLC_IND_AGG3".OUT,
                      T_OUT => "9.1.DLC_IND_AGG3".T_OUT);
   "7.1.IND_AGG3"(AUT := ("C#4_WD_WEIGHT".SV_AG3 <> 0.0) AND "PLC_BIT".RUN AND "PLC_BIT".AUT AND "9.1.DLC_IND_AGG3".OUT AND NOT "PLC_BIT".AGG3_FU AND ("C#7_RD_RUN".SMC_AG3 = "C#7_RD_RUN".SMX_AG3) AND ("C#7_RD_RUN".SMC_AG3 < "C#7_RD_RUN".SMT),   // "7.WEIGHT_PROCESS"
                  MAN1 := "C#2_WB"."NN_CAN AG3" OR "XA_HET_AGG",
                  FAU := "C#2_WB".F2_SW_PAU OR "C#2_WB".SW_PA_AG3 OR ("C#6_WD_CALIB".XUNG_IND_AGG3 = 32767.0),
                  FU_IN := "C#2_WB".NN_FU_AG3,
                  X_CLOCK := "Clock_10Hz",
                  EMTY_IN := "PLC_BIT".WAG3_EM,
                  XNC_AUT := TRUE,
                  SV_IN := "C#4_WD_WEIGHT".SV_AG3,
                  W_IN := "6.1.W_IND_AGG3".W_OUT1,
                  W_RTD := "C#3_WD_SILO".AG3_KL_RTD,
                  W_TR := "C#3_WD_SILO".AG3_SS_TREN,
                  W_DU := "C#3_WD_SILO".AG3_SS_DUOI,
                  T_ON := "C#3_WD_SILO".AG3_TG_ON_CAN,
                  T_OFF := "C#3_WD_SILO".AG3_TG_OFF_CAN,
                  T_DL := "C#3_WD_SILO".AG3_TG_ODC,
                  PV_OUT => "C#7_RD_RUN".PV_AG3,
                  PVM_OUT => "C#7_RD_RUN".PVM_AG3,
                  FU_OUT => "PLC_BIT".AGG3_FU,
                  Q_OUT1 => "C#1_RB"."CAN AG3",
                  STA_RUN => "7.1.IND_AGG3".STA_RUN);
   "C#1_RB".TTC_AG3 := "7.1.IND_AGG3".STA_RUN;
END_REGION
END_FUNCTION

FUNCTION "FCXL_IND_AGG4" : Void   // FC23, LAD
{ S7_Optimized_Access := 'TRUE' }
VERSION : 0.1
// stored: AutoNumber true, CodeModifiedDate 2026-01-15T16:25:53.5191681Z, CompileDate 2026-01-15T16:25:53.5611578Z, CreationDate 2026-01-15T16:24:02.4619467Z, HandleErrorsWithinBlock false, InterfaceModifiedDate 2026-01-11T04:48:18.8495033Z, IsConsistent true, IsIECCheckEnabled false, IsKnowHowProtected false, IsWriteProtected false, LibraryConformanceStatus Error: The block contains calls of single instances. Warning: The object contains access to global data blocks. Warning: The block contains direct access to inputs, outputs, bit memories, indirect access to the registry or indirect access to external memory areas that are unknown at the time of compilation., ModifiedDate 2026-01-15T16:25:53.5191681Z, ParameterModified 2026-01-11T04:48:18.8495033Z, PLCSimAdvancedSupport false, SetENOAutomatically False, StructureModified 2026-01-11T04:48:18.8495033Z, UDAEnableTagReadback false
   VAR_TEMP   // added for the SCL form of the ladder/FBD networks
      _w1 : Bool;
      _w2 : Bool;
      _w3 : Bool;
   END_VAR
BEGIN

REGION Network 1: Cân độc lập AGG4 Full
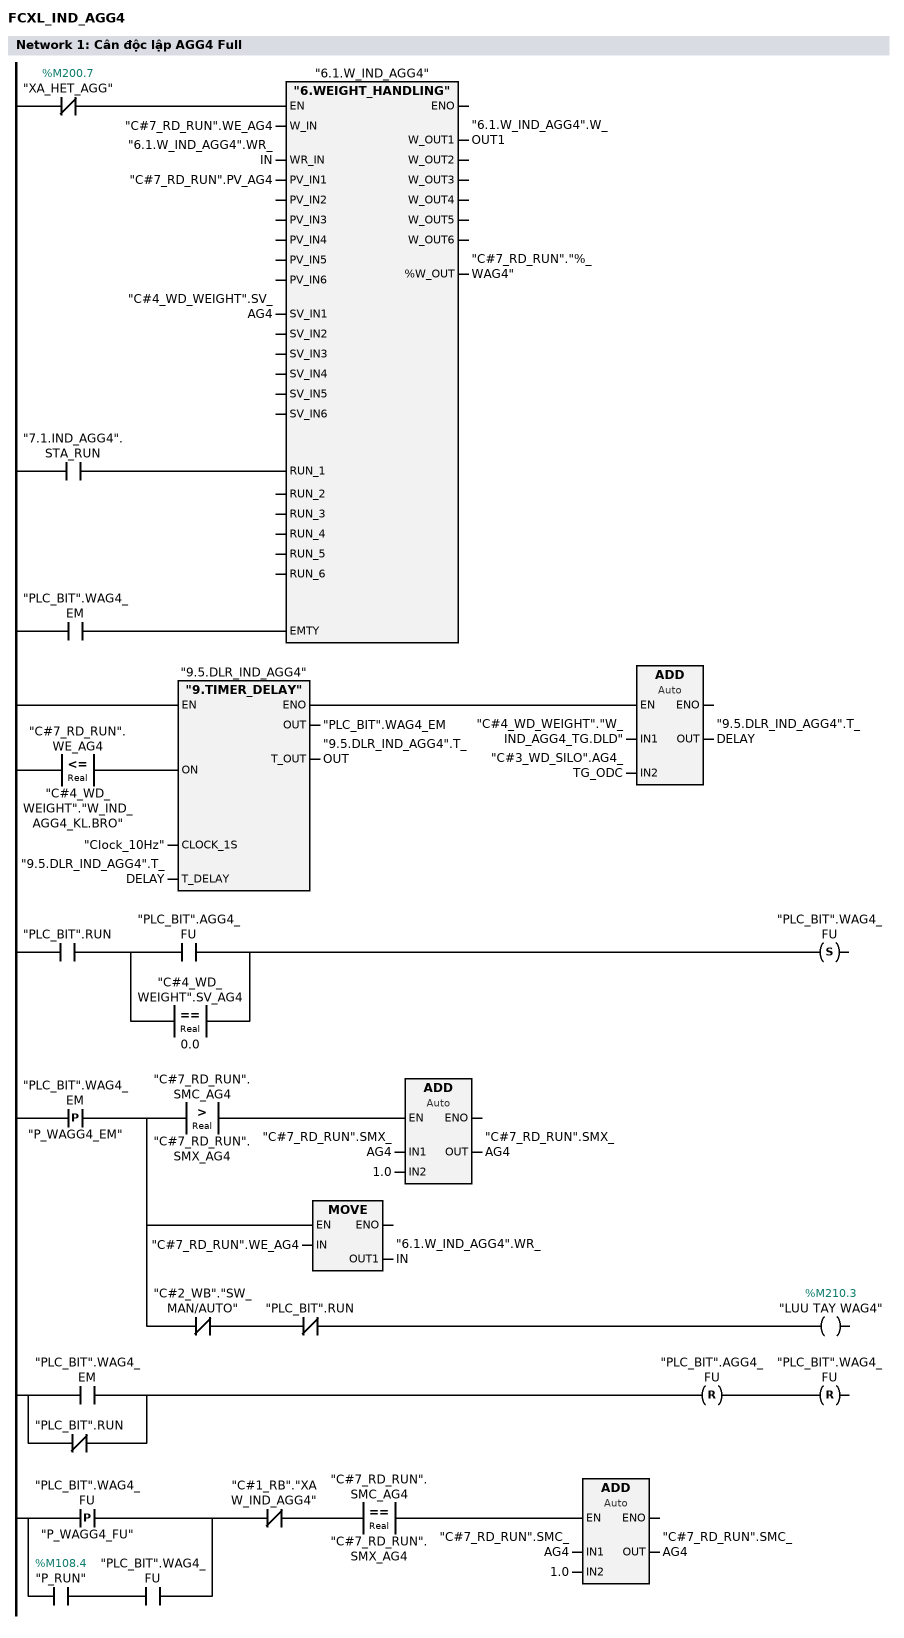
   RUNG wire#powerrail
      I_Contact( "XA_HET_AGG" )
      "6.1.W_IND_AGG4"(RUN_1 := wire#w1, EMTY := wire#w2, W_IN := "C#7_RD_RUN".WE_AG4, WR_IN := "6.1.W_IND_AGG4".WR_IN, PV_IN1 := "C#7_RD_RUN".PV_AG4, PV_IN2 :=, PV_IN3 :=, PV_IN4 :=, PV_IN5 :=, PV_IN6 :=, SV_IN1 := "C#4_WD_WEIGHT".SV_AG4, SV_IN2 :=, SV_IN3 :=, SV_IN4 :=, SV_IN5 :=, SV_IN6 :=, RUN_2 :=, RUN_3 :=, RUN_4 :=, RUN_5 :=, RUN_6 :=, W_OUT1 => "6.1.W_IND_AGG4".W_OUT1, W_OUT2 =>, W_OUT3 =>, W_OUT4 =>, W_OUT5 =>, W_OUT6 =>, "%W_OUT" => "C#7_RD_RUN"."%_WAG4")
   END_RUNG
   RUNG wire#powerrail
      Contact( "7.1.IND_AGG4".STA_RUN )
   END_RUNG wire#w1
   RUNG wire#powerrail
      Contact( "PLC_BIT".WAG4_EM )
   END_RUNG wire#w2
   RUNG wire#powerrail
      "9.5.DLR_IND_AGG4"(ON := wire#w3, CLOCK_1S := "Clock_10Hz", T_DELAY := "9.5.DLR_IND_AGG4".T_DELAY, OUT => "PLC_BIT".WAG4_EM, T_OUT => "9.5.DLR_IND_AGG4".T_OUT)
      Add(in1 := "C#4_WD_WEIGHT"."W_IND_AGG4_TG.DLD", in2 := "C#3_WD_SILO".AG4_TG_ODC, out => "9.5.DLR_IND_AGG4".T_DELAY)
   END_RUNG
   RUNG wire#powerrail
      { S7_Templates := "SrcType := Real" } LE_Contact(in1 := "C#7_RD_RUN".WE_AG4, in2 := "C#4_WD_WEIGHT"."W_IND_AGG4_KL.BRO")
   END_RUNG wire#w3
   RUNG wire#powerrail
      Contact( "PLC_BIT".RUN )
      wire#w4
      Contact( "PLC_BIT".AGG4_FU )
      wire#w5
      S_Coil( "PLC_BIT".WAG4_FU )
   END_RUNG
   RUNG wire#w4
      { S7_Templates := "SrcType := Real" } EQ_Contact(in1 := "C#4_WD_WEIGHT".SV_AG4, in2 := 0.0)
   END_RUNG wire#w5
   RUNG wire#powerrail
      P_Contact(operand := "PLC_BIT".WAG4_EM, bit := "P_WAGG4_EM")
      wire#w6
      { S7_Templates := "SrcType := Real" } GT_Contact(in1 := "C#7_RD_RUN".SMC_AG4, in2 := "C#7_RD_RUN".SMX_AG4)
      Add(in1 := "C#7_RD_RUN".SMX_AG4, in2 := 1.0, out => "C#7_RD_RUN".SMX_AG4)
   END_RUNG
   RUNG wire#w6
      Move(in := "C#7_RD_RUN".WE_AG4, out1 => "6.1.W_IND_AGG4".WR_IN)
   END_RUNG
   RUNG wire#w6
      I_Contact( "C#2_WB"."SW_MAN/AUTO" )
      I_Contact( "PLC_BIT".RUN )
      Coil( "LUU TAY WAG4" )
   END_RUNG
   RUNG wire#powerrail
      Contact( "PLC_BIT".WAG4_EM )
      wire#w7
      R_Coil( "PLC_BIT".AGG4_FU )
      R_Coil( "PLC_BIT".WAG4_FU )
   END_RUNG
   RUNG wire#powerrail
      I_Contact( "PLC_BIT".RUN )
   END_RUNG wire#w7
   RUNG wire#powerrail
      P_Contact(operand := "PLC_BIT".WAG4_FU, bit := "P_WAGG4_FU")
      wire#w8
      I_Contact( "C#1_RB"."XA W_IND_AGG4" )
      { S7_Templates := "SrcType := Real" } EQ_Contact(in1 := "C#7_RD_RUN".SMC_AG4, in2 := "C#7_RD_RUN".SMX_AG4)
      Add(in1 := "C#7_RD_RUN".SMC_AG4, in2 := 1.0, out => "C#7_RD_RUN".SMC_AG4)
   END_RUNG
   RUNG wire#powerrail
      Contact( "P_RUN" )
      Contact( "PLC_BIT".WAG4_FU )
   END_RUNG wire#w8
   // the same network as SCL:
   IF NOT "XA_HET_AGG" THEN
       "6.1.W_IND_AGG4"(W_IN := "C#7_RD_RUN".WE_AG4,   // "6.WEIGHT_HANDLING"
                        WR_IN := "6.1.W_IND_AGG4".WR_IN,
                        PV_IN1 := "C#7_RD_RUN".PV_AG4,
                        SV_IN1 := "C#4_WD_WEIGHT".SV_AG4,
                        RUN_1 := "7.1.IND_AGG4".STA_RUN,
                        EMTY := "PLC_BIT".WAG4_EM,
                        W_OUT1 => "6.1.W_IND_AGG4".W_OUT1,
                        "%W_OUT" => "C#7_RD_RUN"."%_WAG4");
   END_IF;
   "9.5.DLR_IND_AGG4"(ON := "C#7_RD_RUN".WE_AG4 <= "C#4_WD_WEIGHT"."W_IND_AGG4_KL.BRO",   // "9.TIMER_DELAY"
                      CLOCK_1S := "Clock_10Hz",
                      T_DELAY := "9.5.DLR_IND_AGG4".T_DELAY,
                      OUT => "PLC_BIT".WAG4_EM,
                      T_OUT => "9.5.DLR_IND_AGG4".T_OUT,
                      ENO => #_w1);
   IF #_w1 THEN
       "9.5.DLR_IND_AGG4".T_DELAY := "C#4_WD_WEIGHT"."W_IND_AGG4_TG.DLD" + "C#3_WD_SILO".AG4_TG_ODC;
   END_IF;
   IF "PLC_BIT".RUN AND ("PLC_BIT".AGG4_FU OR ("C#4_WD_WEIGHT".SV_AG4 = 0.0)) THEN
       "PLC_BIT".WAG4_FU := TRUE;
   END_IF;
   #_w2 := "PLC_BIT".WAG4_EM AND NOT "P_WAGG4_EM";   // rising edge of "PLC_BIT".WAG4_EM
   "P_WAGG4_EM" := "PLC_BIT".WAG4_EM;
   IF #_w2 AND ("C#7_RD_RUN".SMC_AG4 > "C#7_RD_RUN".SMX_AG4) THEN
       "C#7_RD_RUN".SMX_AG4 := "C#7_RD_RUN".SMX_AG4 + 1.0;
   END_IF;
   IF #_w2 THEN "6.1.W_IND_AGG4".WR_IN := "C#7_RD_RUN".WE_AG4; END_IF;
   "LUU TAY WAG4" := #_w2 AND NOT "C#2_WB"."SW_MAN/AUTO" AND NOT "PLC_BIT".RUN;
   IF "PLC_BIT".WAG4_EM OR NOT "PLC_BIT".RUN THEN
       "PLC_BIT".AGG4_FU := FALSE;
       "PLC_BIT".WAG4_FU := FALSE;
   END_IF;
   #_w3 := "PLC_BIT".WAG4_FU AND NOT "P_WAGG4_FU";   // rising edge of "PLC_BIT".WAG4_FU
   "P_WAGG4_FU" := "PLC_BIT".WAG4_FU;
   IF (#_w3 OR ("P_RUN" AND "PLC_BIT".WAG4_FU)) AND NOT "C#1_RB"."XA W_IND_AGG4" AND ("C#7_RD_RUN".SMC_AG4 = "C#7_RD_RUN".SMX_AG4) THEN
       "C#7_RD_RUN".SMC_AG4 := "C#7_RD_RUN".SMC_AG4 + 1.0;
   END_IF;
END_REGION
END_FUNCTION

FUNCTION "FCCA_IND_AGG4" : Void   // FC13, LAD
{ S7_Optimized_Access := 'TRUE' }
VERSION : 0.1
// stored: AutoNumber true, CodeModifiedDate 2026-01-15T16:25:54.6221046Z, CompileDate 2026-01-15T16:25:54.6613801Z, CreationDate 2026-01-15T16:24:02.4619467Z, HandleErrorsWithinBlock false, InterfaceModifiedDate 2026-01-11T04:46:59.531034Z, IsConsistent true, IsIECCheckEnabled false, IsKnowHowProtected false, IsWriteProtected false, LibraryConformanceStatus Error: The block contains calls of single instances. Warning: The object contains access to global data blocks. Warning: The block contains direct access to inputs, outputs, bit memories, indirect access to the registry or indirect access to external memory areas that are unknown at the time of compilation., ModifiedDate 2026-01-15T16:25:54.6221046Z, ParameterModified 2026-01-11T04:46:59.531034Z, PLCSimAdvancedSupport false, SetENOAutomatically False, StructureModified 2026-01-11T04:46:59.531034Z, UDAEnableTagReadback false
BEGIN

REGION Network 1: Trạng thái cân AGG4
   // Đầu tiên nó sẽ đợi một khoảng thời gian gọi là Thời gian trễ cân, sau đó nó mới đủ điều kiện để cân
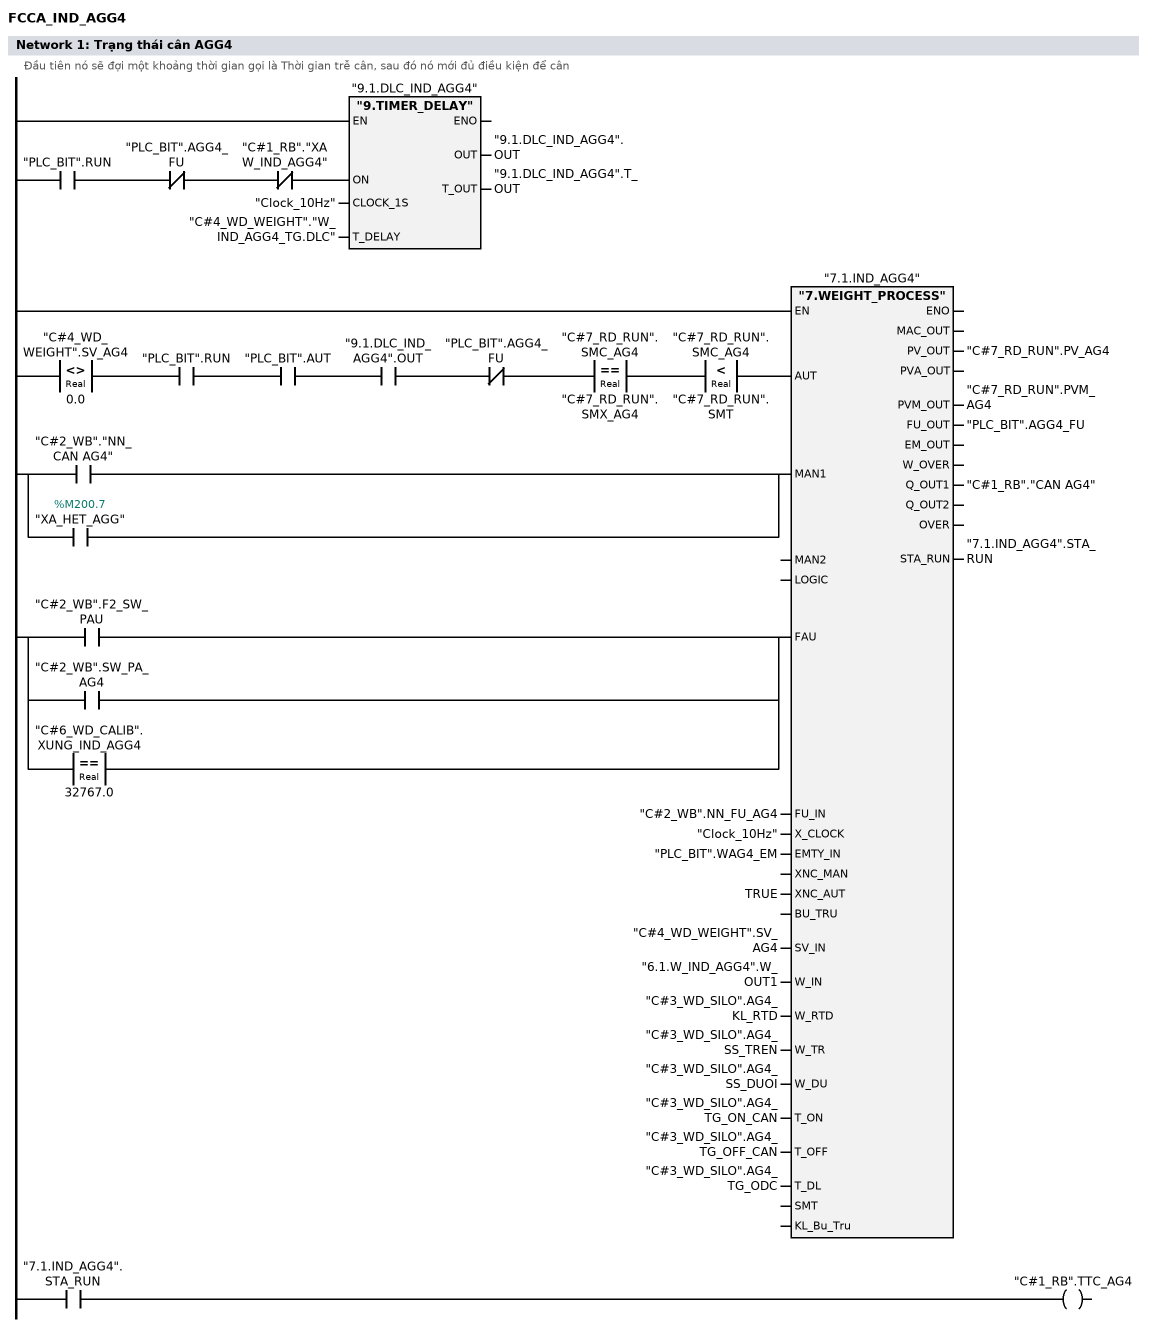
   RUNG wire#powerrail
      "9.1.DLC_IND_AGG4"(ON := wire#w1, CLOCK_1S := "Clock_10Hz", T_DELAY := "C#4_WD_WEIGHT"."W_IND_AGG4_TG.DLC", OUT => "9.1.DLC_IND_AGG4".OUT, T_OUT => "9.1.DLC_IND_AGG4".T_OUT)
   END_RUNG
   RUNG wire#powerrail
      Contact( "PLC_BIT".RUN )
      I_Contact( "PLC_BIT".AGG4_FU )
      I_Contact( "C#1_RB"."XA W_IND_AGG4" )
   END_RUNG wire#w1
   RUNG wire#powerrail
      "7.1.IND_AGG4"(AUT := wire#w2, MAN1 := wire#w3, FAU := wire#w4, MAN2 :=, LOGIC :=, FU_IN := "C#2_WB".NN_FU_AG4, X_CLOCK := "Clock_10Hz", EMTY_IN := "PLC_BIT".WAG4_EM, XNC_MAN :=, XNC_AUT := TRUE, BU_TRU :=, SV_IN := "C#4_WD_WEIGHT".SV_AG4, W_IN := "6.1.W_IND_AGG4".W_OUT1, W_RTD := "C#3_WD_SILO".AG4_KL_RTD, W_TR := "C#3_WD_SILO".AG4_SS_TREN, W_DU := "C#3_WD_SILO".AG4_SS_DUOI, T_ON := "C#3_WD_SILO".AG4_TG_ON_CAN, T_OFF := "C#3_WD_SILO".AG4_TG_OFF_CAN, T_DL := "C#3_WD_SILO".AG4_TG_ODC, SMT :=, KL_Bu_Tru :=, MAC_OUT =>, PV_OUT => "C#7_RD_RUN".PV_AG4, PVA_OUT =>, PVM_OUT => "C#7_RD_RUN".PVM_AG4, FU_OUT => "PLC_BIT".AGG4_FU, EM_OUT =>, W_OVER =>, Q_OUT1 => "C#1_RB"."CAN AG4", Q_OUT2 =>, OVER =>, STA_RUN => "7.1.IND_AGG4".STA_RUN)
   END_RUNG
   RUNG wire#powerrail
      { S7_Templates := "SrcType := Real" } NE_Contact(in1 := "C#4_WD_WEIGHT".SV_AG4, in2 := 0.0)
      Contact( "PLC_BIT".RUN )
      Contact( "PLC_BIT".AUT )
      Contact( "9.1.DLC_IND_AGG4".OUT )
      I_Contact( "PLC_BIT".AGG4_FU )
      { S7_Templates := "SrcType := Real" } EQ_Contact(in1 := "C#7_RD_RUN".SMC_AG4, in2 := "C#7_RD_RUN".SMX_AG4)
      { S7_Templates := "SrcType := Real" } LT_Contact(in1 := "C#7_RD_RUN".SMC_AG4, in2 := "C#7_RD_RUN".SMT)
   END_RUNG wire#w2
   RUNG wire#powerrail
      Contact( "C#2_WB"."NN_CAN AG4" )
   END_RUNG wire#w3
   RUNG wire#powerrail
      Contact( "XA_HET_AGG" )
   END_RUNG wire#w3
   RUNG wire#powerrail
      Contact( "C#2_WB".F2_SW_PAU )
   END_RUNG wire#w4
   RUNG wire#powerrail
      Contact( "C#2_WB".SW_PA_AG4 )
   END_RUNG wire#w4
   RUNG wire#powerrail
      { S7_Templates := "SrcType := Real" } EQ_Contact(in1 := "C#6_WD_CALIB".XUNG_IND_AGG4, in2 := 32767.0)
   END_RUNG wire#w4
   RUNG wire#powerrail
      Contact( "7.1.IND_AGG4".STA_RUN )
      Coil( "C#1_RB".TTC_AG4 )
   END_RUNG
   // the same network as SCL:
   "9.1.DLC_IND_AGG4"(ON := "PLC_BIT".RUN AND NOT "PLC_BIT".AGG4_FU AND NOT "C#1_RB"."XA W_IND_AGG4",   // "9.TIMER_DELAY"
                      CLOCK_1S := "Clock_10Hz",
                      T_DELAY := "C#4_WD_WEIGHT"."W_IND_AGG4_TG.DLC",
                      OUT => "9.1.DLC_IND_AGG4".OUT,
                      T_OUT => "9.1.DLC_IND_AGG4".T_OUT);
   "7.1.IND_AGG4"(AUT := ("C#4_WD_WEIGHT".SV_AG4 <> 0.0) AND "PLC_BIT".RUN AND "PLC_BIT".AUT AND "9.1.DLC_IND_AGG4".OUT AND NOT "PLC_BIT".AGG4_FU AND ("C#7_RD_RUN".SMC_AG4 = "C#7_RD_RUN".SMX_AG4) AND ("C#7_RD_RUN".SMC_AG4 < "C#7_RD_RUN".SMT),   // "7.WEIGHT_PROCESS"
                  MAN1 := "C#2_WB"."NN_CAN AG4" OR "XA_HET_AGG",
                  FAU := "C#2_WB".F2_SW_PAU OR "C#2_WB".SW_PA_AG4 OR ("C#6_WD_CALIB".XUNG_IND_AGG4 = 32767.0),
                  FU_IN := "C#2_WB".NN_FU_AG4,
                  X_CLOCK := "Clock_10Hz",
                  EMTY_IN := "PLC_BIT".WAG4_EM,
                  XNC_AUT := TRUE,
                  SV_IN := "C#4_WD_WEIGHT".SV_AG4,
                  W_IN := "6.1.W_IND_AGG4".W_OUT1,
                  W_RTD := "C#3_WD_SILO".AG4_KL_RTD,
                  W_TR := "C#3_WD_SILO".AG4_SS_TREN,
                  W_DU := "C#3_WD_SILO".AG4_SS_DUOI,
                  T_ON := "C#3_WD_SILO".AG4_TG_ON_CAN,
                  T_OFF := "C#3_WD_SILO".AG4_TG_OFF_CAN,
                  T_DL := "C#3_WD_SILO".AG4_TG_ODC,
                  PV_OUT => "C#7_RD_RUN".PV_AG4,
                  PVM_OUT => "C#7_RD_RUN".PVM_AG4,
                  FU_OUT => "PLC_BIT".AGG4_FU,
                  Q_OUT1 => "C#1_RB"."CAN AG4",
                  STA_RUN => "7.1.IND_AGG4".STA_RUN);
   "C#1_RB".TTC_AG4 := "7.1.IND_AGG4".STA_RUN;
END_REGION
END_FUNCTION

FUNCTION "FCXL_IND_AGG5" : Void   // FC24, LAD
{ S7_Optimized_Access := 'TRUE' }
VERSION : 0.1
// stored: AutoNumber true, CodeModifiedDate 2026-01-15T16:25:53.434175Z, CompileDate 2026-01-15T16:25:53.4741475Z, CreationDate 2026-01-15T16:24:02.4619467Z, HandleErrorsWithinBlock false, InterfaceModifiedDate 2026-01-11T04:48:35.7683688Z, IsConsistent true, IsIECCheckEnabled false, IsKnowHowProtected false, IsWriteProtected false, LibraryConformanceStatus Error: The block contains calls of single instances. Warning: The object contains access to global data blocks. Warning: The block contains direct access to inputs, outputs, bit memories, indirect access to the registry or indirect access to external memory areas that are unknown at the time of compilation., ModifiedDate 2026-01-15T16:25:53.434175Z, ParameterModified 2026-01-11T04:48:35.7683688Z, PLCSimAdvancedSupport false, SetENOAutomatically False, StructureModified 2026-01-11T04:48:35.7683688Z, UDAEnableTagReadback false
   VAR_TEMP   // added for the SCL form of the ladder/FBD networks
      _w1 : Bool;
      _w2 : Bool;
      _w3 : Bool;
   END_VAR
BEGIN

